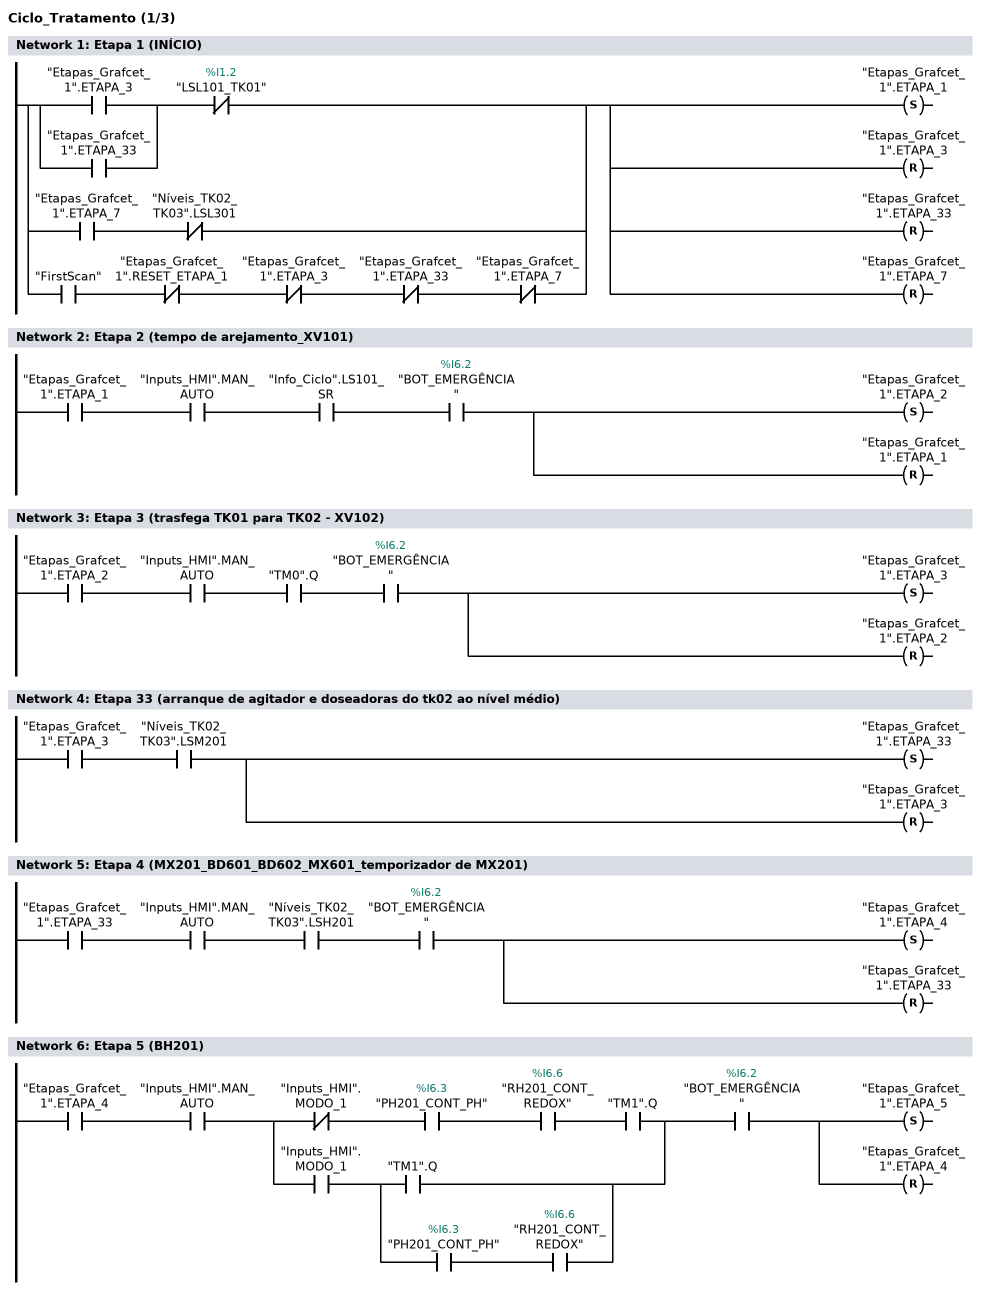
   RUNG wire#powerrail
      Contact( "Etapas_Grafcet_1".ETAPA_3 )
      wire#w1
      I_Contact( "LSL101_TK01" )
      wire#w2
      S_Coil( "Etapas_Grafcet_1".ETAPA_1 )
   END_RUNG
   RUNG wire#powerrail
      Contact( "Etapas_Grafcet_1".ETAPA_33 )
   END_RUNG wire#w1
   RUNG wire#powerrail
      Contact( "Etapas_Grafcet_1".ETAPA_7 )
      I_Contact( "Níveis_TK02_TK03".LSL301 )
   END_RUNG wire#w2
   RUNG wire#powerrail
      Contact( "FirstScan" )
      I_Contact( "Etapas_Grafcet_1".RESET_ETAPA_1 )
      I_Contact( "Etapas_Grafcet_1".ETAPA_3 )
      I_Contact( "Etapas_Grafcet_1".ETAPA_33 )
      I_Contact( "Etapas_Grafcet_1".ETAPA_7 )
   END_RUNG wire#w2
   RUNG wire#w2
      R_Coil( "Etapas_Grafcet_1".ETAPA_3 )
   END_RUNG
   RUNG wire#w2
      R_Coil( "Etapas_Grafcet_1".ETAPA_33 )
   END_RUNG
   RUNG wire#w2
      R_Coil( "Etapas_Grafcet_1".ETAPA_7 )
   END_RUNG
   // the same network as SCL:
   IF (("Etapas_Grafcet_1".ETAPA_3 OR "Etapas_Grafcet_1".ETAPA_33) AND NOT "LSL101_TK01") OR ("Etapas_Grafcet_1".ETAPA_7 AND NOT "Níveis_TK02_TK03".LSL301) OR ("FirstScan" AND NOT "Etapas_Grafcet_1".RESET_ETAPA_1 AND NOT "Etapas_Grafcet_1".ETAPA_3 AND NOT "Etapas_Grafcet_1".ETAPA_33 AND NOT "Etapas_Grafcet_1".ETAPA_7) THEN
       "Etapas_Grafcet_1".ETAPA_1 := TRUE;
   END_IF;
   #_w1 := (("Etapas_Grafcet_1".ETAPA_3 OR "Etapas_Grafcet_1".ETAPA_33) AND NOT "LSL101_TK01") OR ("Etapas_Grafcet_1".ETAPA_7 AND NOT "Níveis_TK02_TK03".LSL301) OR ("FirstScan" AND NOT "Etapas_Grafcet_1".RESET_ETAPA_1 AND NOT "Etapas_Grafcet_1".ETAPA_3 AND NOT "Etapas_Grafcet_1".ETAPA_33 AND NOT "Etapas_Grafcet_1".ETAPA_7);
   IF #_w1 THEN
       "Etapas_Grafcet_1".ETAPA_3 := FALSE;
       "Etapas_Grafcet_1".ETAPA_33 := FALSE;
       "Etapas_Grafcet_1".ETAPA_7 := FALSE;
   END_IF;
END_REGION

REGION Network 2: Etapa 2 (tempo de arejamento_XV101)
   RUNG wire#powerrail
      Contact( "Etapas_Grafcet_1".ETAPA_1 )
      Contact( "Inputs_HMI".MAN_AUTO )
      Contact( "Info_Ciclo".LS101_SR )
      Contact( "BOT_EMERGÊNCIA" )
      wire#w1
      S_Coil( "Etapas_Grafcet_1".ETAPA_2 )
   END_RUNG
   RUNG wire#w1
      R_Coil( "Etapas_Grafcet_1".ETAPA_1 )
   END_RUNG
   // the same network as SCL:
   IF "Etapas_Grafcet_1".ETAPA_1 AND "Inputs_HMI".MAN_AUTO AND "Info_Ciclo".LS101_SR AND "BOT_EMERGÊNCIA" THEN
       "Etapas_Grafcet_1".ETAPA_2 := TRUE;
       "Etapas_Grafcet_1".ETAPA_1 := FALSE;
   END_IF;
END_REGION

REGION Network 3: Etapa 3 (trasfega TK01 para TK02 - XV102)
   RUNG wire#powerrail
      Contact( "Etapas_Grafcet_1".ETAPA_2 )
      Contact( "Inputs_HMI".MAN_AUTO )
      Contact( "TM0".Q )
      Contact( "BOT_EMERGÊNCIA" )
      wire#w1
      S_Coil( "Etapas_Grafcet_1".ETAPA_3 )
   END_RUNG
   RUNG wire#w1
      R_Coil( "Etapas_Grafcet_1".ETAPA_2 )
   END_RUNG
   // the same network as SCL:
   IF "Etapas_Grafcet_1".ETAPA_2 AND "Inputs_HMI".MAN_AUTO AND "TM0".Q AND "BOT_EMERGÊNCIA" THEN
       "Etapas_Grafcet_1".ETAPA_3 := TRUE;
       "Etapas_Grafcet_1".ETAPA_2 := FALSE;
   END_IF;
END_REGION

REGION Network 4: Etapa 33 (arranque de agitador e doseadoras do tk02 ao nível médio)
   RUNG wire#powerrail
      Contact( "Etapas_Grafcet_1".ETAPA_3 )
      Contact( "Níveis_TK02_TK03".LSM201 )
      wire#w1
      S_Coil( "Etapas_Grafcet_1".ETAPA_33 )
   END_RUNG
   RUNG wire#w1
      R_Coil( "Etapas_Grafcet_1".ETAPA_3 )
   END_RUNG
   // the same network as SCL:
   IF "Etapas_Grafcet_1".ETAPA_3 AND "Níveis_TK02_TK03".LSM201 THEN
       "Etapas_Grafcet_1".ETAPA_33 := TRUE;
       "Etapas_Grafcet_1".ETAPA_3 := FALSE;
   END_IF;
END_REGION

REGION Network 5: Etapa 4 (MX201_BD601_BD602_MX601_temporizador de MX201)
   RUNG wire#powerrail
      Contact( "Etapas_Grafcet_1".ETAPA_33 )
      Contact( "Inputs_HMI".MAN_AUTO )
      Contact( "Níveis_TK02_TK03".LSH201 )
      Contact( "BOT_EMERGÊNCIA" )
      wire#w1
      S_Coil( "Etapas_Grafcet_1".ETAPA_4 )
   END_RUNG
   RUNG wire#w1
      R_Coil( "Etapas_Grafcet_1".ETAPA_33 )
   END_RUNG
   // the same network as SCL:
   IF "Etapas_Grafcet_1".ETAPA_33 AND "Inputs_HMI".MAN_AUTO AND "Níveis_TK02_TK03".LSH201 AND "BOT_EMERGÊNCIA" THEN
       "Etapas_Grafcet_1".ETAPA_4 := TRUE;
       "Etapas_Grafcet_1".ETAPA_33 := FALSE;
   END_IF;
END_REGION

REGION Network 6: Etapa 5 (BH201)
   RUNG wire#powerrail
      Contact( "Etapas_Grafcet_1".ETAPA_4 )
      Contact( "Inputs_HMI".MAN_AUTO )
      wire#w1
      I_Contact( "Inputs_HMI".MODO_1 )
      Contact( "PH201_CONT_PH" )
      Contact( "RH201_CONT_REDOX" )
      Contact( "TM1".Q )
      wire#w2
      Contact( "BOT_EMERGÊNCIA" )
      wire#w4
      S_Coil( "Etapas_Grafcet_1".ETAPA_5 )
   END_RUNG
   RUNG wire#w1
      Contact( "Inputs_HMI".MODO_1 )
      wire#w3
      Contact( "TM1".Q )
   END_RUNG wire#w2
   RUNG wire#w3
      Contact( "PH201_CONT_PH" )
      Contact( "RH201_CONT_REDOX" )
   END_RUNG wire#w2
   RUNG wire#w4
      R_Coil( "Etapas_Grafcet_1".ETAPA_4 )
   END_RUNG
   // the same network as SCL:
   IF "Etapas_Grafcet_1".ETAPA_4 AND "Inputs_HMI".MAN_AUTO AND ((NOT "Inputs_HMI".MODO_1 AND "PH201_CONT_PH" AND "RH201_CONT_REDOX" AND "TM1".Q) OR ("Inputs_HMI".MODO_1 AND ("TM1".Q OR ("PH201_CONT_PH" AND "RH201_CONT_REDOX")))) AND "BOT_EMERGÊNCIA" THEN
       "Etapas_Grafcet_1".ETAPA_5 := TRUE;
       "Etapas_Grafcet_1".ETAPA_4 := FALSE;
   END_IF;
END_REGION

REGION Network 7: Etapa 55 (arranque de agitador e doseadoras do tk03 ao nível médio)
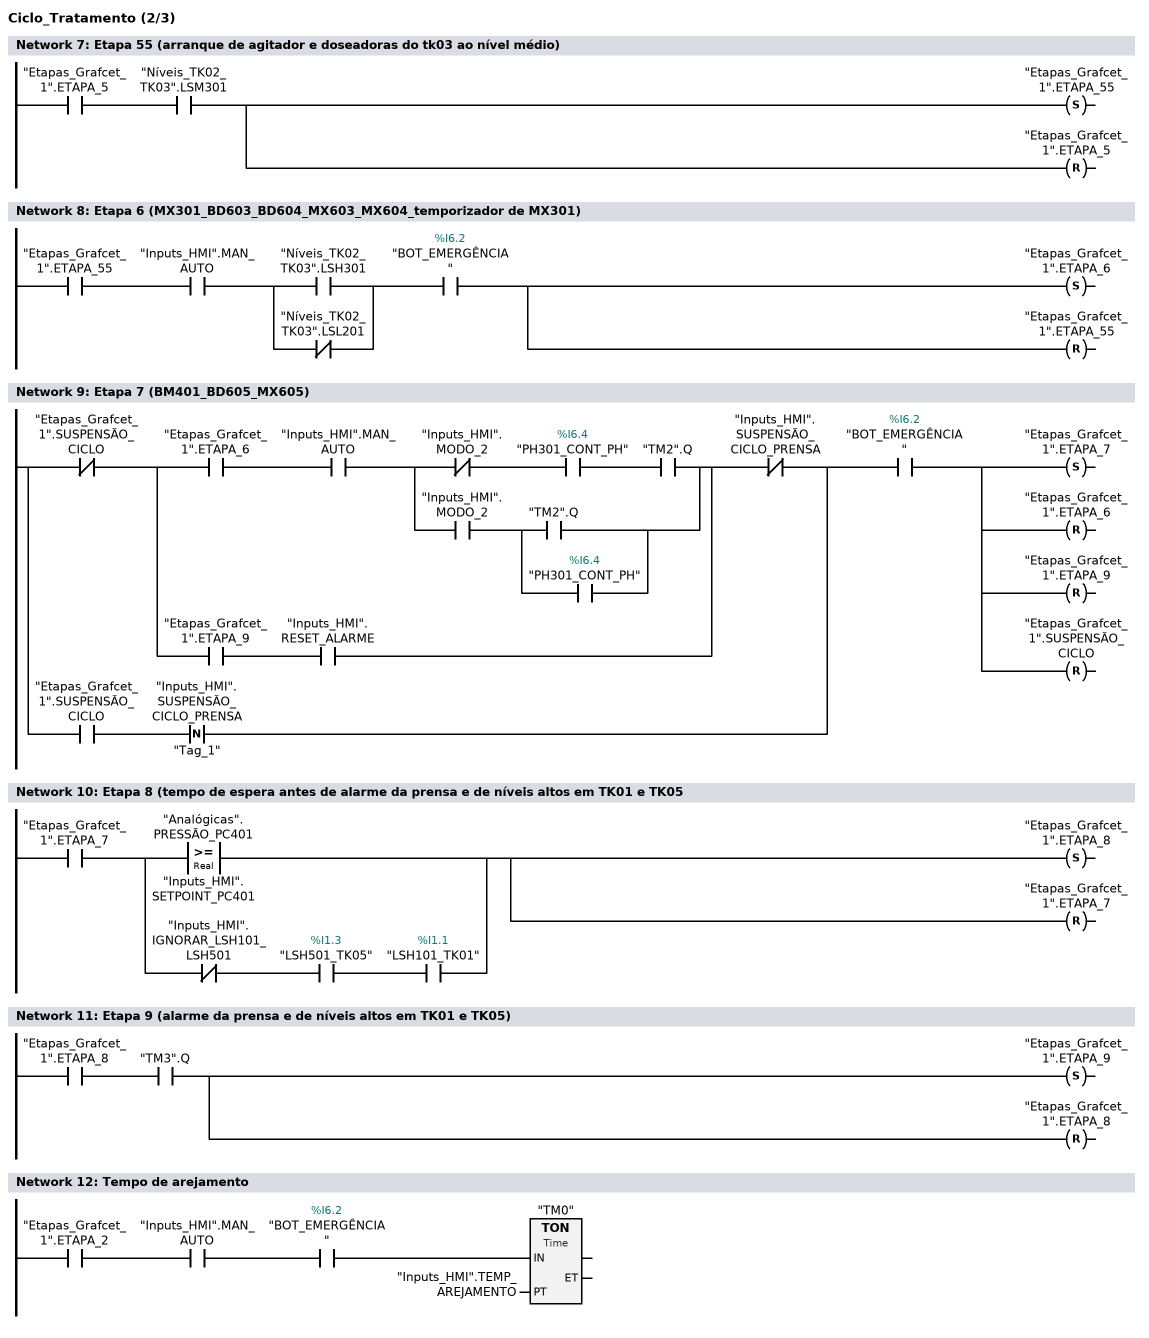
   RUNG wire#powerrail
      Contact( "Etapas_Grafcet_1".ETAPA_5 )
      Contact( "Níveis_TK02_TK03".LSM301 )
      wire#w1
      S_Coil( "Etapas_Grafcet_1".ETAPA_55 )
   END_RUNG
   RUNG wire#w1
      R_Coil( "Etapas_Grafcet_1".ETAPA_5 )
   END_RUNG
   // the same network as SCL:
   IF "Etapas_Grafcet_1".ETAPA_5 AND "Níveis_TK02_TK03".LSM301 THEN
       "Etapas_Grafcet_1".ETAPA_55 := TRUE;
       "Etapas_Grafcet_1".ETAPA_5 := FALSE;
   END_IF;
END_REGION

REGION Network 8: Etapa 6 (MX301_BD603_BD604_MX603_MX604_temporizador de MX301)
   RUNG wire#powerrail
      Contact( "Etapas_Grafcet_1".ETAPA_55 )
      Contact( "Inputs_HMI".MAN_AUTO )
      wire#w1
      Contact( "Níveis_TK02_TK03".LSH301 )
      wire#w2
      Contact( "BOT_EMERGÊNCIA" )
      wire#w3
      S_Coil( "Etapas_Grafcet_1".ETAPA_6 )
   END_RUNG
   RUNG wire#w1
      I_Contact( "Níveis_TK02_TK03".LSL201 )
   END_RUNG wire#w2
   RUNG wire#w3
      R_Coil( "Etapas_Grafcet_1".ETAPA_55 )
   END_RUNG
   // the same network as SCL:
   IF "Etapas_Grafcet_1".ETAPA_55 AND "Inputs_HMI".MAN_AUTO AND ("Níveis_TK02_TK03".LSH301 OR NOT "Níveis_TK02_TK03".LSL201) AND "BOT_EMERGÊNCIA" THEN
       "Etapas_Grafcet_1".ETAPA_6 := TRUE;
       "Etapas_Grafcet_1".ETAPA_55 := FALSE;
   END_IF;
END_REGION

REGION Network 9: Etapa 7 (BM401_BD605_MX605)
   RUNG wire#powerrail
      I_Contact( "Etapas_Grafcet_1".SUSPENSÃO_CICLO )
      wire#w1
      Contact( "Etapas_Grafcet_1".ETAPA_6 )
      Contact( "Inputs_HMI".MAN_AUTO )
      wire#w2
      I_Contact( "Inputs_HMI".MODO_2 )
      Contact( "PH301_CONT_PH" )
      Contact( "TM2".Q )
      wire#w3
      I_Contact( "Inputs_HMI".SUSPENSÃO_CICLO_PRENSA )
      wire#w5
      Contact( "BOT_EMERGÊNCIA" )
      wire#w6
      S_Coil( "Etapas_Grafcet_1".ETAPA_7 )
   END_RUNG
   RUNG wire#w2
      Contact( "Inputs_HMI".MODO_2 )
      wire#w4
      Contact( "TM2".Q )
   END_RUNG wire#w3
   RUNG wire#w4
      Contact( "PH301_CONT_PH" )
   END_RUNG wire#w3
   RUNG wire#w1
      Contact( "Etapas_Grafcet_1".ETAPA_9 )
      Contact( "Inputs_HMI".RESET_ALARME )
   END_RUNG wire#w3
   RUNG wire#powerrail
      Contact( "Etapas_Grafcet_1".SUSPENSÃO_CICLO )
      N_Contact(operand := "Inputs_HMI".SUSPENSÃO_CICLO_PRENSA, bit := "Tag_1")
   END_RUNG wire#w5
   RUNG wire#w6
      R_Coil( "Etapas_Grafcet_1".ETAPA_6 )
   END_RUNG
   RUNG wire#w6
      R_Coil( "Etapas_Grafcet_1".ETAPA_9 )
   END_RUNG
   RUNG wire#w6
      R_Coil( "Etapas_Grafcet_1".SUSPENSÃO_CICLO )
   END_RUNG
   // the same network as SCL:
   #_w1 := "Etapas_Grafcet_1".SUSPENSÃO_CICLO AND NOT "Inputs_HMI".SUSPENSÃO_CICLO_PRENSA AND "Tag_1";   // falling edge of "Inputs_HMI".SUSPENSÃO_CICLO_PRENSA
   "Tag_1" := "Inputs_HMI".SUSPENSÃO_CICLO_PRENSA;
   IF ((NOT "Etapas_Grafcet_1".SUSPENSÃO_CICLO AND (("Etapas_Grafcet_1".ETAPA_6 AND "Inputs_HMI".MAN_AUTO AND ((NOT "Inputs_HMI".MODO_2 AND "PH301_CONT_PH" AND "TM2".Q) OR ("Inputs_HMI".MODO_2 AND ("TM2".Q OR "PH301_CONT_PH")))) OR ("Etapas_Grafcet_1".ETAPA_9 AND "Inputs_HMI".RESET_ALARME)) AND NOT "Inputs_HMI".SUSPENSÃO_CICLO_PRENSA) OR #_w1) AND "BOT_EMERGÊNCIA" THEN
       "Etapas_Grafcet_1".ETAPA_7 := TRUE;
   END_IF;
   #_w2 := ((NOT "Etapas_Grafcet_1".SUSPENSÃO_CICLO AND (("Etapas_Grafcet_1".ETAPA_6 AND "Inputs_HMI".MAN_AUTO AND ((NOT "Inputs_HMI".MODO_2 AND "PH301_CONT_PH" AND "TM2".Q) OR ("Inputs_HMI".MODO_2 AND ("TM2".Q OR "PH301_CONT_PH")))) OR ("Etapas_Grafcet_1".ETAPA_9 AND "Inputs_HMI".RESET_ALARME)) AND NOT "Inputs_HMI".SUSPENSÃO_CICLO_PRENSA) OR #_w1) AND "BOT_EMERGÊNCIA";
   IF #_w2 THEN
       "Etapas_Grafcet_1".ETAPA_6 := FALSE;
       "Etapas_Grafcet_1".ETAPA_9 := FALSE;
       "Etapas_Grafcet_1".SUSPENSÃO_CICLO := FALSE;
   END_IF;
END_REGION

REGION Network 10: Etapa 8 (tempo de espera antes de alarme da prensa e de níveis altos em TK01 e TK05
   RUNG wire#powerrail
      Contact( "Etapas_Grafcet_1".ETAPA_7 )
      wire#w1
      { S7_Templates := "SrcType := Real" } GE_Contact(in1 := "Analógicas".PRESSÃO_PC401, in2 := "Inputs_HMI".SETPOINT_PC401)
      wire#w2
      S_Coil( "Etapas_Grafcet_1".ETAPA_8 )
   END_RUNG
   RUNG wire#w1
      I_Contact( "Inputs_HMI".IGNORAR_LSH101_LSH501 )
      Contact( "LSH501_TK05" )
      Contact( "LSH101_TK01" )
   END_RUNG wire#w2
   RUNG wire#w2
      R_Coil( "Etapas_Grafcet_1".ETAPA_7 )
   END_RUNG
   // the same network as SCL:
   IF "Etapas_Grafcet_1".ETAPA_7 AND (("Analógicas".PRESSÃO_PC401 >= "Inputs_HMI".SETPOINT_PC401) OR (NOT "Inputs_HMI".IGNORAR_LSH101_LSH501 AND "LSH501_TK05" AND "LSH101_TK01")) THEN
       "Etapas_Grafcet_1".ETAPA_8 := TRUE;
       "Etapas_Grafcet_1".ETAPA_7 := FALSE;
   END_IF;
END_REGION

REGION Network 11: Etapa 9 (alarme da prensa e de níveis altos em TK01 e TK05)
   RUNG wire#powerrail
      Contact( "Etapas_Grafcet_1".ETAPA_8 )
      Contact( "TM3".Q )
      wire#w1
      S_Coil( "Etapas_Grafcet_1".ETAPA_9 )
   END_RUNG
   RUNG wire#w1
      R_Coil( "Etapas_Grafcet_1".ETAPA_8 )
   END_RUNG
   // the same network as SCL:
   IF "Etapas_Grafcet_1".ETAPA_8 AND "TM3".Q THEN
       "Etapas_Grafcet_1".ETAPA_9 := TRUE;
       "Etapas_Grafcet_1".ETAPA_8 := FALSE;
   END_IF;
END_REGION

REGION Network 12: Tempo de arejamento
   RUNG wire#powerrail
      Contact( "Etapas_Grafcet_1".ETAPA_2 )
      Contact( "Inputs_HMI".MAN_AUTO )
      Contact( "BOT_EMERGÊNCIA" )
      { S7_Templates := "time_type := Time" } "TM0".TON(pt := "Inputs_HMI".TEMP_AREJAMENTO, et =>)
   END_RUNG
   // the same network as SCL:
   "TM0".TON(IN := "Etapas_Grafcet_1".ETAPA_2 AND "Inputs_HMI".MAN_AUTO AND "BOT_EMERGÊNCIA",
             PT := "Inputs_HMI".TEMP_AREJAMENTO);
END_REGION

REGION Network 13: Etapa Suspensão Ciclo
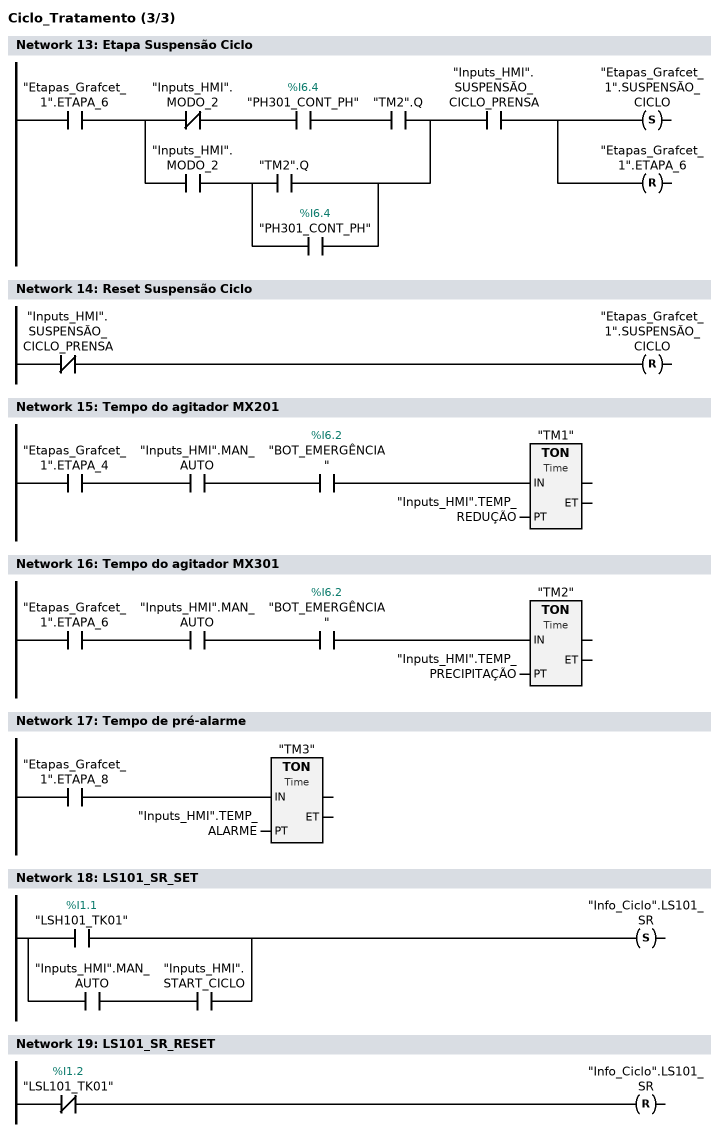
   RUNG wire#powerrail
      Contact( "Etapas_Grafcet_1".ETAPA_6 )
      wire#w1
      I_Contact( "Inputs_HMI".MODO_2 )
      Contact( "PH301_CONT_PH" )
      Contact( "TM2".Q )
      wire#w2
      Contact( "Inputs_HMI".SUSPENSÃO_CICLO_PRENSA )
      wire#w4
      S_Coil( "Etapas_Grafcet_1".SUSPENSÃO_CICLO )
   END_RUNG
   RUNG wire#w1
      Contact( "Inputs_HMI".MODO_2 )
      wire#w3
      Contact( "TM2".Q )
   END_RUNG wire#w2
   RUNG wire#w3
      Contact( "PH301_CONT_PH" )
   END_RUNG wire#w2
   RUNG wire#w4
      R_Coil( "Etapas_Grafcet_1".ETAPA_6 )
   END_RUNG
   // the same network as SCL:
   IF "Etapas_Grafcet_1".ETAPA_6 AND ((NOT "Inputs_HMI".MODO_2 AND "PH301_CONT_PH" AND "TM2".Q) OR ("Inputs_HMI".MODO_2 AND ("TM2".Q OR "PH301_CONT_PH"))) AND "Inputs_HMI".SUSPENSÃO_CICLO_PRENSA THEN
       "Etapas_Grafcet_1".SUSPENSÃO_CICLO := TRUE;
       "Etapas_Grafcet_1".ETAPA_6 := FALSE;
   END_IF;
END_REGION

REGION Network 14: Reset Suspensão Ciclo
   RUNG wire#powerrail
      I_Contact( "Inputs_HMI".SUSPENSÃO_CICLO_PRENSA )
      R_Coil( "Etapas_Grafcet_1".SUSPENSÃO_CICLO )
   END_RUNG
   // the same network as SCL:
   IF NOT "Inputs_HMI".SUSPENSÃO_CICLO_PRENSA THEN "Etapas_Grafcet_1".SUSPENSÃO_CICLO := FALSE; END_IF;
END_REGION

REGION Network 15: Tempo do agitador MX201
   RUNG wire#powerrail
      Contact( "Etapas_Grafcet_1".ETAPA_4 )
      Contact( "Inputs_HMI".MAN_AUTO )
      Contact( "BOT_EMERGÊNCIA" )
      { S7_Templates := "time_type := Time" } "TM1".TON(pt := "Inputs_HMI".TEMP_REDUÇÃO, et =>)
   END_RUNG
   // the same network as SCL:
   "TM1".TON(IN := "Etapas_Grafcet_1".ETAPA_4 AND "Inputs_HMI".MAN_AUTO AND "BOT_EMERGÊNCIA",
             PT := "Inputs_HMI".TEMP_REDUÇÃO);
END_REGION

REGION Network 16: Tempo do agitador MX301
   RUNG wire#powerrail
      Contact( "Etapas_Grafcet_1".ETAPA_6 )
      Contact( "Inputs_HMI".MAN_AUTO )
      Contact( "BOT_EMERGÊNCIA" )
      { S7_Templates := "time_type := Time" } "TM2".TON(pt := "Inputs_HMI".TEMP_PRECIPITAÇÃO, et =>)
   END_RUNG
   // the same network as SCL:
   "TM2".TON(IN := "Etapas_Grafcet_1".ETAPA_6 AND "Inputs_HMI".MAN_AUTO AND "BOT_EMERGÊNCIA",
             PT := "Inputs_HMI".TEMP_PRECIPITAÇÃO);
END_REGION

REGION Network 17: Tempo de pré-alarme
   RUNG wire#powerrail
      Contact( "Etapas_Grafcet_1".ETAPA_8 )
      { S7_Templates := "time_type := Time" } "TM3".TON(pt := "Inputs_HMI".TEMP_ALARME, et =>)
   END_RUNG
   // the same network as SCL:
   "TM3".TON(IN := "Etapas_Grafcet_1".ETAPA_8, PT := "Inputs_HMI".TEMP_ALARME);
END_REGION

REGION Network 18: LS101_SR_SET
   RUNG wire#powerrail
      Contact( "LSH101_TK01" )
      wire#w1
      S_Coil( "Info_Ciclo".LS101_SR )
   END_RUNG
   RUNG wire#powerrail
      Contact( "Inputs_HMI".MAN_AUTO )
      Contact( "Inputs_HMI".START_CICLO )
   END_RUNG wire#w1
   // the same network as SCL:
   IF "LSH101_TK01" OR ("Inputs_HMI".MAN_AUTO AND "Inputs_HMI".START_CICLO) THEN
       "Info_Ciclo".LS101_SR := TRUE;
   END_IF;
END_REGION

REGION Network 19: LS101_SR_RESET
   RUNG wire#powerrail
      I_Contact( "LSL101_TK01" )
      R_Coil( "Info_Ciclo".LS101_SR )
   END_RUNG
   // the same network as SCL:
   IF NOT "LSL101_TK01" THEN "Info_Ciclo".LS101_SR := FALSE; END_IF;
END_REGION
END_FUNCTION

FUNCTION "Estab_Níveis" : Void   // FC20, LAD
TITLE = Protege equipamentos e evita transbordo em modo manual
{ S7_Optimized_Access := 'TRUE' }
VERSION : 0.1
// stored: AutoNumber true, IsIECCheckEnabled false, SetENOAutomatically false, UDAEnableTagReadback false
BEGIN

REGION Network 1: LSL001
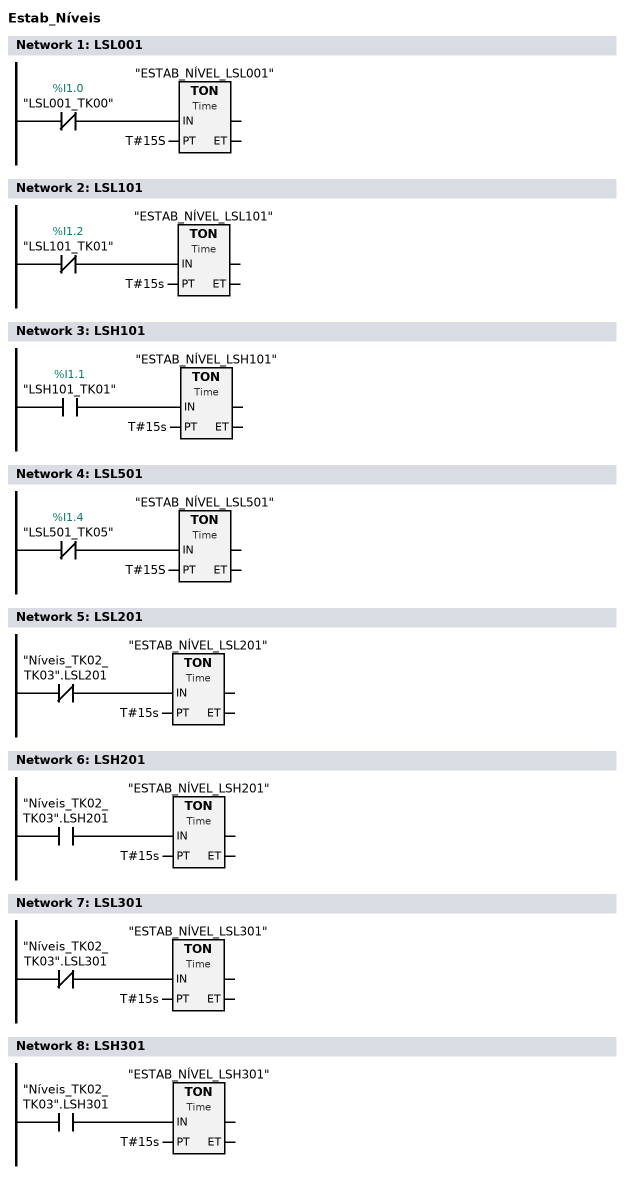
   RUNG wire#powerrail
      I_Contact( "LSL001_TK00" )
      { S7_Templates := "time_type := Time" } "ESTAB_NÍVEL_LSL001".TON(pt := T#15S, et =>)
   END_RUNG
   // the same network as SCL:
   "ESTAB_NÍVEL_LSL001".TON(IN := NOT "LSL001_TK00", PT := T#15S);
END_REGION

REGION Network 2: LSL101
   RUNG wire#powerrail
      I_Contact( "LSL101_TK01" )
      { S7_Templates := "time_type := Time" } "ESTAB_NÍVEL_LSL101".TON(pt := T#15s, et =>)
   END_RUNG
   // the same network as SCL:
   "ESTAB_NÍVEL_LSL101".TON(IN := NOT "LSL101_TK01", PT := T#15s);
END_REGION

REGION Network 3: LSH101
   RUNG wire#powerrail
      Contact( "LSH101_TK01" )
      { S7_Templates := "time_type := Time" } "ESTAB_NÍVEL_LSH101".TON(pt := T#15s, et =>)
   END_RUNG
   // the same network as SCL:
   "ESTAB_NÍVEL_LSH101".TON(IN := "LSH101_TK01", PT := T#15s);
END_REGION

REGION Network 4: LSL501
   RUNG wire#powerrail
      I_Contact( "LSL501_TK05" )
      { S7_Templates := "time_type := Time" } "ESTAB_NÍVEL_LSL501".TON(pt := T#15S, et =>)
   END_RUNG
   // the same network as SCL:
   "ESTAB_NÍVEL_LSL501".TON(IN := NOT "LSL501_TK05", PT := T#15S);
END_REGION

REGION Network 5: LSL201
   RUNG wire#powerrail
      I_Contact( "Níveis_TK02_TK03".LSL201 )
      { S7_Templates := "time_type := Time" } "ESTAB_NÍVEL_LSL201".TON(pt := T#15s, et =>)
   END_RUNG
   // the same network as SCL:
   "ESTAB_NÍVEL_LSL201".TON(IN := NOT "Níveis_TK02_TK03".LSL201, PT := T#15s);
END_REGION

REGION Network 6: LSH201
   RUNG wire#powerrail
      Contact( "Níveis_TK02_TK03".LSH201 )
      { S7_Templates := "time_type := Time" } "ESTAB_NÍVEL_LSH201".TON(pt := T#15s, et =>)
   END_RUNG
   // the same network as SCL:
   "ESTAB_NÍVEL_LSH201".TON(IN := "Níveis_TK02_TK03".LSH201, PT := T#15s);
END_REGION

REGION Network 7: LSL301
   RUNG wire#powerrail
      I_Contact( "Níveis_TK02_TK03".LSL301 )
      { S7_Templates := "time_type := Time" } "ESTAB_NÍVEL_LSL301".TON(pt := T#15s, et =>)
   END_RUNG
   // the same network as SCL:
   "ESTAB_NÍVEL_LSL301".TON(IN := NOT "Níveis_TK02_TK03".LSL301, PT := T#15s);
END_REGION

REGION Network 8: LSH301
   RUNG wire#powerrail
      Contact( "Níveis_TK02_TK03".LSH301 )
      { S7_Templates := "time_type := Time" } "ESTAB_NÍVEL_LSH301".TON(pt := T#15s, et =>)
   END_RUNG
   // the same network as SCL:
   "ESTAB_NÍVEL_LSH301".TON(IN := "Níveis_TK02_TK03".LSH301, PT := T#15s);
END_REGION
END_FUNCTION

FUNCTION "Reset_Etapas_Iniciais" : Void   // FC23, LAD
TITLE = Reset às etapas inicias em caso de falha de energia, de modo e continuar o processo do ponto onde estava
{ S7_Optimized_Access := 'TRUE' }
VERSION : 0.1
// stored: AutoNumber true, IsIECCheckEnabled false, SetENOAutomatically false, UDAEnableTagReadback false
BEGIN

REGION Network 1: Reset etapa 1
   // as etapas 3, 33 e 7 não precisam nem devem fazer reset à etapa 1. Já é feito indiretamente no FC4
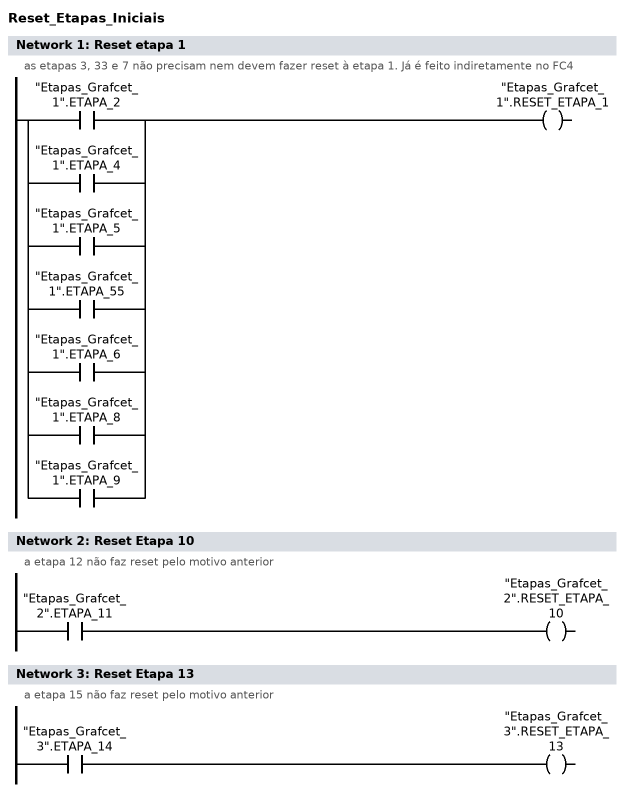
   RUNG wire#powerrail
      Contact( "Etapas_Grafcet_1".ETAPA_2 )
      wire#w1
      Coil( "Etapas_Grafcet_1".RESET_ETAPA_1 )
   END_RUNG
   RUNG wire#powerrail
      Contact( "Etapas_Grafcet_1".ETAPA_4 )
   END_RUNG wire#w1
   RUNG wire#powerrail
      Contact( "Etapas_Grafcet_1".ETAPA_5 )
   END_RUNG wire#w1
   RUNG wire#powerrail
      Contact( "Etapas_Grafcet_1".ETAPA_55 )
   END_RUNG wire#w1
   RUNG wire#powerrail
      Contact( "Etapas_Grafcet_1".ETAPA_6 )
   END_RUNG wire#w1
   RUNG wire#powerrail
      Contact( "Etapas_Grafcet_1".ETAPA_8 )
   END_RUNG wire#w1
   RUNG wire#powerrail
      Contact( "Etapas_Grafcet_1".ETAPA_9 )
   END_RUNG wire#w1
   // the same network as SCL:
   "Etapas_Grafcet_1".RESET_ETAPA_1 := "Etapas_Grafcet_1".ETAPA_2 OR "Etapas_Grafcet_1".ETAPA_4 OR "Etapas_Grafcet_1".ETAPA_5 OR "Etapas_Grafcet_1".ETAPA_55 OR "Etapas_Grafcet_1".ETAPA_6 OR "Etapas_Grafcet_1".ETAPA_8 OR "Etapas_Grafcet_1".ETAPA_9;
END_REGION

REGION Network 2: Reset Etapa 10
   // a etapa 12 não faz reset pelo motivo anterior
   RUNG wire#powerrail
      Contact( "Etapas_Grafcet_2".ETAPA_11 )
      Coil( "Etapas_Grafcet_2".RESET_ETAPA_10 )
   END_RUNG
   // the same network as SCL:
   "Etapas_Grafcet_2".RESET_ETAPA_10 := "Etapas_Grafcet_2".ETAPA_11;
END_REGION

REGION Network 3: Reset Etapa 13
   // a etapa 15 não faz reset pelo motivo anterior
   RUNG wire#powerrail
      Contact( "Etapas_Grafcet_3".ETAPA_14 )
      Coil( "Etapas_Grafcet_3".RESET_ETAPA_13 )
   END_RUNG
   // the same network as SCL:
   "Etapas_Grafcet_3".RESET_ETAPA_13 := "Etapas_Grafcet_3".ETAPA_14;
END_REGION
END_FUNCTION

FUNCTION "Saídas" : Void   // FC2, LAD
{ S7_Optimized_Access := 'TRUE' }
VERSION : 0.1
// stored: AutoNumber true, IsIECCheckEnabled false, SetENOAutomatically false, UDAEnableTagReadback false
   VAR_TEMP   // added for the SCL form of the ladder/FBD networks
      _w1 : Bool;
   END_VAR
BEGIN

REGION Network 1: bomba de alimentação ao processo BS001A
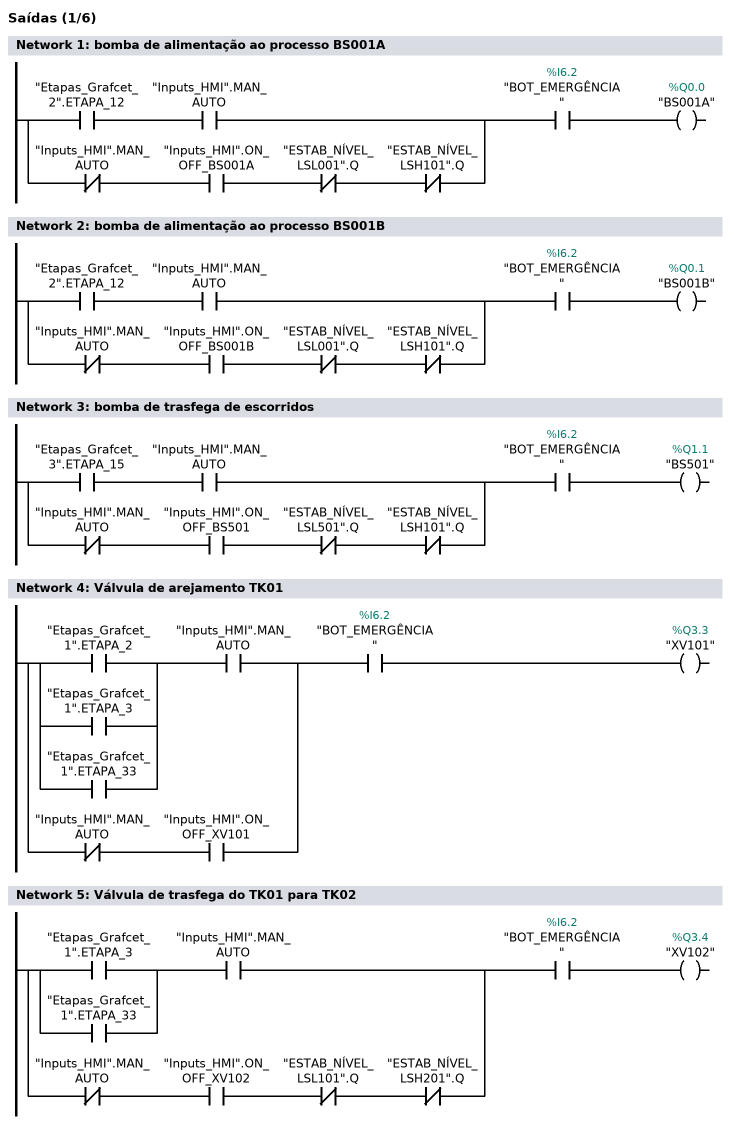
   RUNG wire#powerrail
      Contact( "Etapas_Grafcet_2".ETAPA_12 )
      Contact( "Inputs_HMI".MAN_AUTO )
      wire#w1
      Contact( "BOT_EMERGÊNCIA" )
      Coil( "BS001A" )
   END_RUNG
   RUNG wire#powerrail
      I_Contact( "Inputs_HMI".MAN_AUTO )
      Contact( "Inputs_HMI".ON_OFF_BS001A )
      I_Contact( "ESTAB_NÍVEL_LSL001".Q )
      I_Contact( "ESTAB_NÍVEL_LSH101".Q )
   END_RUNG wire#w1
   // the same network as SCL:
   "BS001A" := (("Etapas_Grafcet_2".ETAPA_12 AND "Inputs_HMI".MAN_AUTO) OR (NOT "Inputs_HMI".MAN_AUTO AND "Inputs_HMI".ON_OFF_BS001A AND NOT "ESTAB_NÍVEL_LSL001".Q AND NOT "ESTAB_NÍVEL_LSH101".Q)) AND "BOT_EMERGÊNCIA";
END_REGION

REGION Network 2: bomba de alimentação ao processo BS001B
   RUNG wire#powerrail
      Contact( "Etapas_Grafcet_2".ETAPA_12 )
      Contact( "Inputs_HMI".MAN_AUTO )
      wire#w1
      Contact( "BOT_EMERGÊNCIA" )
      Coil( "BS001B" )
   END_RUNG
   RUNG wire#powerrail
      I_Contact( "Inputs_HMI".MAN_AUTO )
      Contact( "Inputs_HMI".ON_OFF_BS001B )
      I_Contact( "ESTAB_NÍVEL_LSL001".Q )
      I_Contact( "ESTAB_NÍVEL_LSH101".Q )
   END_RUNG wire#w1
   // the same network as SCL:
   "BS001B" := (("Etapas_Grafcet_2".ETAPA_12 AND "Inputs_HMI".MAN_AUTO) OR (NOT "Inputs_HMI".MAN_AUTO AND "Inputs_HMI".ON_OFF_BS001B AND NOT "ESTAB_NÍVEL_LSL001".Q AND NOT "ESTAB_NÍVEL_LSH101".Q)) AND "BOT_EMERGÊNCIA";
END_REGION

REGION Network 3: bomba de trasfega de escorridos
   RUNG wire#powerrail
      Contact( "Etapas_Grafcet_3".ETAPA_15 )
      Contact( "Inputs_HMI".MAN_AUTO )
      wire#w1
      Contact( "BOT_EMERGÊNCIA" )
      Coil( "BS501" )
   END_RUNG
   RUNG wire#powerrail
      I_Contact( "Inputs_HMI".MAN_AUTO )
      Contact( "Inputs_HMI".ON_OFF_BS501 )
      I_Contact( "ESTAB_NÍVEL_LSL501".Q )
      I_Contact( "ESTAB_NÍVEL_LSH101".Q )
   END_RUNG wire#w1
   // the same network as SCL:
   "BS501" := (("Etapas_Grafcet_3".ETAPA_15 AND "Inputs_HMI".MAN_AUTO) OR (NOT "Inputs_HMI".MAN_AUTO AND "Inputs_HMI".ON_OFF_BS501 AND NOT "ESTAB_NÍVEL_LSL501".Q AND NOT "ESTAB_NÍVEL_LSH101".Q)) AND "BOT_EMERGÊNCIA";
END_REGION

REGION Network 4: Válvula de arejamento TK01
   RUNG wire#powerrail
      Contact( "Etapas_Grafcet_1".ETAPA_2 )
      wire#w1
      Contact( "Inputs_HMI".MAN_AUTO )
      wire#w2
      Contact( "BOT_EMERGÊNCIA" )
      Coil( "XV101" )
   END_RUNG
   RUNG wire#powerrail
      Contact( "Etapas_Grafcet_1".ETAPA_3 )
   END_RUNG wire#w1
   RUNG wire#powerrail
      Contact( "Etapas_Grafcet_1".ETAPA_33 )
   END_RUNG wire#w1
   RUNG wire#powerrail
      I_Contact( "Inputs_HMI".MAN_AUTO )
      Contact( "Inputs_HMI".ON_OFF_XV101 )
   END_RUNG wire#w2
   // the same network as SCL:
   "XV101" := ((("Etapas_Grafcet_1".ETAPA_2 OR "Etapas_Grafcet_1".ETAPA_3 OR "Etapas_Grafcet_1".ETAPA_33) AND "Inputs_HMI".MAN_AUTO) OR (NOT "Inputs_HMI".MAN_AUTO AND "Inputs_HMI".ON_OFF_XV101)) AND "BOT_EMERGÊNCIA";
END_REGION

REGION Network 5: Válvula de trasfega do TK01 para TK02
   RUNG wire#powerrail
      Contact( "Etapas_Grafcet_1".ETAPA_3 )
      wire#w1
      Contact( "Inputs_HMI".MAN_AUTO )
      wire#w2
      Contact( "BOT_EMERGÊNCIA" )
      Coil( "XV102" )
   END_RUNG
   RUNG wire#powerrail
      Contact( "Etapas_Grafcet_1".ETAPA_33 )
   END_RUNG wire#w1
   RUNG wire#powerrail
      I_Contact( "Inputs_HMI".MAN_AUTO )
      Contact( "Inputs_HMI".ON_OFF_XV102 )
      I_Contact( "ESTAB_NÍVEL_LSL101".Q )
      I_Contact( "ESTAB_NÍVEL_LSH201".Q )
   END_RUNG wire#w2
   // the same network as SCL:
   "XV102" := ((("Etapas_Grafcet_1".ETAPA_3 OR "Etapas_Grafcet_1".ETAPA_33) AND "Inputs_HMI".MAN_AUTO) OR (NOT "Inputs_HMI".MAN_AUTO AND "Inputs_HMI".ON_OFF_XV102 AND NOT "ESTAB_NÍVEL_LSL101".Q AND NOT "ESTAB_NÍVEL_LSH201".Q)) AND "BOT_EMERGÊNCIA";
END_REGION

REGION Network 6: Agitador MX201
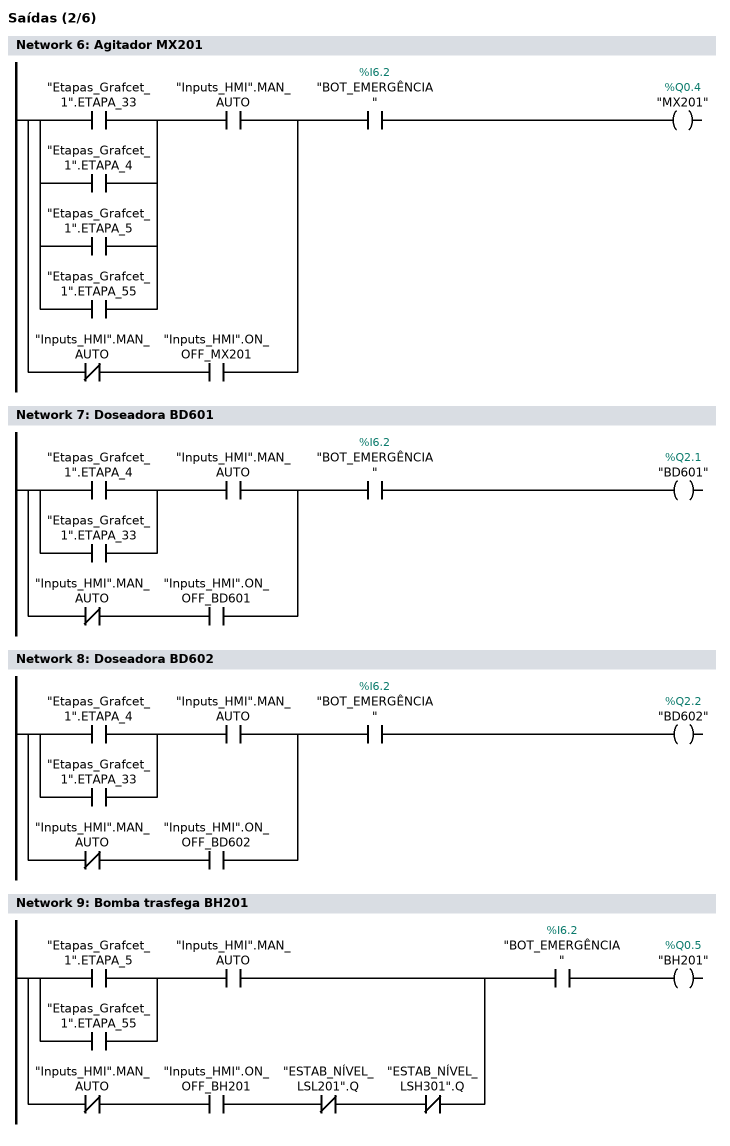
   RUNG wire#powerrail
      Contact( "Etapas_Grafcet_1".ETAPA_33 )
      wire#w1
      Contact( "Inputs_HMI".MAN_AUTO )
      wire#w2
      Contact( "BOT_EMERGÊNCIA" )
      Coil( "MX201" )
   END_RUNG
   RUNG wire#powerrail
      Contact( "Etapas_Grafcet_1".ETAPA_4 )
   END_RUNG wire#w1
   RUNG wire#powerrail
      Contact( "Etapas_Grafcet_1".ETAPA_5 )
   END_RUNG wire#w1
   RUNG wire#powerrail
      Contact( "Etapas_Grafcet_1".ETAPA_55 )
   END_RUNG wire#w1
   RUNG wire#powerrail
      I_Contact( "Inputs_HMI".MAN_AUTO )
      Contact( "Inputs_HMI".ON_OFF_MX201 )
   END_RUNG wire#w2
   // the same network as SCL:
   "MX201" := ((("Etapas_Grafcet_1".ETAPA_33 OR "Etapas_Grafcet_1".ETAPA_4 OR "Etapas_Grafcet_1".ETAPA_5 OR "Etapas_Grafcet_1".ETAPA_55) AND "Inputs_HMI".MAN_AUTO) OR (NOT "Inputs_HMI".MAN_AUTO AND "Inputs_HMI".ON_OFF_MX201)) AND "BOT_EMERGÊNCIA";
END_REGION

REGION Network 7: Doseadora BD601
   RUNG wire#powerrail
      Contact( "Etapas_Grafcet_1".ETAPA_4 )
      wire#w1
      Contact( "Inputs_HMI".MAN_AUTO )
      wire#w2
      Contact( "BOT_EMERGÊNCIA" )
      Coil( "BD601" )
   END_RUNG
   RUNG wire#powerrail
      Contact( "Etapas_Grafcet_1".ETAPA_33 )
   END_RUNG wire#w1
   RUNG wire#powerrail
      I_Contact( "Inputs_HMI".MAN_AUTO )
      Contact( "Inputs_HMI".ON_OFF_BD601 )
   END_RUNG wire#w2
   // the same network as SCL:
   "BD601" := ((("Etapas_Grafcet_1".ETAPA_4 OR "Etapas_Grafcet_1".ETAPA_33) AND "Inputs_HMI".MAN_AUTO) OR (NOT "Inputs_HMI".MAN_AUTO AND "Inputs_HMI".ON_OFF_BD601)) AND "BOT_EMERGÊNCIA";
END_REGION

REGION Network 8: Doseadora BD602
   RUNG wire#powerrail
      Contact( "Etapas_Grafcet_1".ETAPA_4 )
      wire#w1
      Contact( "Inputs_HMI".MAN_AUTO )
      wire#w2
      Contact( "BOT_EMERGÊNCIA" )
      Coil( "BD602" )
   END_RUNG
   RUNG wire#powerrail
      Contact( "Etapas_Grafcet_1".ETAPA_33 )
   END_RUNG wire#w1
   RUNG wire#powerrail
      I_Contact( "Inputs_HMI".MAN_AUTO )
      Contact( "Inputs_HMI".ON_OFF_BD602 )
   END_RUNG wire#w2
   // the same network as SCL:
   "BD602" := ((("Etapas_Grafcet_1".ETAPA_4 OR "Etapas_Grafcet_1".ETAPA_33) AND "Inputs_HMI".MAN_AUTO) OR (NOT "Inputs_HMI".MAN_AUTO AND "Inputs_HMI".ON_OFF_BD602)) AND "BOT_EMERGÊNCIA";
END_REGION

REGION Network 9: Bomba trasfega BH201
   RUNG wire#powerrail
      Contact( "Etapas_Grafcet_1".ETAPA_5 )
      wire#w1
      Contact( "Inputs_HMI".MAN_AUTO )
      wire#w2
      Contact( "BOT_EMERGÊNCIA" )
      Coil( "BH201" )
   END_RUNG
   RUNG wire#powerrail
      Contact( "Etapas_Grafcet_1".ETAPA_55 )
   END_RUNG wire#w1
   RUNG wire#powerrail
      I_Contact( "Inputs_HMI".MAN_AUTO )
      Contact( "Inputs_HMI".ON_OFF_BH201 )
      I_Contact( "ESTAB_NÍVEL_LSL201".Q )
      I_Contact( "ESTAB_NÍVEL_LSH301".Q )
   END_RUNG wire#w2
   // the same network as SCL:
   "BH201" := ((("Etapas_Grafcet_1".ETAPA_5 OR "Etapas_Grafcet_1".ETAPA_55) AND "Inputs_HMI".MAN_AUTO) OR (NOT "Inputs_HMI".MAN_AUTO AND "Inputs_HMI".ON_OFF_BH201 AND NOT "ESTAB_NÍVEL_LSL201".Q AND NOT "ESTAB_NÍVEL_LSH301".Q)) AND "BOT_EMERGÊNCIA";
END_REGION

REGION Network 10: Agitador MX301
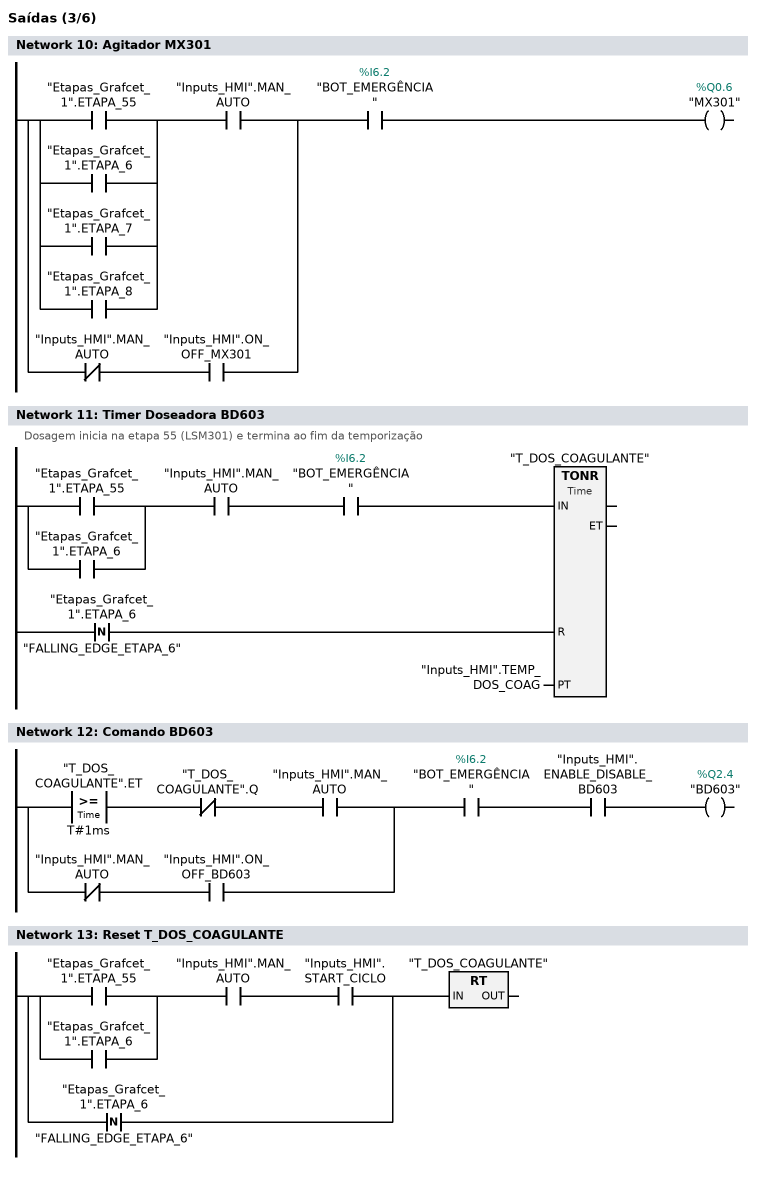
   RUNG wire#powerrail
      Contact( "Etapas_Grafcet_1".ETAPA_55 )
      wire#w1
      Contact( "Inputs_HMI".MAN_AUTO )
      wire#w2
      Contact( "BOT_EMERGÊNCIA" )
      Coil( "MX301" )
   END_RUNG
   RUNG wire#powerrail
      Contact( "Etapas_Grafcet_1".ETAPA_6 )
   END_RUNG wire#w1
   RUNG wire#powerrail
      Contact( "Etapas_Grafcet_1".ETAPA_7 )
   END_RUNG wire#w1
   RUNG wire#powerrail
      Contact( "Etapas_Grafcet_1".ETAPA_8 )
   END_RUNG wire#w1
   RUNG wire#powerrail
      I_Contact( "Inputs_HMI".MAN_AUTO )
      Contact( "Inputs_HMI".ON_OFF_MX301 )
   END_RUNG wire#w2
   // the same network as SCL:
   "MX301" := ((("Etapas_Grafcet_1".ETAPA_55 OR "Etapas_Grafcet_1".ETAPA_6 OR "Etapas_Grafcet_1".ETAPA_7 OR "Etapas_Grafcet_1".ETAPA_8) AND "Inputs_HMI".MAN_AUTO) OR (NOT "Inputs_HMI".MAN_AUTO AND "Inputs_HMI".ON_OFF_MX301)) AND "BOT_EMERGÊNCIA";
END_REGION

REGION Network 11: Timer Doseadora BD603
   // Dosagem inicia na etapa 55 (LSM301) e termina ao fim da temporização
   RUNG wire#powerrail
      Contact( "Etapas_Grafcet_1".ETAPA_55 )
      wire#w1
      Contact( "Inputs_HMI".MAN_AUTO )
      Contact( "BOT_EMERGÊNCIA" )
      { S7_Templates := "time_type := Time" } "T_DOS_COAGULANTE".TONR(r := wire#w2, pt := "Inputs_HMI".TEMP_DOS_COAG, et =>)
   END_RUNG
   RUNG wire#powerrail
      Contact( "Etapas_Grafcet_1".ETAPA_6 )
   END_RUNG wire#w1
   RUNG wire#powerrail
      N_Contact(operand := "Etapas_Grafcet_1".ETAPA_6, bit := "FALLING_EDGE_ETAPA_6")
   END_RUNG wire#w2
   // the same network as SCL:
   #_w1 := NOT "Etapas_Grafcet_1".ETAPA_6 AND "FALLING_EDGE_ETAPA_6";   // falling edge of "Etapas_Grafcet_1".ETAPA_6
   "FALLING_EDGE_ETAPA_6" := "Etapas_Grafcet_1".ETAPA_6;
   "T_DOS_COAGULANTE".TONR(IN := ("Etapas_Grafcet_1".ETAPA_55 OR "Etapas_Grafcet_1".ETAPA_6) AND "Inputs_HMI".MAN_AUTO AND "BOT_EMERGÊNCIA",
                           R := #_w1,
                           PT := "Inputs_HMI".TEMP_DOS_COAG);
END_REGION

REGION Network 12: Comando BD603
   RUNG wire#powerrail
      { S7_Templates := "SrcType := Time" } GE_Contact(in1 := "T_DOS_COAGULANTE".ET, in2 := T#1ms)
      I_Contact( "T_DOS_COAGULANTE".Q )
      Contact( "Inputs_HMI".MAN_AUTO )
      wire#w1
      Contact( "BOT_EMERGÊNCIA" )
      Contact( "Inputs_HMI".ENABLE_DISABLE_BD603 )
      Coil( "BD603" )
   END_RUNG
   RUNG wire#powerrail
      I_Contact( "Inputs_HMI".MAN_AUTO )
      Contact( "Inputs_HMI".ON_OFF_BD603 )
   END_RUNG wire#w1
   // the same network as SCL:
   "BD603" := ((("T_DOS_COAGULANTE".ET >= T#1ms) AND NOT "T_DOS_COAGULANTE".Q AND "Inputs_HMI".MAN_AUTO) OR (NOT "Inputs_HMI".MAN_AUTO AND "Inputs_HMI".ON_OFF_BD603)) AND "BOT_EMERGÊNCIA" AND "Inputs_HMI".ENABLE_DISABLE_BD603;
END_REGION

REGION Network 13: Reset T_DOS_COAGULANTE
   RUNG wire#powerrail
      Contact( "Etapas_Grafcet_1".ETAPA_55 )
      wire#w1
      Contact( "Inputs_HMI".MAN_AUTO )
      Contact( "Inputs_HMI".START_CICLO )
      wire#w2
      RT_Coil( "T_DOS_COAGULANTE" )
   END_RUNG
   RUNG wire#powerrail
      Contact( "Etapas_Grafcet_1".ETAPA_6 )
   END_RUNG wire#w1
   RUNG wire#powerrail
      N_Contact(operand := "Etapas_Grafcet_1".ETAPA_6, bit := "FALLING_EDGE_ETAPA_6")
   END_RUNG wire#w2
   // the same network as SCL:
   #_w1 := NOT "Etapas_Grafcet_1".ETAPA_6 AND "FALLING_EDGE_ETAPA_6";   // falling edge of "Etapas_Grafcet_1".ETAPA_6
   "FALLING_EDGE_ETAPA_6" := "Etapas_Grafcet_1".ETAPA_6;
   IF (("Etapas_Grafcet_1".ETAPA_55 OR "Etapas_Grafcet_1".ETAPA_6) AND "Inputs_HMI".MAN_AUTO AND "Inputs_HMI".START_CICLO) OR #_w1 THEN
       RESET_TIMER("T_DOS_COAGULANTE");
   END_IF;
END_REGION

REGION Network 14: Doseadora BD604
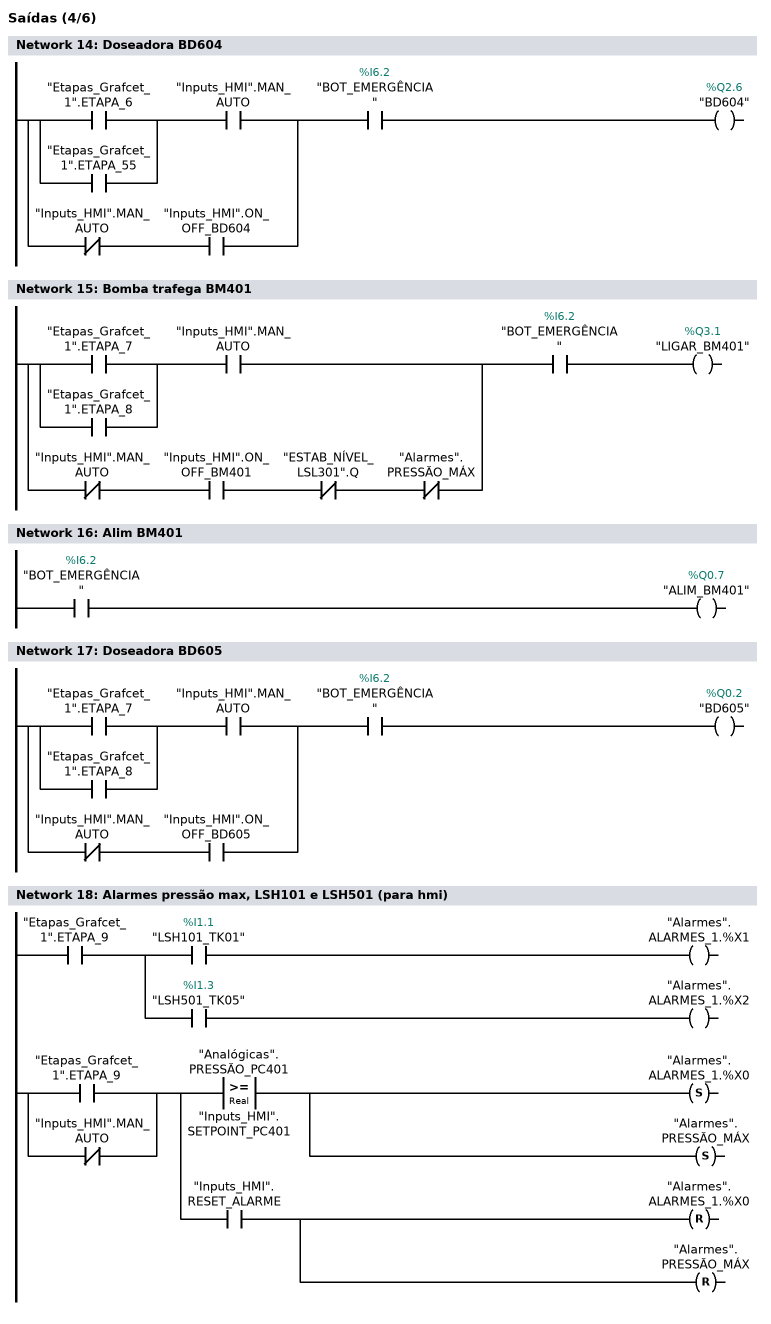
   RUNG wire#powerrail
      Contact( "Etapas_Grafcet_1".ETAPA_6 )
      wire#w1
      Contact( "Inputs_HMI".MAN_AUTO )
      wire#w2
      Contact( "BOT_EMERGÊNCIA" )
      Coil( "BD604" )
   END_RUNG
   RUNG wire#powerrail
      Contact( "Etapas_Grafcet_1".ETAPA_55 )
   END_RUNG wire#w1
   RUNG wire#powerrail
      I_Contact( "Inputs_HMI".MAN_AUTO )
      Contact( "Inputs_HMI".ON_OFF_BD604 )
   END_RUNG wire#w2
   // the same network as SCL:
   "BD604" := ((("Etapas_Grafcet_1".ETAPA_6 OR "Etapas_Grafcet_1".ETAPA_55) AND "Inputs_HMI".MAN_AUTO) OR (NOT "Inputs_HMI".MAN_AUTO AND "Inputs_HMI".ON_OFF_BD604)) AND "BOT_EMERGÊNCIA";
END_REGION

REGION Network 15: Bomba trafega BM401
   RUNG wire#powerrail
      Contact( "Etapas_Grafcet_1".ETAPA_7 )
      wire#w1
      Contact( "Inputs_HMI".MAN_AUTO )
      wire#w2
      Contact( "BOT_EMERGÊNCIA" )
      Coil( "LIGAR_BM401" )
   END_RUNG
   RUNG wire#powerrail
      Contact( "Etapas_Grafcet_1".ETAPA_8 )
   END_RUNG wire#w1
   RUNG wire#powerrail
      I_Contact( "Inputs_HMI".MAN_AUTO )
      Contact( "Inputs_HMI".ON_OFF_BM401 )
      I_Contact( "ESTAB_NÍVEL_LSL301".Q )
      I_Contact( "Alarmes".PRESSÃO_MÁX )
   END_RUNG wire#w2
   // the same network as SCL:
   "LIGAR_BM401" := ((("Etapas_Grafcet_1".ETAPA_7 OR "Etapas_Grafcet_1".ETAPA_8) AND "Inputs_HMI".MAN_AUTO) OR (NOT "Inputs_HMI".MAN_AUTO AND "Inputs_HMI".ON_OFF_BM401 AND NOT "ESTAB_NÍVEL_LSL301".Q AND NOT "Alarmes".PRESSÃO_MÁX)) AND "BOT_EMERGÊNCIA";
END_REGION

REGION Network 16: Alim BM401
   RUNG wire#powerrail
      Contact( "BOT_EMERGÊNCIA" )
      Coil( "ALIM_BM401" )
   END_RUNG
   // the same network as SCL:
   "ALIM_BM401" := "BOT_EMERGÊNCIA";
END_REGION

REGION Network 17: Doseadora BD605
   RUNG wire#powerrail
      Contact( "Etapas_Grafcet_1".ETAPA_7 )
      wire#w1
      Contact( "Inputs_HMI".MAN_AUTO )
      wire#w2
      Contact( "BOT_EMERGÊNCIA" )
      Coil( "BD605" )
   END_RUNG
   RUNG wire#powerrail
      Contact( "Etapas_Grafcet_1".ETAPA_8 )
   END_RUNG wire#w1
   RUNG wire#powerrail
      I_Contact( "Inputs_HMI".MAN_AUTO )
      Contact( "Inputs_HMI".ON_OFF_BD605 )
   END_RUNG wire#w2
   // the same network as SCL:
   "BD605" := ((("Etapas_Grafcet_1".ETAPA_7 OR "Etapas_Grafcet_1".ETAPA_8) AND "Inputs_HMI".MAN_AUTO) OR (NOT "Inputs_HMI".MAN_AUTO AND "Inputs_HMI".ON_OFF_BD605)) AND "BOT_EMERGÊNCIA";
END_REGION

REGION Network 18: Alarmes pressão max, LSH101 e LSH501 (para hmi)
   RUNG wire#powerrail
      Contact( "Etapas_Grafcet_1".ETAPA_9 )
      wire#w1
      Contact( "LSH101_TK01" )
      Coil( "Alarmes".ALARMES_1.%X1 )
   END_RUNG
   RUNG wire#w1
      Contact( "LSH501_TK05" )
      Coil( "Alarmes".ALARMES_1.%X2 )
   END_RUNG
   RUNG wire#powerrail
      Contact( "Etapas_Grafcet_1".ETAPA_9 )
      wire#w2
      { S7_Templates := "SrcType := Real" } GE_Contact(in1 := "Analógicas".PRESSÃO_PC401, in2 := "Inputs_HMI".SETPOINT_PC401)
      wire#w3
      S_Coil( "Alarmes".ALARMES_1.%X0 )
   END_RUNG
   RUNG wire#powerrail
      I_Contact( "Inputs_HMI".MAN_AUTO )
   END_RUNG wire#w2
   RUNG wire#w3
      S_Coil( "Alarmes".PRESSÃO_MÁX )
   END_RUNG
   RUNG wire#w2
      Contact( "Inputs_HMI".RESET_ALARME )
      wire#w4
      R_Coil( "Alarmes".ALARMES_1.%X0 )
   END_RUNG
   RUNG wire#w4
      R_Coil( "Alarmes".PRESSÃO_MÁX )
   END_RUNG
   // the same network as SCL:
   "Alarmes".ALARMES_1.%X1 := "Etapas_Grafcet_1".ETAPA_9 AND "LSH101_TK01";
   "Alarmes".ALARMES_1.%X2 := "Etapas_Grafcet_1".ETAPA_9 AND "LSH501_TK05";
   #_w1 := "Etapas_Grafcet_1".ETAPA_9 OR NOT "Inputs_HMI".MAN_AUTO;
   IF #_w1 AND ("Analógicas".PRESSÃO_PC401 >= "Inputs_HMI".SETPOINT_PC401) THEN
       "Alarmes".ALARMES_1.%X0 := TRUE;
       "Alarmes".PRESSÃO_MÁX := TRUE;
   END_IF;
   IF #_w1 AND "Inputs_HMI".RESET_ALARME THEN
       "Alarmes".ALARMES_1.%X0 := FALSE;
       "Alarmes".PRESSÃO_MÁX := FALSE;
   END_IF;
END_REGION

REGION Network 19: Alarme (luminoso)
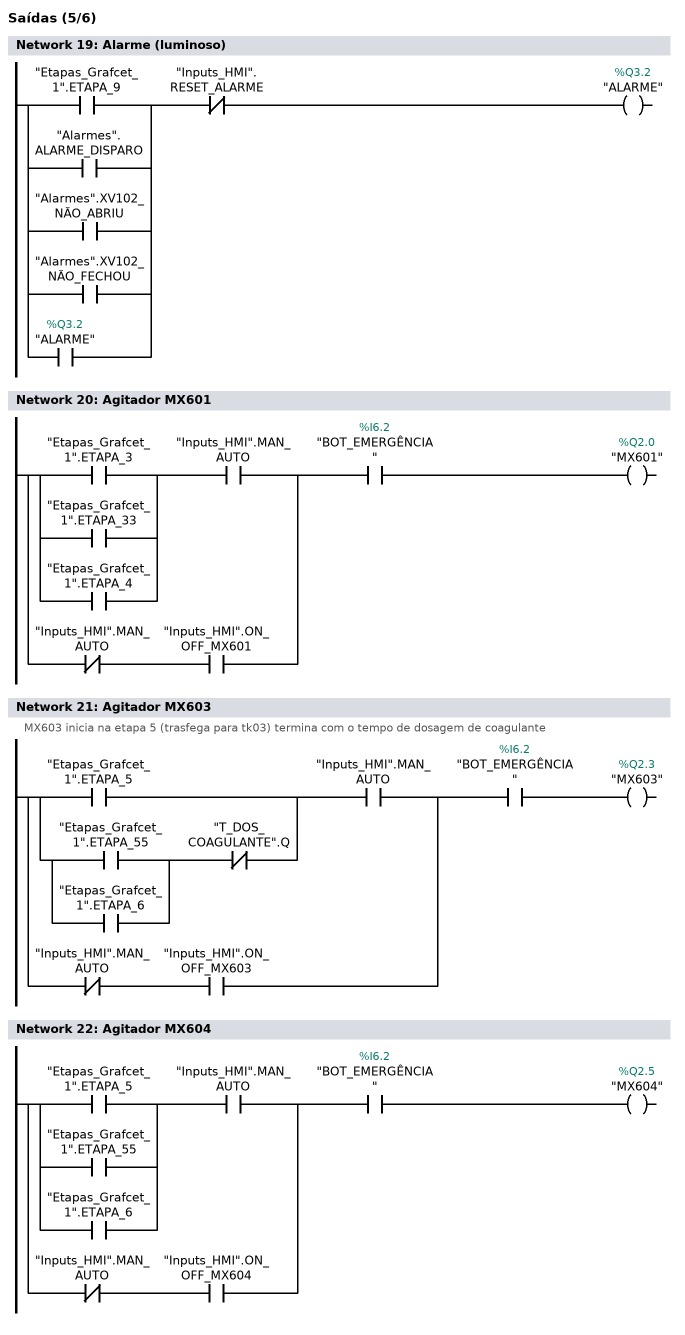
   RUNG wire#powerrail
      Contact( "Etapas_Grafcet_1".ETAPA_9 )
      wire#w1
      I_Contact( "Inputs_HMI".RESET_ALARME )
      Coil( "ALARME" )
   END_RUNG
   RUNG wire#powerrail
      Contact( "Alarmes".ALARME_DISPARO )
   END_RUNG wire#w1
   RUNG wire#powerrail
      Contact( "Alarmes".XV102_NÃO_ABRIU )
   END_RUNG wire#w1
   RUNG wire#powerrail
      Contact( "Alarmes".XV102_NÃO_FECHOU )
   END_RUNG wire#w1
   RUNG wire#powerrail
      Contact( "ALARME" )
   END_RUNG wire#w1
   // the same network as SCL:
   "ALARME" := ("Etapas_Grafcet_1".ETAPA_9 OR "Alarmes".ALARME_DISPARO OR "Alarmes".XV102_NÃO_ABRIU OR "Alarmes".XV102_NÃO_FECHOU OR "ALARME") AND NOT "Inputs_HMI".RESET_ALARME;
END_REGION

REGION Network 20: Agitador MX601
   RUNG wire#powerrail
      Contact( "Etapas_Grafcet_1".ETAPA_3 )
      wire#w1
      Contact( "Inputs_HMI".MAN_AUTO )
      wire#w2
      Contact( "BOT_EMERGÊNCIA" )
      Coil( "MX601" )
   END_RUNG
   RUNG wire#powerrail
      Contact( "Etapas_Grafcet_1".ETAPA_33 )
   END_RUNG wire#w1
   RUNG wire#powerrail
      Contact( "Etapas_Grafcet_1".ETAPA_4 )
   END_RUNG wire#w1
   RUNG wire#powerrail
      I_Contact( "Inputs_HMI".MAN_AUTO )
      Contact( "Inputs_HMI".ON_OFF_MX601 )
   END_RUNG wire#w2
   // the same network as SCL:
   "MX601" := ((("Etapas_Grafcet_1".ETAPA_3 OR "Etapas_Grafcet_1".ETAPA_33 OR "Etapas_Grafcet_1".ETAPA_4) AND "Inputs_HMI".MAN_AUTO) OR (NOT "Inputs_HMI".MAN_AUTO AND "Inputs_HMI".ON_OFF_MX601)) AND "BOT_EMERGÊNCIA";
END_REGION

REGION Network 21: Agitador MX603
   // MX603 inicia na etapa 5 (trasfega para tk03) termina com o tempo de dosagem de coagulante
   RUNG wire#powerrail
      Contact( "Etapas_Grafcet_1".ETAPA_5 )
      wire#w1
      Contact( "Inputs_HMI".MAN_AUTO )
      wire#w3
      Contact( "BOT_EMERGÊNCIA" )
      Coil( "MX603" )
   END_RUNG
   RUNG wire#powerrail
      Contact( "Etapas_Grafcet_1".ETAPA_55 )
      wire#w2
      I_Contact( "T_DOS_COAGULANTE".Q )
   END_RUNG wire#w1
   RUNG wire#powerrail
      Contact( "Etapas_Grafcet_1".ETAPA_6 )
   END_RUNG wire#w2
   RUNG wire#powerrail
      I_Contact( "Inputs_HMI".MAN_AUTO )
      Contact( "Inputs_HMI".ON_OFF_MX603 )
   END_RUNG wire#w3
   // the same network as SCL:
   "MX603" := ((("Etapas_Grafcet_1".ETAPA_5 OR (("Etapas_Grafcet_1".ETAPA_55 OR "Etapas_Grafcet_1".ETAPA_6) AND NOT "T_DOS_COAGULANTE".Q)) AND "Inputs_HMI".MAN_AUTO) OR (NOT "Inputs_HMI".MAN_AUTO AND "Inputs_HMI".ON_OFF_MX603)) AND "BOT_EMERGÊNCIA";
END_REGION

REGION Network 22: Agitador MX604
   RUNG wire#powerrail
      Contact( "Etapas_Grafcet_1".ETAPA_5 )
      wire#w1
      Contact( "Inputs_HMI".MAN_AUTO )
      wire#w2
      Contact( "BOT_EMERGÊNCIA" )
      Coil( "MX604" )
   END_RUNG
   RUNG wire#powerrail
      Contact( "Etapas_Grafcet_1".ETAPA_55 )
   END_RUNG wire#w1
   RUNG wire#powerrail
      Contact( "Etapas_Grafcet_1".ETAPA_6 )
   END_RUNG wire#w1
   RUNG wire#powerrail
      I_Contact( "Inputs_HMI".MAN_AUTO )
      Contact( "Inputs_HMI".ON_OFF_MX604 )
   END_RUNG wire#w2
   // the same network as SCL:
   "MX604" := ((("Etapas_Grafcet_1".ETAPA_5 OR "Etapas_Grafcet_1".ETAPA_55 OR "Etapas_Grafcet_1".ETAPA_6) AND "Inputs_HMI".MAN_AUTO) OR (NOT "Inputs_HMI".MAN_AUTO AND "Inputs_HMI".ON_OFF_MX604)) AND "BOT_EMERGÊNCIA";
END_REGION

REGION Network 23: Agitador MX605
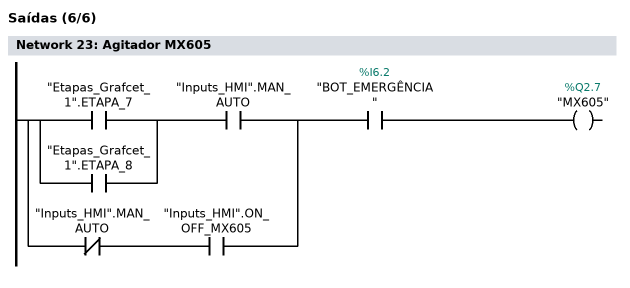
   RUNG wire#powerrail
      Contact( "Etapas_Grafcet_1".ETAPA_7 )
      wire#w1
      Contact( "Inputs_HMI".MAN_AUTO )
      wire#w2
      Contact( "BOT_EMERGÊNCIA" )
      Coil( "MX605" )
   END_RUNG
   RUNG wire#powerrail
      Contact( "Etapas_Grafcet_1".ETAPA_8 )
   END_RUNG wire#w1
   RUNG wire#powerrail
      I_Contact( "Inputs_HMI".MAN_AUTO )
      Contact( "Inputs_HMI".ON_OFF_MX605 )
   END_RUNG wire#w2
   // the same network as SCL:
   "MX605" := ((("Etapas_Grafcet_1".ETAPA_7 OR "Etapas_Grafcet_1".ETAPA_8) AND "Inputs_HMI".MAN_AUTO) OR (NOT "Inputs_HMI".MAN_AUTO AND "Inputs_HMI".ON_OFF_MX605)) AND "BOT_EMERGÊNCIA";
END_REGION
END_FUNCTION

FUNCTION "Trasfega_Escorridos" : Void   // FC3, LAD
{ S7_Optimized_Access := 'TRUE' }
VERSION : 0.1
// stored: AutoNumber true, IsIECCheckEnabled false, SetENOAutomatically false, UDAEnableTagReadback false
BEGIN

REGION Network 1: Etapa 13 (INÍCIO)
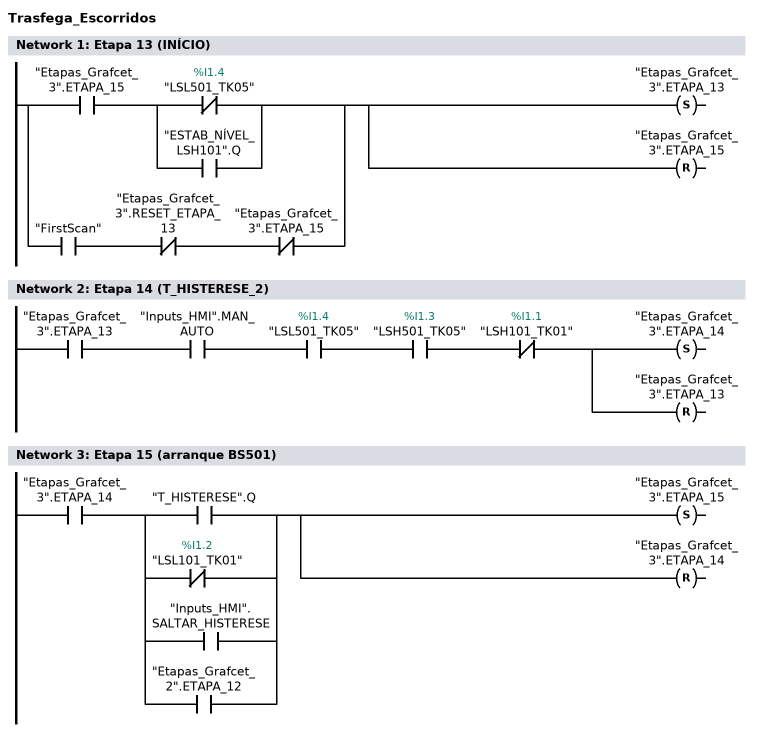
   RUNG wire#powerrail
      Contact( "Etapas_Grafcet_3".ETAPA_15 )
      wire#w1
      I_Contact( "LSL501_TK05" )
      wire#w2
      S_Coil( "Etapas_Grafcet_3".ETAPA_13 )
   END_RUNG
   RUNG wire#w1
      Contact( "ESTAB_NÍVEL_LSH101".Q )
   END_RUNG wire#w2
   RUNG wire#powerrail
      Contact( "FirstScan" )
      I_Contact( "Etapas_Grafcet_3".RESET_ETAPA_13 )
      I_Contact( "Etapas_Grafcet_3".ETAPA_15 )
   END_RUNG wire#w2
   RUNG wire#w2
      R_Coil( "Etapas_Grafcet_3".ETAPA_15 )
   END_RUNG
   // the same network as SCL:
   IF ("Etapas_Grafcet_3".ETAPA_15 AND (NOT "LSL501_TK05" OR "ESTAB_NÍVEL_LSH101".Q)) OR ("FirstScan" AND NOT "Etapas_Grafcet_3".RESET_ETAPA_13 AND NOT "Etapas_Grafcet_3".ETAPA_15) THEN
       "Etapas_Grafcet_3".ETAPA_13 := TRUE;
       "Etapas_Grafcet_3".ETAPA_15 := FALSE;
   END_IF;
END_REGION

REGION Network 2: Etapa 14 (T_HISTERESE_2)
   RUNG wire#powerrail
      Contact( "Etapas_Grafcet_3".ETAPA_13 )
      Contact( "Inputs_HMI".MAN_AUTO )
      Contact( "LSL501_TK05" )
      Contact( "LSH501_TK05" )
      I_Contact( "LSH101_TK01" )
      wire#w1
      S_Coil( "Etapas_Grafcet_3".ETAPA_14 )
   END_RUNG
   RUNG wire#w1
      R_Coil( "Etapas_Grafcet_3".ETAPA_13 )
   END_RUNG
   // the same network as SCL:
   IF "Etapas_Grafcet_3".ETAPA_13 AND "Inputs_HMI".MAN_AUTO AND "LSL501_TK05" AND "LSH501_TK05" AND NOT "LSH101_TK01" THEN
       "Etapas_Grafcet_3".ETAPA_14 := TRUE;
       "Etapas_Grafcet_3".ETAPA_13 := FALSE;
   END_IF;
END_REGION

REGION Network 3: Etapa 15 (arranque BS501)
   RUNG wire#powerrail
      Contact( "Etapas_Grafcet_3".ETAPA_14 )
      wire#w1
      Contact( "T_HISTERESE".Q )
      wire#w2
      S_Coil( "Etapas_Grafcet_3".ETAPA_15 )
   END_RUNG
   RUNG wire#w1
      I_Contact( "LSL101_TK01" )
   END_RUNG wire#w2
   RUNG wire#w1
      Contact( "Inputs_HMI".SALTAR_HISTERESE )
   END_RUNG wire#w2
   RUNG wire#w1
      Contact( "Etapas_Grafcet_2".ETAPA_12 )
   END_RUNG wire#w2
   RUNG wire#w2
      R_Coil( "Etapas_Grafcet_3".ETAPA_14 )
   END_RUNG
   // the same network as SCL:
   IF "Etapas_Grafcet_3".ETAPA_14 AND ("T_HISTERESE".Q OR NOT "LSL101_TK01" OR "Inputs_HMI".SALTAR_HISTERESE OR "Etapas_Grafcet_2".ETAPA_12) THEN
       "Etapas_Grafcet_3".ETAPA_15 := TRUE;
       "Etapas_Grafcet_3".ETAPA_14 := FALSE;
   END_IF;
END_REGION
END_FUNCTION

FUNCTION "Comando_Avaria_Bombas" : Void   // FC21, LAD
{ S7_Optimized_Access := 'TRUE' }
VERSION : 0.1
// stored: AutoNumber true, IsIECCheckEnabled false, SetENOAutomatically false, UDAEnableTagReadback false
BEGIN

REGION Network 1: Se Bomba 1 Avariar ficam a trabalhar a Bomba 2 e Bomba 3
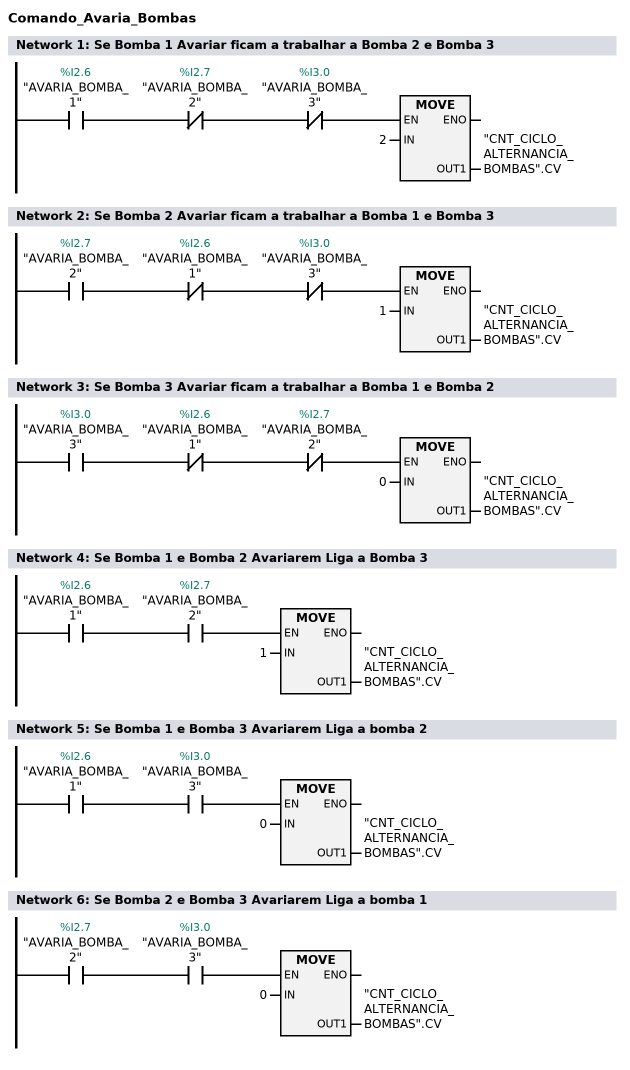
   RUNG wire#powerrail
      Contact( "AVARIA_BOMBA_1" )
      I_Contact( "AVARIA_BOMBA_2" )
      I_Contact( "AVARIA_BOMBA_3" )
      Move(in := 2, out1 => "CNT_CICLO_ALTERNANCIA_BOMBAS".CV)
   END_RUNG
   // the same network as SCL:
   IF "AVARIA_BOMBA_1" AND NOT "AVARIA_BOMBA_2" AND NOT "AVARIA_BOMBA_3" THEN
       "CNT_CICLO_ALTERNANCIA_BOMBAS".CV := 2;
   END_IF;
END_REGION

REGION Network 2: Se Bomba 2 Avariar ficam a trabalhar a Bomba 1 e Bomba 3
   RUNG wire#powerrail
      Contact( "AVARIA_BOMBA_2" )
      I_Contact( "AVARIA_BOMBA_1" )
      I_Contact( "AVARIA_BOMBA_3" )
      Move(in := 1, out1 => "CNT_CICLO_ALTERNANCIA_BOMBAS".CV)
   END_RUNG
   // the same network as SCL:
   IF "AVARIA_BOMBA_2" AND NOT "AVARIA_BOMBA_1" AND NOT "AVARIA_BOMBA_3" THEN
       "CNT_CICLO_ALTERNANCIA_BOMBAS".CV := 1;
   END_IF;
END_REGION

REGION Network 3: Se Bomba 3 Avariar ficam a trabalhar a Bomba 1 e Bomba 2
   RUNG wire#powerrail
      Contact( "AVARIA_BOMBA_3" )
      I_Contact( "AVARIA_BOMBA_1" )
      I_Contact( "AVARIA_BOMBA_2" )
      Move(in := 0, out1 => "CNT_CICLO_ALTERNANCIA_BOMBAS".CV)
   END_RUNG
   // the same network as SCL:
   IF "AVARIA_BOMBA_3" AND NOT "AVARIA_BOMBA_1" AND NOT "AVARIA_BOMBA_2" THEN
       "CNT_CICLO_ALTERNANCIA_BOMBAS".CV := 0;
   END_IF;
END_REGION

REGION Network 4: Se Bomba 1 e Bomba 2 Avariarem Liga a Bomba 3
   RUNG wire#powerrail
      Contact( "AVARIA_BOMBA_1" )
      Contact( "AVARIA_BOMBA_2" )
      Move(in := 1, out1 => "CNT_CICLO_ALTERNANCIA_BOMBAS".CV)
   END_RUNG
   // the same network as SCL:
   IF "AVARIA_BOMBA_1" AND "AVARIA_BOMBA_2" THEN "CNT_CICLO_ALTERNANCIA_BOMBAS".CV := 1; END_IF;
END_REGION

REGION Network 5: Se Bomba 1 e Bomba 3 Avariarem Liga a bomba 2
   RUNG wire#powerrail
      Contact( "AVARIA_BOMBA_1" )
      Contact( "AVARIA_BOMBA_3" )
      Move(in := 0, out1 => "CNT_CICLO_ALTERNANCIA_BOMBAS".CV)
   END_RUNG
   // the same network as SCL:
   IF "AVARIA_BOMBA_1" AND "AVARIA_BOMBA_3" THEN "CNT_CICLO_ALTERNANCIA_BOMBAS".CV := 0; END_IF;
END_REGION

REGION Network 6: Se Bomba 2 e Bomba 3 Avariarem Liga a bomba 1
   RUNG wire#powerrail
      Contact( "AVARIA_BOMBA_2" )
      Contact( "AVARIA_BOMBA_3" )
      Move(in := 0, out1 => "CNT_CICLO_ALTERNANCIA_BOMBAS".CV)
   END_RUNG
   // the same network as SCL:
   IF "AVARIA_BOMBA_2" AND "AVARIA_BOMBA_3" THEN "CNT_CICLO_ALTERNANCIA_BOMBAS".CV := 0; END_IF;
END_REGION
END_FUNCTION

FUNCTION "T_Func_Bombas" : Void   // FC9, LAD
{ S7_Optimized_Access := 'TRUE' }
VERSION : 0.1
// stored: AutoNumber true, IsIECCheckEnabled false, SetENOAutomatically false, UDAEnableTagReadback false
   VAR_TEMP   // added for the SCL form of the ladder/FBD networks
      _w1 : Bool;
   END_VAR
BEGIN

REGION Network 1: Período de tempo de alternancia das bombas
   // Se contador = 0, trabalha B1 e B2. Se = 1, trabalha B1 e B3. Se = 2, trabalha B2 e B3
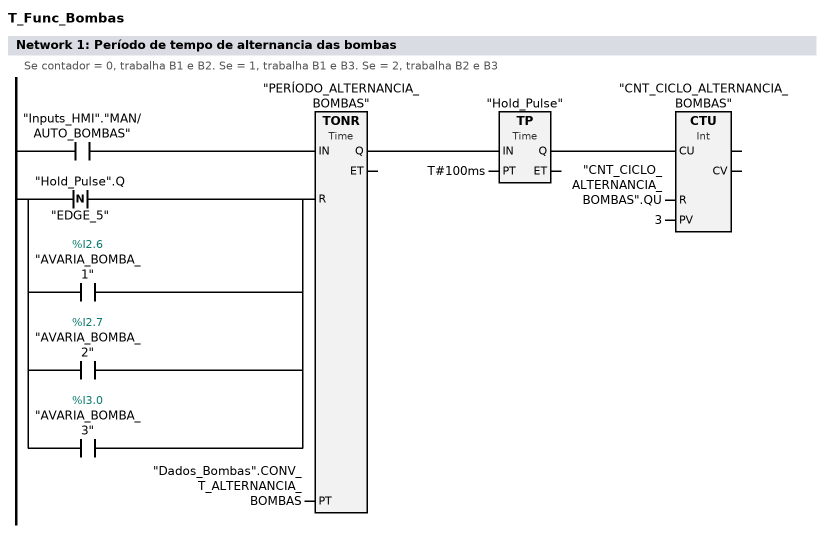
   RUNG wire#powerrail
      Contact( "Inputs_HMI"."MAN/AUTO_BOMBAS" )
      { S7_Templates := "time_type := Time" } "PERÍODO_ALTERNANCIA_BOMBAS".TONR(r := wire#w1, pt := "Dados_Bombas".CONV_T_ALTERNANCIA_BOMBAS, et =>)
      { S7_Templates := "time_type := Time" } "Hold_Pulse".TP(pt := T#100ms, et =>)
      { S7_Templates := "value_type := Int" } "CNT_CICLO_ALTERNANCIA_BOMBAS".CTU(r := "CNT_CICLO_ALTERNANCIA_BOMBAS".QU, pv := 3, cv =>)
   END_RUNG
   RUNG wire#powerrail
      N_Contact(operand := "Hold_Pulse".Q, bit := "EDGE_5")
   END_RUNG wire#w1
   RUNG wire#powerrail
      Contact( "AVARIA_BOMBA_1" )
   END_RUNG wire#w1
   RUNG wire#powerrail
      Contact( "AVARIA_BOMBA_2" )
   END_RUNG wire#w1
   RUNG wire#powerrail
      Contact( "AVARIA_BOMBA_3" )
   END_RUNG wire#w1
   // the same network as SCL:
   #_w1 := NOT "Hold_Pulse".Q AND "EDGE_5";   // falling edge of "Hold_Pulse".Q
   "EDGE_5" := "Hold_Pulse".Q;
   "PERÍODO_ALTERNANCIA_BOMBAS".TONR(IN := "Inputs_HMI"."MAN/AUTO_BOMBAS",
                           R := #_w1 OR "AVARIA_BOMBA_1" OR "AVARIA_BOMBA_2" OR "AVARIA_BOMBA_3",
                           PT := "Dados_Bombas".CONV_T_ALTERNANCIA_BOMBAS);
   "Hold_Pulse".TP(IN := "PERÍODO_ALTERNANCIA_BOMBAS".Q, PT := T#100ms);
   "CNT_CICLO_ALTERNANCIA_BOMBAS".CTU(CU := "Hold_Pulse".Q, R := "CNT_CICLO_ALTERNANCIA_BOMBAS".QU, PV := 3);
END_REGION
END_FUNCTION

FUNCTION "Totalizador_Bombas" : Void   // FC10, LAD
{ S7_Optimized_Access := 'TRUE' }
VERSION : 0.1
// stored: AutoNumber true, IsIECCheckEnabled false, SetENOAutomatically false, UDAEnableTagReadback false
BEGIN

REGION Network 1
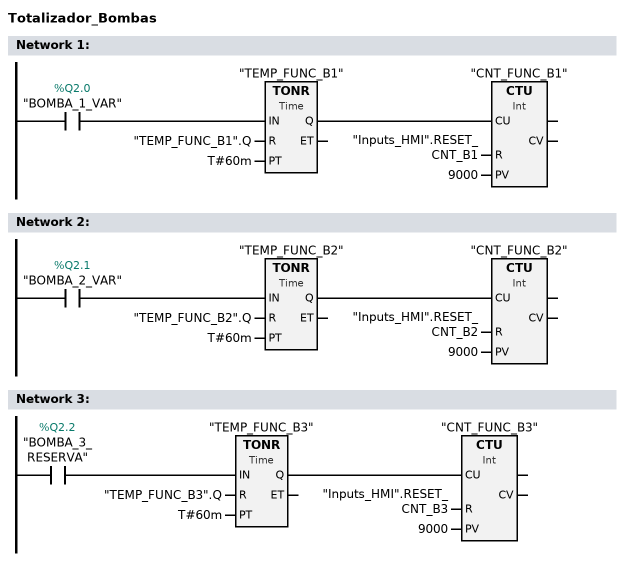
   RUNG wire#powerrail
      Contact( "BOMBA_1_VAR" )
      { S7_Templates := "time_type := Time" } "TEMP_FUNC_B1".TONR(r := "TEMP_FUNC_B1".Q, pt := T#60m, et =>)
      { S7_Templates := "value_type := Int" } "CNT_FUNC_B1".CTU(r := "Inputs_HMI".RESET_CNT_B1, pv := 9000, cv =>)
   END_RUNG
   // the same network as SCL:
   "TEMP_FUNC_B1".TONR(IN := "BOMBA_1_VAR", R := "TEMP_FUNC_B1".Q, PT := T#60m);
   "CNT_FUNC_B1".CTU(CU := "TEMP_FUNC_B1".Q, R := "Inputs_HMI".RESET_CNT_B1, PV := 9000);
END_REGION

REGION Network 2
   RUNG wire#powerrail
      Contact( "BOMBA_2_VAR" )
      { S7_Templates := "time_type := Time" } "TEMP_FUNC_B2".TONR(r := "TEMP_FUNC_B2".Q, pt := T#60m, et =>)
      { S7_Templates := "value_type := Int" } "CNT_FUNC_B2".CTU(r := "Inputs_HMI".RESET_CNT_B2, pv := 9000, cv =>)
   END_RUNG
   // the same network as SCL:
   "TEMP_FUNC_B2".TONR(IN := "BOMBA_2_VAR", R := "TEMP_FUNC_B2".Q, PT := T#60m);
   "CNT_FUNC_B2".CTU(CU := "TEMP_FUNC_B2".Q, R := "Inputs_HMI".RESET_CNT_B2, PV := 9000);
END_REGION

REGION Network 3
   RUNG wire#powerrail
      Contact( "BOMBA_3_RESERVA" )
      { S7_Templates := "time_type := Time" } "TEMP_FUNC_B3".TONR(r := "TEMP_FUNC_B3".Q, pt := T#60m, et =>)
      { S7_Templates := "value_type := Int" } "CNT_FUNC_B3".CTU(r := "Inputs_HMI".RESET_CNT_B3, pv := 9000, cv =>)
   END_RUNG
   // the same network as SCL:
   "TEMP_FUNC_B3".TONR(IN := "BOMBA_3_RESERVA", R := "TEMP_FUNC_B3".Q, PT := T#60m);
   "CNT_FUNC_B3".CTU(CU := "TEMP_FUNC_B3".Q, R := "Inputs_HMI".RESET_CNT_B3, PV := 9000);
END_REGION
END_FUNCTION

FUNCTION "Ciclo_Hórario_Filtros" : Void   // FC16, LAD
{ S7_Optimized_Access := 'TRUE' }
VERSION : 0.1
// stored: AutoNumber true, IsIECCheckEnabled false, SetENOAutomatically false, UDAEnableTagReadback false
   VAR_TEMP   // added for the SCL form of the ladder/FBD networks
      _w1 : Bool;
   END_VAR
BEGIN

REGION Network 1: Leitura de tempo do sistema
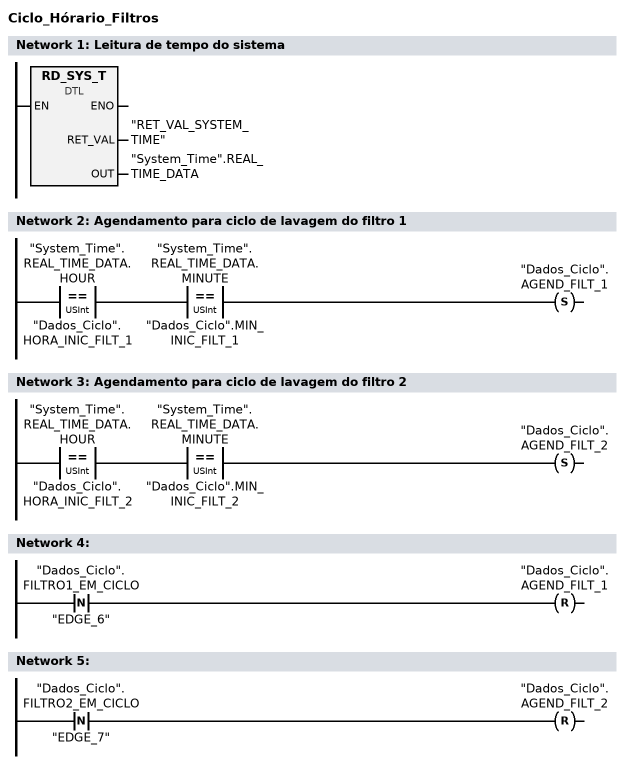
   RUNG wire#powerrail
      { S7_Templates := "date_type := DTL" } RD_SYS_T(RET_VAL => "RET_VAL_SYSTEM_TIME", OUT => "System_Time".REAL_TIME_DATA)
   END_RUNG
   // the same network as SCL:
   "RET_VAL_SYSTEM_TIME" := RD_SYS_T(OUT => "System_Time".REAL_TIME_DATA);
END_REGION

REGION Network 2: Agendamento para ciclo de lavagem do filtro 1
   RUNG wire#powerrail
      { S7_Templates := "SrcType := USInt" } EQ_Contact(in1 := "System_Time".REAL_TIME_DATA.HOUR, in2 := "Dados_Ciclo".HORA_INIC_FILT_1)
      { S7_Templates := "SrcType := USInt" } EQ_Contact(in1 := "System_Time".REAL_TIME_DATA.MINUTE, in2 := "Dados_Ciclo".MIN_INIC_FILT_1)
      S_Coil( "Dados_Ciclo".AGEND_FILT_1 )
   END_RUNG
   // the same network as SCL:
   IF ("System_Time".REAL_TIME_DATA.HOUR = "Dados_Ciclo".HORA_INIC_FILT_1) AND ("System_Time".REAL_TIME_DATA.MINUTE = "Dados_Ciclo".MIN_INIC_FILT_1) THEN
       "Dados_Ciclo".AGEND_FILT_1 := TRUE;
   END_IF;
END_REGION

REGION Network 3: Agendamento para ciclo de lavagem do filtro 2
   RUNG wire#powerrail
      { S7_Templates := "SrcType := USInt" } EQ_Contact(in1 := "System_Time".REAL_TIME_DATA.HOUR, in2 := "Dados_Ciclo".HORA_INIC_FILT_2)
      { S7_Templates := "SrcType := USInt" } EQ_Contact(in1 := "System_Time".REAL_TIME_DATA.MINUTE, in2 := "Dados_Ciclo".MIN_INIC_FILT_2)
      S_Coil( "Dados_Ciclo".AGEND_FILT_2 )
   END_RUNG
   // the same network as SCL:
   IF ("System_Time".REAL_TIME_DATA.HOUR = "Dados_Ciclo".HORA_INIC_FILT_2) AND ("System_Time".REAL_TIME_DATA.MINUTE = "Dados_Ciclo".MIN_INIC_FILT_2) THEN
       "Dados_Ciclo".AGEND_FILT_2 := TRUE;
   END_IF;
END_REGION

REGION Network 4
   RUNG wire#powerrail
      N_Contact(operand := "Dados_Ciclo".FILTRO1_EM_CICLO, bit := "EDGE_6")
      R_Coil( "Dados_Ciclo".AGEND_FILT_1 )
   END_RUNG
   // the same network as SCL:
   #_w1 := NOT "Dados_Ciclo".FILTRO1_EM_CICLO AND "EDGE_6";   // falling edge of "Dados_Ciclo".FILTRO1_EM_CICLO
   "EDGE_6" := "Dados_Ciclo".FILTRO1_EM_CICLO;
   IF #_w1 THEN "Dados_Ciclo".AGEND_FILT_1 := FALSE; END_IF;
END_REGION

REGION Network 5
   RUNG wire#powerrail
      N_Contact(operand := "Dados_Ciclo".FILTRO2_EM_CICLO, bit := "EDGE_7")
      R_Coil( "Dados_Ciclo".AGEND_FILT_2 )
   END_RUNG
   // the same network as SCL:
   #_w1 := NOT "Dados_Ciclo".FILTRO2_EM_CICLO AND "EDGE_7";   // falling edge of "Dados_Ciclo".FILTRO2_EM_CICLO
   "EDGE_7" := "Dados_Ciclo".FILTRO2_EM_CICLO;
   IF #_w1 THEN "Dados_Ciclo".AGEND_FILT_2 := FALSE; END_IF;
END_REGION
END_FUNCTION

FUNCTION "Ciclo_Limpeza" : Void   // FC1, LAD
TITLE = Ciclo de lavagem e enxaguamento
{ S7_Optimized_Access := 'TRUE' }
VERSION : 0.1
// stored: AutoNumber true, IsIECCheckEnabled false, SetENOAutomatically false, UDAEnableTagReadback false
   VAR_TEMP   // added for the SCL form of the ladder/FBD networks
      _w1 : Bool;
      _w2 : Bool;
      _w3 : Bool;
   END_VAR
BEGIN

REGION Network 1: Etapa 1 (Início)
   // Início com EV's na posição de filtração. As bombas podem estar ligadas ou não, conforme a posição do switch 4
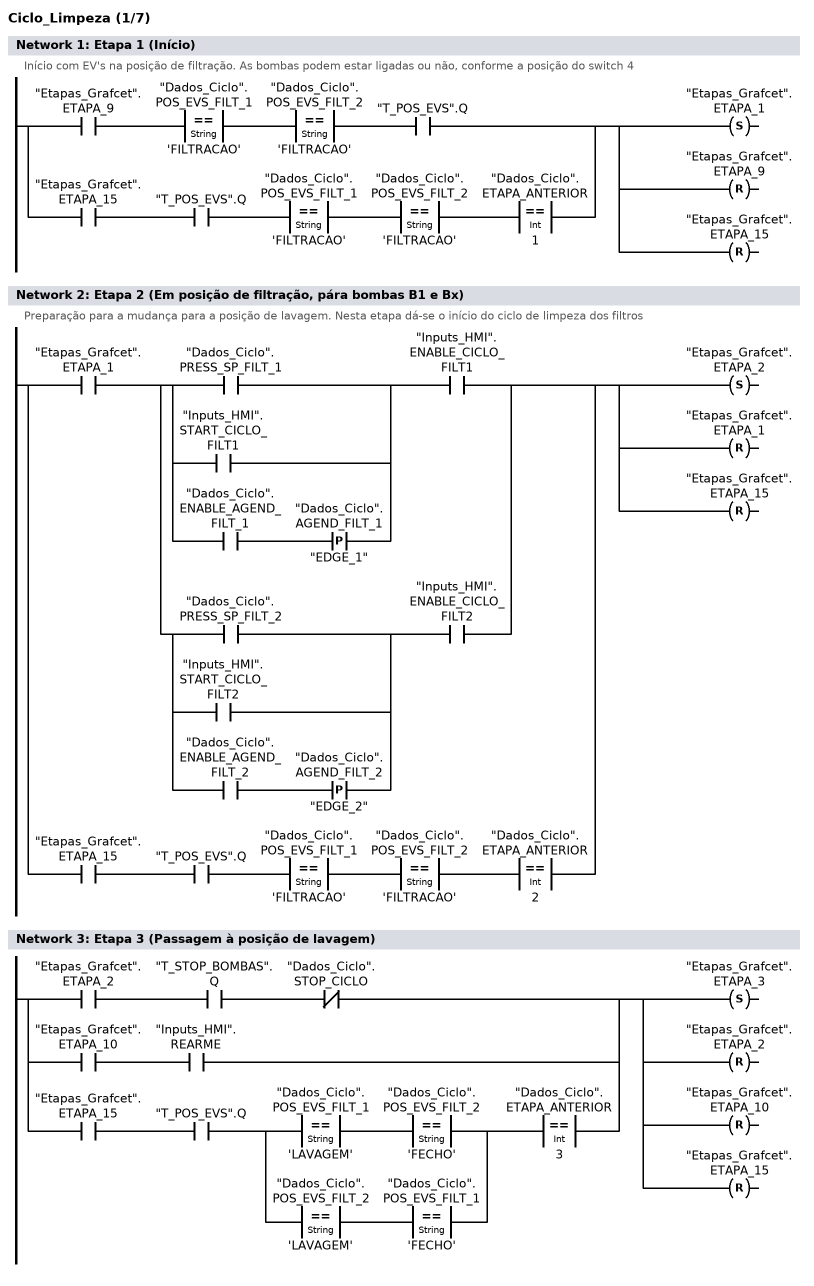
   RUNG wire#powerrail
      Contact( "Etapas_Grafcet".ETAPA_9 )
      { S7_Templates := "SrcType := String" } EQ_Contact(in1 := "Dados_Ciclo".POS_EVS_FILT_1, in2 := 'FILTRACAO')
      { S7_Templates := "SrcType := String" } EQ_Contact(in1 := "Dados_Ciclo".POS_EVS_FILT_2, in2 := 'FILTRACAO')
      Contact( "T_POS_EVS".Q )
      wire#w1
      S_Coil( "Etapas_Grafcet".ETAPA_1 )
   END_RUNG
   RUNG wire#powerrail
      Contact( "Etapas_Grafcet".ETAPA_15 )
      Contact( "T_POS_EVS".Q )
      { S7_Templates := "SrcType := String" } EQ_Contact(in1 := "Dados_Ciclo".POS_EVS_FILT_1, in2 := 'FILTRACAO')
      { S7_Templates := "SrcType := String" } EQ_Contact(in1 := "Dados_Ciclo".POS_EVS_FILT_2, in2 := 'FILTRACAO')
      { S7_Templates := "SrcType := Int" } EQ_Contact(in1 := "Dados_Ciclo".ETAPA_ANTERIOR, in2 := 1)
   END_RUNG wire#w1
   RUNG wire#w1
      R_Coil( "Etapas_Grafcet".ETAPA_9 )
   END_RUNG
   RUNG wire#w1
      R_Coil( "Etapas_Grafcet".ETAPA_15 )
   END_RUNG
   // the same network as SCL:
   IF ("Etapas_Grafcet".ETAPA_9 AND ("Dados_Ciclo".POS_EVS_FILT_1 = 'FILTRACAO') AND ("Dados_Ciclo".POS_EVS_FILT_2 = 'FILTRACAO') AND "T_POS_EVS".Q) OR ("Etapas_Grafcet".ETAPA_15 AND "T_POS_EVS".Q AND ("Dados_Ciclo".POS_EVS_FILT_1 = 'FILTRACAO') AND ("Dados_Ciclo".POS_EVS_FILT_2 = 'FILTRACAO') AND ("Dados_Ciclo".ETAPA_ANTERIOR = 1)) THEN
       "Etapas_Grafcet".ETAPA_1 := TRUE;
   END_IF;
   #_w1 := ("Etapas_Grafcet".ETAPA_9 AND ("Dados_Ciclo".POS_EVS_FILT_1 = 'FILTRACAO') AND ("Dados_Ciclo".POS_EVS_FILT_2 = 'FILTRACAO') AND "T_POS_EVS".Q) OR ("Etapas_Grafcet".ETAPA_15 AND "T_POS_EVS".Q AND ("Dados_Ciclo".POS_EVS_FILT_1 = 'FILTRACAO') AND ("Dados_Ciclo".POS_EVS_FILT_2 = 'FILTRACAO') AND ("Dados_Ciclo".ETAPA_ANTERIOR = 1));
   IF #_w1 THEN
       "Etapas_Grafcet".ETAPA_9 := FALSE;
       "Etapas_Grafcet".ETAPA_15 := FALSE;
   END_IF;
END_REGION

REGION Network 2: Etapa 2 (Em posição de filtração, pára bombas B1 e Bx)
   // Preparação para a mudança para a posição de lavagem. Nesta etapa dá-se o início do ciclo de limpeza dos filtros
   RUNG wire#powerrail
      Contact( "Etapas_Grafcet".ETAPA_1 )
      wire#w1
      Contact( "Dados_Ciclo".PRESS_SP_FILT_1 )
      wire#w2
      Contact( "Inputs_HMI".ENABLE_CICLO_FILT1 )
      wire#w3
      S_Coil( "Etapas_Grafcet".ETAPA_2 )
   END_RUNG
   RUNG wire#w1
      Contact( "Inputs_HMI".START_CICLO_FILT1 )
   END_RUNG wire#w2
   RUNG wire#w1
      Contact( "Dados_Ciclo".ENABLE_AGEND_FILT_1 )
      P_Contact(operand := "Dados_Ciclo".AGEND_FILT_1, bit := "EDGE_1")
   END_RUNG wire#w2
   RUNG wire#w1
      Contact( "Dados_Ciclo".PRESS_SP_FILT_2 )
      wire#w4
      Contact( "Inputs_HMI".ENABLE_CICLO_FILT2 )
   END_RUNG wire#w3
   RUNG wire#w1
      Contact( "Inputs_HMI".START_CICLO_FILT2 )
   END_RUNG wire#w4
   RUNG wire#w1
      Contact( "Dados_Ciclo".ENABLE_AGEND_FILT_2 )
      P_Contact(operand := "Dados_Ciclo".AGEND_FILT_2, bit := "EDGE_2")
   END_RUNG wire#w4
   RUNG wire#powerrail
      Contact( "Etapas_Grafcet".ETAPA_15 )
      Contact( "T_POS_EVS".Q )
      { S7_Templates := "SrcType := String" } EQ_Contact(in1 := "Dados_Ciclo".POS_EVS_FILT_1, in2 := 'FILTRACAO')
      { S7_Templates := "SrcType := String" } EQ_Contact(in1 := "Dados_Ciclo".POS_EVS_FILT_2, in2 := 'FILTRACAO')
      { S7_Templates := "SrcType := Int" } EQ_Contact(in1 := "Dados_Ciclo".ETAPA_ANTERIOR, in2 := 2)
   END_RUNG wire#w3
   RUNG wire#w3
      R_Coil( "Etapas_Grafcet".ETAPA_1 )
   END_RUNG
   RUNG wire#w3
      R_Coil( "Etapas_Grafcet".ETAPA_15 )
   END_RUNG
   // the same network as SCL:
   #_w1 := "Etapas_Grafcet".ETAPA_1 AND "Dados_Ciclo".ENABLE_AGEND_FILT_1 AND "Dados_Ciclo".AGEND_FILT_1 AND NOT "EDGE_1";   // rising edge of "Dados_Ciclo".AGEND_FILT_1
   "EDGE_1" := "Dados_Ciclo".AGEND_FILT_1;
   #_w2 := "Etapas_Grafcet".ETAPA_1 AND "Dados_Ciclo".ENABLE_AGEND_FILT_2 AND "Dados_Ciclo".AGEND_FILT_2 AND NOT "EDGE_2";   // rising edge of "Dados_Ciclo".AGEND_FILT_2
   "EDGE_2" := "Dados_Ciclo".AGEND_FILT_2;
   IF ((("Etapas_Grafcet".ETAPA_1 AND ("Dados_Ciclo".PRESS_SP_FILT_1 OR "Inputs_HMI".START_CICLO_FILT1)) OR #_w1) AND "Inputs_HMI".ENABLE_CICLO_FILT1) OR ((("Etapas_Grafcet".ETAPA_1 AND ("Dados_Ciclo".PRESS_SP_FILT_2 OR "Inputs_HMI".START_CICLO_FILT2)) OR #_w2) AND "Inputs_HMI".ENABLE_CICLO_FILT2) OR ("Etapas_Grafcet".ETAPA_15 AND "T_POS_EVS".Q AND ("Dados_Ciclo".POS_EVS_FILT_1 = 'FILTRACAO') AND ("Dados_Ciclo".POS_EVS_FILT_2 = 'FILTRACAO') AND ("Dados_Ciclo".ETAPA_ANTERIOR = 2)) THEN
       "Etapas_Grafcet".ETAPA_2 := TRUE;
   END_IF;
   #_w3 := ((("Etapas_Grafcet".ETAPA_1 AND ("Dados_Ciclo".PRESS_SP_FILT_1 OR "Inputs_HMI".START_CICLO_FILT1)) OR #_w1) AND "Inputs_HMI".ENABLE_CICLO_FILT1) OR ((("Etapas_Grafcet".ETAPA_1 AND ("Dados_Ciclo".PRESS_SP_FILT_2 OR "Inputs_HMI".START_CICLO_FILT2)) OR #_w2) AND "Inputs_HMI".ENABLE_CICLO_FILT2) OR ("Etapas_Grafcet".ETAPA_15 AND "T_POS_EVS".Q AND ("Dados_Ciclo".POS_EVS_FILT_1 = 'FILTRACAO') AND ("Dados_Ciclo".POS_EVS_FILT_2 = 'FILTRACAO') AND ("Dados_Ciclo".ETAPA_ANTERIOR = 2));
   IF #_w3 THEN
       "Etapas_Grafcet".ETAPA_1 := FALSE;
       "Etapas_Grafcet".ETAPA_15 := FALSE;
   END_IF;
END_REGION

REGION Network 3: Etapa 3 (Passagem à posição de lavagem)
   RUNG wire#powerrail
      Contact( "Etapas_Grafcet".ETAPA_2 )
      Contact( "T_STOP_BOMBAS".Q )
      I_Contact( "Dados_Ciclo".STOP_CICLO )
      wire#w1
      S_Coil( "Etapas_Grafcet".ETAPA_3 )
   END_RUNG
   RUNG wire#powerrail
      Contact( "Etapas_Grafcet".ETAPA_10 )
      Contact( "Inputs_HMI".REARME )
   END_RUNG wire#w1
   RUNG wire#powerrail
      Contact( "Etapas_Grafcet".ETAPA_15 )
      Contact( "T_POS_EVS".Q )
      wire#w2
      { S7_Templates := "SrcType := String" } EQ_Contact(in1 := "Dados_Ciclo".POS_EVS_FILT_1, in2 := 'LAVAGEM')
      { S7_Templates := "SrcType := String" } EQ_Contact(in1 := "Dados_Ciclo".POS_EVS_FILT_2, in2 := 'FECHO')
      wire#w3
      { S7_Templates := "SrcType := Int" } EQ_Contact(in1 := "Dados_Ciclo".ETAPA_ANTERIOR, in2 := 3)
   END_RUNG wire#w1
   RUNG wire#w2
      { S7_Templates := "SrcType := String" } EQ_Contact(in1 := "Dados_Ciclo".POS_EVS_FILT_2, in2 := 'LAVAGEM')
      { S7_Templates := "SrcType := String" } EQ_Contact(in1 := "Dados_Ciclo".POS_EVS_FILT_1, in2 := 'FECHO')
   END_RUNG wire#w3
   RUNG wire#w1
      R_Coil( "Etapas_Grafcet".ETAPA_2 )
   END_RUNG
   RUNG wire#w1
      R_Coil( "Etapas_Grafcet".ETAPA_10 )
   END_RUNG
   RUNG wire#w1
      R_Coil( "Etapas_Grafcet".ETAPA_15 )
   END_RUNG
   // the same network as SCL:
   IF ("Etapas_Grafcet".ETAPA_2 AND "T_STOP_BOMBAS".Q AND NOT "Dados_Ciclo".STOP_CICLO) OR ("Etapas_Grafcet".ETAPA_10 AND "Inputs_HMI".REARME) OR ("Etapas_Grafcet".ETAPA_15 AND "T_POS_EVS".Q AND ((("Dados_Ciclo".POS_EVS_FILT_1 = 'LAVAGEM') AND ("Dados_Ciclo".POS_EVS_FILT_2 = 'FECHO')) OR (("Dados_Ciclo".POS_EVS_FILT_2 = 'LAVAGEM') AND ("Dados_Ciclo".POS_EVS_FILT_1 = 'FECHO'))) AND ("Dados_Ciclo".ETAPA_ANTERIOR = 3)) THEN
       "Etapas_Grafcet".ETAPA_3 := TRUE;
   END_IF;
   #_w1 := ("Etapas_Grafcet".ETAPA_2 AND "T_STOP_BOMBAS".Q AND NOT "Dados_Ciclo".STOP_CICLO) OR ("Etapas_Grafcet".ETAPA_10 AND "Inputs_HMI".REARME) OR ("Etapas_Grafcet".ETAPA_15 AND "T_POS_EVS".Q AND ((("Dados_Ciclo".POS_EVS_FILT_1 = 'LAVAGEM') AND ("Dados_Ciclo".POS_EVS_FILT_2 = 'FECHO')) OR (("Dados_Ciclo".POS_EVS_FILT_2 = 'LAVAGEM') AND ("Dados_Ciclo".POS_EVS_FILT_1 = 'FECHO'))) AND ("Dados_Ciclo".ETAPA_ANTERIOR = 3));
   IF #_w1 THEN
       "Etapas_Grafcet".ETAPA_2 := FALSE;
       "Etapas_Grafcet".ETAPA_10 := FALSE;
       "Etapas_Grafcet".ETAPA_15 := FALSE;
   END_IF;
END_REGION

REGION Network 4: Etapa 4 (Em lavagem, B1 e BX ligadas)
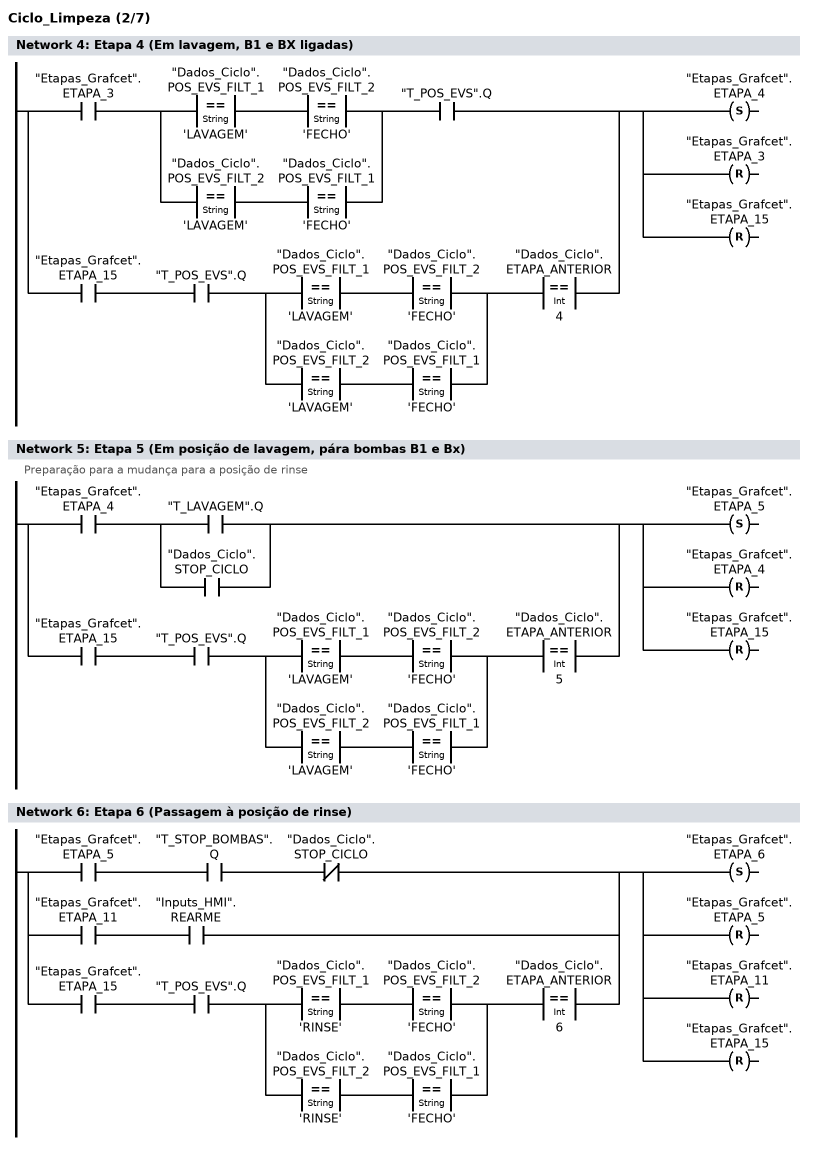
   RUNG wire#powerrail
      Contact( "Etapas_Grafcet".ETAPA_3 )
      wire#w1
      { S7_Templates := "SrcType := String" } EQ_Contact(in1 := "Dados_Ciclo".POS_EVS_FILT_1, in2 := 'LAVAGEM')
      { S7_Templates := "SrcType := String" } EQ_Contact(in1 := "Dados_Ciclo".POS_EVS_FILT_2, in2 := 'FECHO')
      wire#w2
      Contact( "T_POS_EVS".Q )
      wire#w3
      S_Coil( "Etapas_Grafcet".ETAPA_4 )
   END_RUNG
   RUNG wire#w1
      { S7_Templates := "SrcType := String" } EQ_Contact(in1 := "Dados_Ciclo".POS_EVS_FILT_2, in2 := 'LAVAGEM')
      { S7_Templates := "SrcType := String" } EQ_Contact(in1 := "Dados_Ciclo".POS_EVS_FILT_1, in2 := 'FECHO')
   END_RUNG wire#w2
   RUNG wire#powerrail
      Contact( "Etapas_Grafcet".ETAPA_15 )
      Contact( "T_POS_EVS".Q )
      wire#w4
      { S7_Templates := "SrcType := String" } EQ_Contact(in1 := "Dados_Ciclo".POS_EVS_FILT_1, in2 := 'LAVAGEM')
      { S7_Templates := "SrcType := String" } EQ_Contact(in1 := "Dados_Ciclo".POS_EVS_FILT_2, in2 := 'FECHO')
      wire#w5
      { S7_Templates := "SrcType := Int" } EQ_Contact(in1 := "Dados_Ciclo".ETAPA_ANTERIOR, in2 := 4)
   END_RUNG wire#w3
   RUNG wire#w4
      { S7_Templates := "SrcType := String" } EQ_Contact(in1 := "Dados_Ciclo".POS_EVS_FILT_2, in2 := 'LAVAGEM')
      { S7_Templates := "SrcType := String" } EQ_Contact(in1 := "Dados_Ciclo".POS_EVS_FILT_1, in2 := 'FECHO')
   END_RUNG wire#w5
   RUNG wire#w3
      R_Coil( "Etapas_Grafcet".ETAPA_3 )
   END_RUNG
   RUNG wire#w3
      R_Coil( "Etapas_Grafcet".ETAPA_15 )
   END_RUNG
   // the same network as SCL:
   IF ("Etapas_Grafcet".ETAPA_3 AND ((("Dados_Ciclo".POS_EVS_FILT_1 = 'LAVAGEM') AND ("Dados_Ciclo".POS_EVS_FILT_2 = 'FECHO')) OR (("Dados_Ciclo".POS_EVS_FILT_2 = 'LAVAGEM') AND ("Dados_Ciclo".POS_EVS_FILT_1 = 'FECHO'))) AND "T_POS_EVS".Q) OR ("Etapas_Grafcet".ETAPA_15 AND "T_POS_EVS".Q AND ((("Dados_Ciclo".POS_EVS_FILT_1 = 'LAVAGEM') AND ("Dados_Ciclo".POS_EVS_FILT_2 = 'FECHO')) OR (("Dados_Ciclo".POS_EVS_FILT_2 = 'LAVAGEM') AND ("Dados_Ciclo".POS_EVS_FILT_1 = 'FECHO'))) AND ("Dados_Ciclo".ETAPA_ANTERIOR = 4)) THEN
       "Etapas_Grafcet".ETAPA_4 := TRUE;
   END_IF;
   #_w1 := ("Etapas_Grafcet".ETAPA_3 AND ((("Dados_Ciclo".POS_EVS_FILT_1 = 'LAVAGEM') AND ("Dados_Ciclo".POS_EVS_FILT_2 = 'FECHO')) OR (("Dados_Ciclo".POS_EVS_FILT_2 = 'LAVAGEM') AND ("Dados_Ciclo".POS_EVS_FILT_1 = 'FECHO'))) AND "T_POS_EVS".Q) OR ("Etapas_Grafcet".ETAPA_15 AND "T_POS_EVS".Q AND ((("Dados_Ciclo".POS_EVS_FILT_1 = 'LAVAGEM') AND ("Dados_Ciclo".POS_EVS_FILT_2 = 'FECHO')) OR (("Dados_Ciclo".POS_EVS_FILT_2 = 'LAVAGEM') AND ("Dados_Ciclo".POS_EVS_FILT_1 = 'FECHO'))) AND ("Dados_Ciclo".ETAPA_ANTERIOR = 4));
   IF #_w1 THEN
       "Etapas_Grafcet".ETAPA_3 := FALSE;
       "Etapas_Grafcet".ETAPA_15 := FALSE;
   END_IF;
END_REGION

REGION Network 5: Etapa 5 (Em posição de lavagem, pára bombas B1 e Bx)
   // Preparação para a mudança para a posição de rinse
   RUNG wire#powerrail
      Contact( "Etapas_Grafcet".ETAPA_4 )
      wire#w1
      Contact( "T_LAVAGEM".Q )
      wire#w2
      S_Coil( "Etapas_Grafcet".ETAPA_5 )
   END_RUNG
   RUNG wire#w1
      Contact( "Dados_Ciclo".STOP_CICLO )
   END_RUNG wire#w2
   RUNG wire#powerrail
      Contact( "Etapas_Grafcet".ETAPA_15 )
      Contact( "T_POS_EVS".Q )
      wire#w3
      { S7_Templates := "SrcType := String" } EQ_Contact(in1 := "Dados_Ciclo".POS_EVS_FILT_1, in2 := 'LAVAGEM')
      { S7_Templates := "SrcType := String" } EQ_Contact(in1 := "Dados_Ciclo".POS_EVS_FILT_2, in2 := 'FECHO')
      wire#w4
      { S7_Templates := "SrcType := Int" } EQ_Contact(in1 := "Dados_Ciclo".ETAPA_ANTERIOR, in2 := 5)
   END_RUNG wire#w2
   RUNG wire#w3
      { S7_Templates := "SrcType := String" } EQ_Contact(in1 := "Dados_Ciclo".POS_EVS_FILT_2, in2 := 'LAVAGEM')
      { S7_Templates := "SrcType := String" } EQ_Contact(in1 := "Dados_Ciclo".POS_EVS_FILT_1, in2 := 'FECHO')
   END_RUNG wire#w4
   RUNG wire#w2
      R_Coil( "Etapas_Grafcet".ETAPA_4 )
   END_RUNG
   RUNG wire#w2
      R_Coil( "Etapas_Grafcet".ETAPA_15 )
   END_RUNG
   // the same network as SCL:
   IF ("Etapas_Grafcet".ETAPA_4 AND ("T_LAVAGEM".Q OR "Dados_Ciclo".STOP_CICLO)) OR ("Etapas_Grafcet".ETAPA_15 AND "T_POS_EVS".Q AND ((("Dados_Ciclo".POS_EVS_FILT_1 = 'LAVAGEM') AND ("Dados_Ciclo".POS_EVS_FILT_2 = 'FECHO')) OR (("Dados_Ciclo".POS_EVS_FILT_2 = 'LAVAGEM') AND ("Dados_Ciclo".POS_EVS_FILT_1 = 'FECHO'))) AND ("Dados_Ciclo".ETAPA_ANTERIOR = 5)) THEN
       "Etapas_Grafcet".ETAPA_5 := TRUE;
   END_IF;
   #_w1 := ("Etapas_Grafcet".ETAPA_4 AND ("T_LAVAGEM".Q OR "Dados_Ciclo".STOP_CICLO)) OR ("Etapas_Grafcet".ETAPA_15 AND "T_POS_EVS".Q AND ((("Dados_Ciclo".POS_EVS_FILT_1 = 'LAVAGEM') AND ("Dados_Ciclo".POS_EVS_FILT_2 = 'FECHO')) OR (("Dados_Ciclo".POS_EVS_FILT_2 = 'LAVAGEM') AND ("Dados_Ciclo".POS_EVS_FILT_1 = 'FECHO'))) AND ("Dados_Ciclo".ETAPA_ANTERIOR = 5));
   IF #_w1 THEN
       "Etapas_Grafcet".ETAPA_4 := FALSE;
       "Etapas_Grafcet".ETAPA_15 := FALSE;
   END_IF;
END_REGION

REGION Network 6: Etapa 6 (Passagem à posição de rinse)
   RUNG wire#powerrail
      Contact( "Etapas_Grafcet".ETAPA_5 )
      Contact( "T_STOP_BOMBAS".Q )
      I_Contact( "Dados_Ciclo".STOP_CICLO )
      wire#w1
      S_Coil( "Etapas_Grafcet".ETAPA_6 )
   END_RUNG
   RUNG wire#powerrail
      Contact( "Etapas_Grafcet".ETAPA_11 )
      Contact( "Inputs_HMI".REARME )
   END_RUNG wire#w1
   RUNG wire#powerrail
      Contact( "Etapas_Grafcet".ETAPA_15 )
      Contact( "T_POS_EVS".Q )
      wire#w2
      { S7_Templates := "SrcType := String" } EQ_Contact(in1 := "Dados_Ciclo".POS_EVS_FILT_1, in2 := 'RINSE')
      { S7_Templates := "SrcType := String" } EQ_Contact(in1 := "Dados_Ciclo".POS_EVS_FILT_2, in2 := 'FECHO')
      wire#w3
      { S7_Templates := "SrcType := Int" } EQ_Contact(in1 := "Dados_Ciclo".ETAPA_ANTERIOR, in2 := 6)
   END_RUNG wire#w1
   RUNG wire#w2
      { S7_Templates := "SrcType := String" } EQ_Contact(in1 := "Dados_Ciclo".POS_EVS_FILT_2, in2 := 'RINSE')
      { S7_Templates := "SrcType := String" } EQ_Contact(in1 := "Dados_Ciclo".POS_EVS_FILT_1, in2 := 'FECHO')
   END_RUNG wire#w3
   RUNG wire#w1
      R_Coil( "Etapas_Grafcet".ETAPA_5 )
   END_RUNG
   RUNG wire#w1
      R_Coil( "Etapas_Grafcet".ETAPA_11 )
   END_RUNG
   RUNG wire#w1
      R_Coil( "Etapas_Grafcet".ETAPA_15 )
   END_RUNG
   // the same network as SCL:
   IF ("Etapas_Grafcet".ETAPA_5 AND "T_STOP_BOMBAS".Q AND NOT "Dados_Ciclo".STOP_CICLO) OR ("Etapas_Grafcet".ETAPA_11 AND "Inputs_HMI".REARME) OR ("Etapas_Grafcet".ETAPA_15 AND "T_POS_EVS".Q AND ((("Dados_Ciclo".POS_EVS_FILT_1 = 'RINSE') AND ("Dados_Ciclo".POS_EVS_FILT_2 = 'FECHO')) OR (("Dados_Ciclo".POS_EVS_FILT_2 = 'RINSE') AND ("Dados_Ciclo".POS_EVS_FILT_1 = 'FECHO'))) AND ("Dados_Ciclo".ETAPA_ANTERIOR = 6)) THEN
       "Etapas_Grafcet".ETAPA_6 := TRUE;
   END_IF;
   #_w1 := ("Etapas_Grafcet".ETAPA_5 AND "T_STOP_BOMBAS".Q AND NOT "Dados_Ciclo".STOP_CICLO) OR ("Etapas_Grafcet".ETAPA_11 AND "Inputs_HMI".REARME) OR ("Etapas_Grafcet".ETAPA_15 AND "T_POS_EVS".Q AND ((("Dados_Ciclo".POS_EVS_FILT_1 = 'RINSE') AND ("Dados_Ciclo".POS_EVS_FILT_2 = 'FECHO')) OR (("Dados_Ciclo".POS_EVS_FILT_2 = 'RINSE') AND ("Dados_Ciclo".POS_EVS_FILT_1 = 'FECHO'))) AND ("Dados_Ciclo".ETAPA_ANTERIOR = 6));
   IF #_w1 THEN
       "Etapas_Grafcet".ETAPA_5 := FALSE;
       "Etapas_Grafcet".ETAPA_11 := FALSE;
       "Etapas_Grafcet".ETAPA_15 := FALSE;
   END_IF;
END_REGION

REGION Network 7: Etapa 7 (Em rinse, B1 ligada)
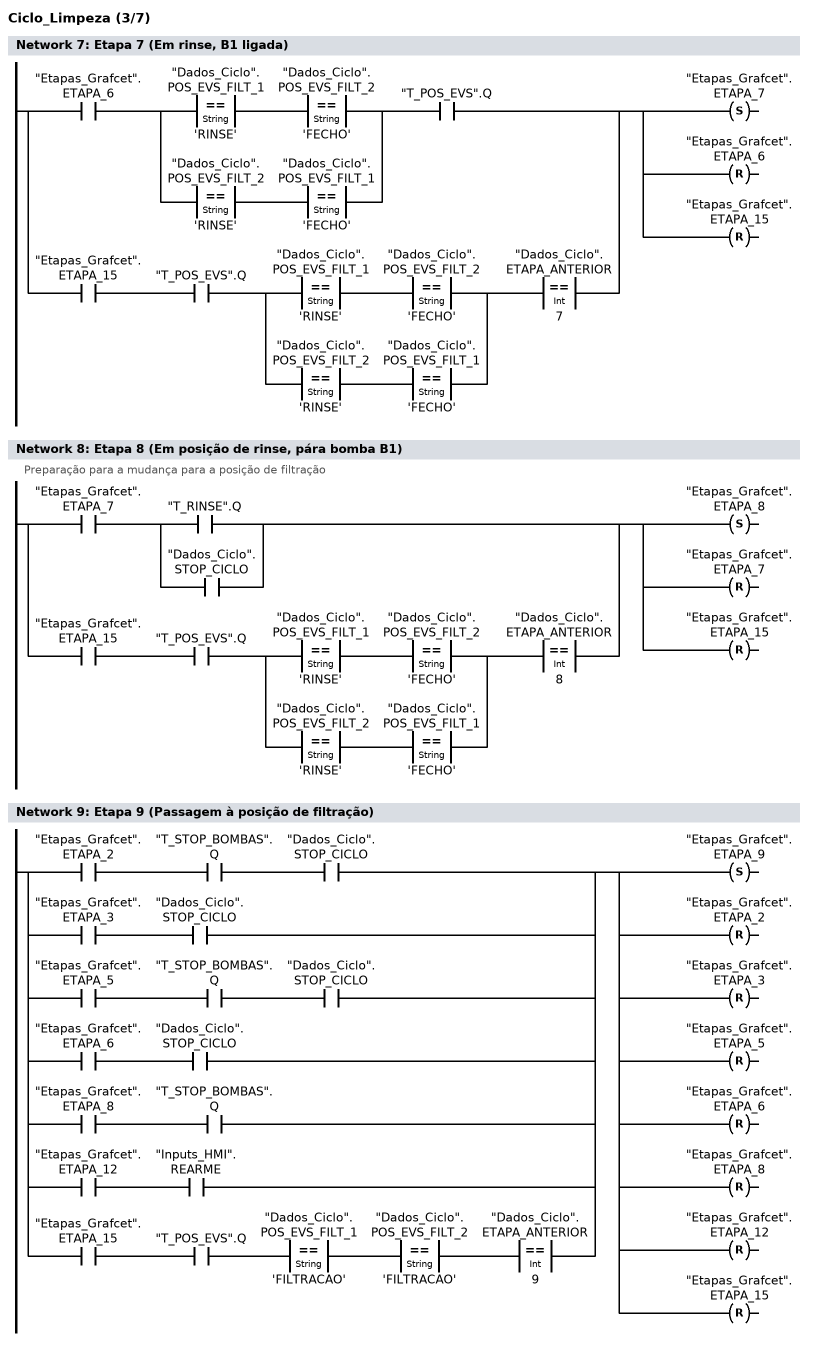
   RUNG wire#powerrail
      Contact( "Etapas_Grafcet".ETAPA_6 )
      wire#w1
      { S7_Templates := "SrcType := String" } EQ_Contact(in1 := "Dados_Ciclo".POS_EVS_FILT_1, in2 := 'RINSE')
      { S7_Templates := "SrcType := String" } EQ_Contact(in1 := "Dados_Ciclo".POS_EVS_FILT_2, in2 := 'FECHO')
      wire#w2
      Contact( "T_POS_EVS".Q )
      wire#w3
      S_Coil( "Etapas_Grafcet".ETAPA_7 )
   END_RUNG
   RUNG wire#w1
      { S7_Templates := "SrcType := String" } EQ_Contact(in1 := "Dados_Ciclo".POS_EVS_FILT_2, in2 := 'RINSE')
      { S7_Templates := "SrcType := String" } EQ_Contact(in1 := "Dados_Ciclo".POS_EVS_FILT_1, in2 := 'FECHO')
   END_RUNG wire#w2
   RUNG wire#powerrail
      Contact( "Etapas_Grafcet".ETAPA_15 )
      Contact( "T_POS_EVS".Q )
      wire#w4
      { S7_Templates := "SrcType := String" } EQ_Contact(in1 := "Dados_Ciclo".POS_EVS_FILT_1, in2 := 'RINSE')
      { S7_Templates := "SrcType := String" } EQ_Contact(in1 := "Dados_Ciclo".POS_EVS_FILT_2, in2 := 'FECHO')
      wire#w5
      { S7_Templates := "SrcType := Int" } EQ_Contact(in1 := "Dados_Ciclo".ETAPA_ANTERIOR, in2 := 7)
   END_RUNG wire#w3
   RUNG wire#w4
      { S7_Templates := "SrcType := String" } EQ_Contact(in1 := "Dados_Ciclo".POS_EVS_FILT_2, in2 := 'RINSE')
      { S7_Templates := "SrcType := String" } EQ_Contact(in1 := "Dados_Ciclo".POS_EVS_FILT_1, in2 := 'FECHO')
   END_RUNG wire#w5
   RUNG wire#w3
      R_Coil( "Etapas_Grafcet".ETAPA_6 )
   END_RUNG
   RUNG wire#w3
      R_Coil( "Etapas_Grafcet".ETAPA_15 )
   END_RUNG
   // the same network as SCL:
   IF ("Etapas_Grafcet".ETAPA_6 AND ((("Dados_Ciclo".POS_EVS_FILT_1 = 'RINSE') AND ("Dados_Ciclo".POS_EVS_FILT_2 = 'FECHO')) OR (("Dados_Ciclo".POS_EVS_FILT_2 = 'RINSE') AND ("Dados_Ciclo".POS_EVS_FILT_1 = 'FECHO'))) AND "T_POS_EVS".Q) OR ("Etapas_Grafcet".ETAPA_15 AND "T_POS_EVS".Q AND ((("Dados_Ciclo".POS_EVS_FILT_1 = 'RINSE') AND ("Dados_Ciclo".POS_EVS_FILT_2 = 'FECHO')) OR (("Dados_Ciclo".POS_EVS_FILT_2 = 'RINSE') AND ("Dados_Ciclo".POS_EVS_FILT_1 = 'FECHO'))) AND ("Dados_Ciclo".ETAPA_ANTERIOR = 7)) THEN
       "Etapas_Grafcet".ETAPA_7 := TRUE;
   END_IF;
   #_w1 := ("Etapas_Grafcet".ETAPA_6 AND ((("Dados_Ciclo".POS_EVS_FILT_1 = 'RINSE') AND ("Dados_Ciclo".POS_EVS_FILT_2 = 'FECHO')) OR (("Dados_Ciclo".POS_EVS_FILT_2 = 'RINSE') AND ("Dados_Ciclo".POS_EVS_FILT_1 = 'FECHO'))) AND "T_POS_EVS".Q) OR ("Etapas_Grafcet".ETAPA_15 AND "T_POS_EVS".Q AND ((("Dados_Ciclo".POS_EVS_FILT_1 = 'RINSE') AND ("Dados_Ciclo".POS_EVS_FILT_2 = 'FECHO')) OR (("Dados_Ciclo".POS_EVS_FILT_2 = 'RINSE') AND ("Dados_Ciclo".POS_EVS_FILT_1 = 'FECHO'))) AND ("Dados_Ciclo".ETAPA_ANTERIOR = 7));
   IF #_w1 THEN
       "Etapas_Grafcet".ETAPA_6 := FALSE;
       "Etapas_Grafcet".ETAPA_15 := FALSE;
   END_IF;
END_REGION

REGION Network 8: Etapa 8 (Em posição de rinse, pára bomba B1)
   // Preparação para a mudança para a posição de filtração
   RUNG wire#powerrail
      Contact( "Etapas_Grafcet".ETAPA_7 )
      wire#w1
      Contact( "T_RINSE".Q )
      wire#w2
      S_Coil( "Etapas_Grafcet".ETAPA_8 )
   END_RUNG
   RUNG wire#w1
      Contact( "Dados_Ciclo".STOP_CICLO )
   END_RUNG wire#w2
   RUNG wire#powerrail
      Contact( "Etapas_Grafcet".ETAPA_15 )
      Contact( "T_POS_EVS".Q )
      wire#w3
      { S7_Templates := "SrcType := String" } EQ_Contact(in1 := "Dados_Ciclo".POS_EVS_FILT_1, in2 := 'RINSE')
      { S7_Templates := "SrcType := String" } EQ_Contact(in1 := "Dados_Ciclo".POS_EVS_FILT_2, in2 := 'FECHO')
      wire#w4
      { S7_Templates := "SrcType := Int" } EQ_Contact(in1 := "Dados_Ciclo".ETAPA_ANTERIOR, in2 := 8)
   END_RUNG wire#w2
   RUNG wire#w3
      { S7_Templates := "SrcType := String" } EQ_Contact(in1 := "Dados_Ciclo".POS_EVS_FILT_2, in2 := 'RINSE')
      { S7_Templates := "SrcType := String" } EQ_Contact(in1 := "Dados_Ciclo".POS_EVS_FILT_1, in2 := 'FECHO')
   END_RUNG wire#w4
   RUNG wire#w2
      R_Coil( "Etapas_Grafcet".ETAPA_7 )
   END_RUNG
   RUNG wire#w2
      R_Coil( "Etapas_Grafcet".ETAPA_15 )
   END_RUNG
   // the same network as SCL:
   IF ("Etapas_Grafcet".ETAPA_7 AND ("T_RINSE".Q OR "Dados_Ciclo".STOP_CICLO)) OR ("Etapas_Grafcet".ETAPA_15 AND "T_POS_EVS".Q AND ((("Dados_Ciclo".POS_EVS_FILT_1 = 'RINSE') AND ("Dados_Ciclo".POS_EVS_FILT_2 = 'FECHO')) OR (("Dados_Ciclo".POS_EVS_FILT_2 = 'RINSE') AND ("Dados_Ciclo".POS_EVS_FILT_1 = 'FECHO'))) AND ("Dados_Ciclo".ETAPA_ANTERIOR = 8)) THEN
       "Etapas_Grafcet".ETAPA_8 := TRUE;
   END_IF;
   #_w1 := ("Etapas_Grafcet".ETAPA_7 AND ("T_RINSE".Q OR "Dados_Ciclo".STOP_CICLO)) OR ("Etapas_Grafcet".ETAPA_15 AND "T_POS_EVS".Q AND ((("Dados_Ciclo".POS_EVS_FILT_1 = 'RINSE') AND ("Dados_Ciclo".POS_EVS_FILT_2 = 'FECHO')) OR (("Dados_Ciclo".POS_EVS_FILT_2 = 'RINSE') AND ("Dados_Ciclo".POS_EVS_FILT_1 = 'FECHO'))) AND ("Dados_Ciclo".ETAPA_ANTERIOR = 8));
   IF #_w1 THEN
       "Etapas_Grafcet".ETAPA_7 := FALSE;
       "Etapas_Grafcet".ETAPA_15 := FALSE;
   END_IF;
END_REGION

REGION Network 9: Etapa 9 (Passagem à posição de filtração)
   RUNG wire#powerrail
      Contact( "Etapas_Grafcet".ETAPA_2 )
      Contact( "T_STOP_BOMBAS".Q )
      Contact( "Dados_Ciclo".STOP_CICLO )
      wire#w1
      S_Coil( "Etapas_Grafcet".ETAPA_9 )
   END_RUNG
   RUNG wire#powerrail
      Contact( "Etapas_Grafcet".ETAPA_3 )
      Contact( "Dados_Ciclo".STOP_CICLO )
   END_RUNG wire#w1
   RUNG wire#powerrail
      Contact( "Etapas_Grafcet".ETAPA_5 )
      Contact( "T_STOP_BOMBAS".Q )
      Contact( "Dados_Ciclo".STOP_CICLO )
   END_RUNG wire#w1
   RUNG wire#powerrail
      Contact( "Etapas_Grafcet".ETAPA_6 )
      Contact( "Dados_Ciclo".STOP_CICLO )
   END_RUNG wire#w1
   RUNG wire#powerrail
      Contact( "Etapas_Grafcet".ETAPA_8 )
      Contact( "T_STOP_BOMBAS".Q )
   END_RUNG wire#w1
   RUNG wire#powerrail
      Contact( "Etapas_Grafcet".ETAPA_12 )
      Contact( "Inputs_HMI".REARME )
   END_RUNG wire#w1
   RUNG wire#powerrail
      Contact( "Etapas_Grafcet".ETAPA_15 )
      Contact( "T_POS_EVS".Q )
      { S7_Templates := "SrcType := String" } EQ_Contact(in1 := "Dados_Ciclo".POS_EVS_FILT_1, in2 := 'FILTRACAO')
      { S7_Templates := "SrcType := String" } EQ_Contact(in1 := "Dados_Ciclo".POS_EVS_FILT_2, in2 := 'FILTRACAO')
      { S7_Templates := "SrcType := Int" } EQ_Contact(in1 := "Dados_Ciclo".ETAPA_ANTERIOR, in2 := 9)
   END_RUNG wire#w1
   RUNG wire#w1
      R_Coil( "Etapas_Grafcet".ETAPA_2 )
   END_RUNG
   RUNG wire#w1
      R_Coil( "Etapas_Grafcet".ETAPA_3 )
   END_RUNG
   RUNG wire#w1
      R_Coil( "Etapas_Grafcet".ETAPA_5 )
   END_RUNG
   RUNG wire#w1
      R_Coil( "Etapas_Grafcet".ETAPA_6 )
   END_RUNG
   RUNG wire#w1
      R_Coil( "Etapas_Grafcet".ETAPA_8 )
   END_RUNG
   RUNG wire#w1
      R_Coil( "Etapas_Grafcet".ETAPA_12 )
   END_RUNG
   RUNG wire#w1
      R_Coil( "Etapas_Grafcet".ETAPA_15 )
   END_RUNG
   // the same network as SCL:
   IF ("Etapas_Grafcet".ETAPA_2 AND "T_STOP_BOMBAS".Q AND "Dados_Ciclo".STOP_CICLO) OR ("Etapas_Grafcet".ETAPA_3 AND "Dados_Ciclo".STOP_CICLO) OR ("Etapas_Grafcet".ETAPA_5 AND "T_STOP_BOMBAS".Q AND "Dados_Ciclo".STOP_CICLO) OR ("Etapas_Grafcet".ETAPA_6 AND "Dados_Ciclo".STOP_CICLO) OR ("Etapas_Grafcet".ETAPA_8 AND "T_STOP_BOMBAS".Q) OR ("Etapas_Grafcet".ETAPA_12 AND "Inputs_HMI".REARME) OR ("Etapas_Grafcet".ETAPA_15 AND "T_POS_EVS".Q AND ("Dados_Ciclo".POS_EVS_FILT_1 = 'FILTRACAO') AND ("Dados_Ciclo".POS_EVS_FILT_2 = 'FILTRACAO') AND ("Dados_Ciclo".ETAPA_ANTERIOR = 9)) THEN
       "Etapas_Grafcet".ETAPA_9 := TRUE;
   END_IF;
   #_w1 := ("Etapas_Grafcet".ETAPA_2 AND "T_STOP_BOMBAS".Q AND "Dados_Ciclo".STOP_CICLO) OR ("Etapas_Grafcet".ETAPA_3 AND "Dados_Ciclo".STOP_CICLO) OR ("Etapas_Grafcet".ETAPA_5 AND "T_STOP_BOMBAS".Q AND "Dados_Ciclo".STOP_CICLO) OR ("Etapas_Grafcet".ETAPA_6 AND "Dados_Ciclo".STOP_CICLO) OR ("Etapas_Grafcet".ETAPA_8 AND "T_STOP_BOMBAS".Q) OR ("Etapas_Grafcet".ETAPA_12 AND "Inputs_HMI".REARME) OR ("Etapas_Grafcet".ETAPA_15 AND "T_POS_EVS".Q AND ("Dados_Ciclo".POS_EVS_FILT_1 = 'FILTRACAO') AND ("Dados_Ciclo".POS_EVS_FILT_2 = 'FILTRACAO') AND ("Dados_Ciclo".ETAPA_ANTERIOR = 9));
   IF #_w1 THEN
       "Etapas_Grafcet".ETAPA_2 := FALSE;
       "Etapas_Grafcet".ETAPA_3 := FALSE;
       "Etapas_Grafcet".ETAPA_5 := FALSE;
       "Etapas_Grafcet".ETAPA_6 := FALSE;
       "Etapas_Grafcet".ETAPA_8 := FALSE;
       "Etapas_Grafcet".ETAPA_12 := FALSE;
       "Etapas_Grafcet".ETAPA_15 := FALSE;
   END_IF;
END_REGION

REGION Network 10: ETAPA 10 (Alarme posição lavagem)
   // As ev's não estão na posição de lavagem / fecho
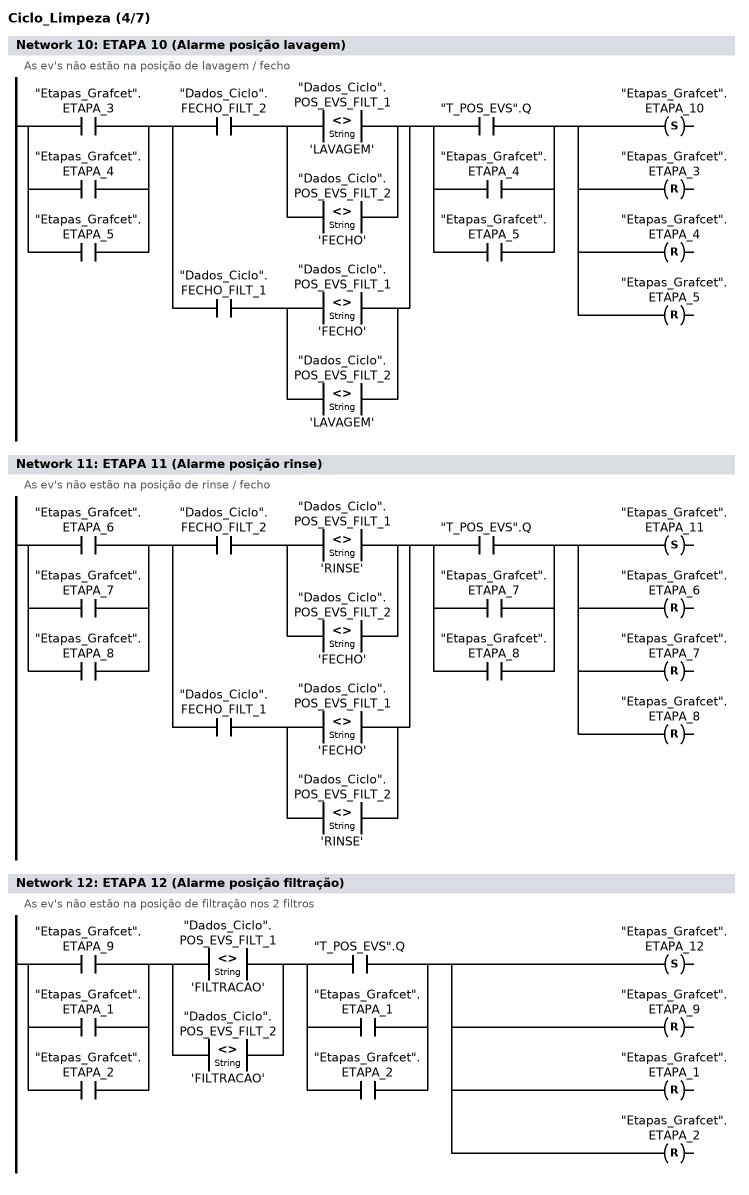
   RUNG wire#powerrail
      Contact( "Etapas_Grafcet".ETAPA_3 )
      wire#w1
      Contact( "Dados_Ciclo".FECHO_FILT_2 )
      wire#w2
      { S7_Templates := "SrcType := String" } NE_Contact(in1 := "Dados_Ciclo".POS_EVS_FILT_1, in2 := 'LAVAGEM')
      wire#w3
      Contact( "T_POS_EVS".Q )
      wire#w5
      S_Coil( "Etapas_Grafcet".ETAPA_10 )
   END_RUNG
   RUNG wire#powerrail
      Contact( "Etapas_Grafcet".ETAPA_4 )
   END_RUNG wire#w1
   RUNG wire#powerrail
      Contact( "Etapas_Grafcet".ETAPA_5 )
   END_RUNG wire#w1
   RUNG wire#w2
      { S7_Templates := "SrcType := String" } NE_Contact(in1 := "Dados_Ciclo".POS_EVS_FILT_2, in2 := 'FECHO')
   END_RUNG wire#w3
   RUNG wire#w1
      Contact( "Dados_Ciclo".FECHO_FILT_1 )
      wire#w4
      { S7_Templates := "SrcType := String" } NE_Contact(in1 := "Dados_Ciclo".POS_EVS_FILT_1, in2 := 'FECHO')
   END_RUNG wire#w3
   RUNG wire#w4
      { S7_Templates := "SrcType := String" } NE_Contact(in1 := "Dados_Ciclo".POS_EVS_FILT_2, in2 := 'LAVAGEM')
   END_RUNG wire#w3
   RUNG wire#w3
      Contact( "Etapas_Grafcet".ETAPA_4 )
   END_RUNG wire#w5
   RUNG wire#w3
      Contact( "Etapas_Grafcet".ETAPA_5 )
   END_RUNG wire#w5
   RUNG wire#w5
      R_Coil( "Etapas_Grafcet".ETAPA_3 )
   END_RUNG
   RUNG wire#w5
      R_Coil( "Etapas_Grafcet".ETAPA_4 )
   END_RUNG
   RUNG wire#w5
      R_Coil( "Etapas_Grafcet".ETAPA_5 )
   END_RUNG
   // the same network as SCL:
   IF ("Etapas_Grafcet".ETAPA_3 OR "Etapas_Grafcet".ETAPA_4 OR "Etapas_Grafcet".ETAPA_5) AND (("Dados_Ciclo".FECHO_FILT_2 AND (("Dados_Ciclo".POS_EVS_FILT_1 <> 'LAVAGEM') OR ("Dados_Ciclo".POS_EVS_FILT_2 <> 'FECHO'))) OR ("Dados_Ciclo".FECHO_FILT_1 AND (("Dados_Ciclo".POS_EVS_FILT_1 <> 'FECHO') OR ("Dados_Ciclo".POS_EVS_FILT_2 <> 'LAVAGEM')))) AND ("T_POS_EVS".Q OR "Etapas_Grafcet".ETAPA_4 OR "Etapas_Grafcet".ETAPA_5) THEN
       "Etapas_Grafcet".ETAPA_10 := TRUE;
   END_IF;
   #_w1 := ("Etapas_Grafcet".ETAPA_3 OR "Etapas_Grafcet".ETAPA_4 OR "Etapas_Grafcet".ETAPA_5) AND (("Dados_Ciclo".FECHO_FILT_2 AND (("Dados_Ciclo".POS_EVS_FILT_1 <> 'LAVAGEM') OR ("Dados_Ciclo".POS_EVS_FILT_2 <> 'FECHO'))) OR ("Dados_Ciclo".FECHO_FILT_1 AND (("Dados_Ciclo".POS_EVS_FILT_1 <> 'FECHO') OR ("Dados_Ciclo".POS_EVS_FILT_2 <> 'LAVAGEM')))) AND ("T_POS_EVS".Q OR "Etapas_Grafcet".ETAPA_4 OR "Etapas_Grafcet".ETAPA_5);
   IF #_w1 THEN
       "Etapas_Grafcet".ETAPA_3 := FALSE;
       "Etapas_Grafcet".ETAPA_4 := FALSE;
       "Etapas_Grafcet".ETAPA_5 := FALSE;
   END_IF;
END_REGION

REGION Network 11: ETAPA 11 (Alarme posição rinse)
   // As ev's não estão na posição de rinse / fecho
   RUNG wire#powerrail
      Contact( "Etapas_Grafcet".ETAPA_6 )
      wire#w1
      Contact( "Dados_Ciclo".FECHO_FILT_2 )
      wire#w2
      { S7_Templates := "SrcType := String" } NE_Contact(in1 := "Dados_Ciclo".POS_EVS_FILT_1, in2 := 'RINSE')
      wire#w3
      Contact( "T_POS_EVS".Q )
      wire#w5
      S_Coil( "Etapas_Grafcet".ETAPA_11 )
   END_RUNG
   RUNG wire#powerrail
      Contact( "Etapas_Grafcet".ETAPA_7 )
   END_RUNG wire#w1
   RUNG wire#powerrail
      Contact( "Etapas_Grafcet".ETAPA_8 )
   END_RUNG wire#w1
   RUNG wire#w2
      { S7_Templates := "SrcType := String" } NE_Contact(in1 := "Dados_Ciclo".POS_EVS_FILT_2, in2 := 'FECHO')
   END_RUNG wire#w3
   RUNG wire#w1
      Contact( "Dados_Ciclo".FECHO_FILT_1 )
      wire#w4
      { S7_Templates := "SrcType := String" } NE_Contact(in1 := "Dados_Ciclo".POS_EVS_FILT_1, in2 := 'FECHO')
   END_RUNG wire#w3
   RUNG wire#w4
      { S7_Templates := "SrcType := String" } NE_Contact(in1 := "Dados_Ciclo".POS_EVS_FILT_2, in2 := 'RINSE')
   END_RUNG wire#w3
   RUNG wire#w3
      Contact( "Etapas_Grafcet".ETAPA_7 )
   END_RUNG wire#w5
   RUNG wire#w3
      Contact( "Etapas_Grafcet".ETAPA_8 )
   END_RUNG wire#w5
   RUNG wire#w5
      R_Coil( "Etapas_Grafcet".ETAPA_6 )
   END_RUNG
   RUNG wire#w5
      R_Coil( "Etapas_Grafcet".ETAPA_7 )
   END_RUNG
   RUNG wire#w5
      R_Coil( "Etapas_Grafcet".ETAPA_8 )
   END_RUNG
   // the same network as SCL:
   IF ("Etapas_Grafcet".ETAPA_6 OR "Etapas_Grafcet".ETAPA_7 OR "Etapas_Grafcet".ETAPA_8) AND (("Dados_Ciclo".FECHO_FILT_2 AND (("Dados_Ciclo".POS_EVS_FILT_1 <> 'RINSE') OR ("Dados_Ciclo".POS_EVS_FILT_2 <> 'FECHO'))) OR ("Dados_Ciclo".FECHO_FILT_1 AND (("Dados_Ciclo".POS_EVS_FILT_1 <> 'FECHO') OR ("Dados_Ciclo".POS_EVS_FILT_2 <> 'RINSE')))) AND ("T_POS_EVS".Q OR "Etapas_Grafcet".ETAPA_7 OR "Etapas_Grafcet".ETAPA_8) THEN
       "Etapas_Grafcet".ETAPA_11 := TRUE;
   END_IF;
   #_w1 := ("Etapas_Grafcet".ETAPA_6 OR "Etapas_Grafcet".ETAPA_7 OR "Etapas_Grafcet".ETAPA_8) AND (("Dados_Ciclo".FECHO_FILT_2 AND (("Dados_Ciclo".POS_EVS_FILT_1 <> 'RINSE') OR ("Dados_Ciclo".POS_EVS_FILT_2 <> 'FECHO'))) OR ("Dados_Ciclo".FECHO_FILT_1 AND (("Dados_Ciclo".POS_EVS_FILT_1 <> 'FECHO') OR ("Dados_Ciclo".POS_EVS_FILT_2 <> 'RINSE')))) AND ("T_POS_EVS".Q OR "Etapas_Grafcet".ETAPA_7 OR "Etapas_Grafcet".ETAPA_8);
   IF #_w1 THEN
       "Etapas_Grafcet".ETAPA_6 := FALSE;
       "Etapas_Grafcet".ETAPA_7 := FALSE;
       "Etapas_Grafcet".ETAPA_8 := FALSE;
   END_IF;
END_REGION

REGION Network 12: ETAPA 12 (Alarme posição filtração)
   // As ev's não estão na posição de filtração nos 2 filtros
   RUNG wire#powerrail
      Contact( "Etapas_Grafcet".ETAPA_9 )
      wire#w1
      { S7_Templates := "SrcType := String" } NE_Contact(in1 := "Dados_Ciclo".POS_EVS_FILT_1, in2 := 'FILTRACAO')
      wire#w2
      Contact( "T_POS_EVS".Q )
      wire#w3
      S_Coil( "Etapas_Grafcet".ETAPA_12 )
   END_RUNG
   RUNG wire#powerrail
      Contact( "Etapas_Grafcet".ETAPA_1 )
   END_RUNG wire#w1
   RUNG wire#powerrail
      Contact( "Etapas_Grafcet".ETAPA_2 )
   END_RUNG wire#w1
   RUNG wire#w1
      { S7_Templates := "SrcType := String" } NE_Contact(in1 := "Dados_Ciclo".POS_EVS_FILT_2, in2 := 'FILTRACAO')
   END_RUNG wire#w2
   RUNG wire#w2
      Contact( "Etapas_Grafcet".ETAPA_1 )
   END_RUNG wire#w3
   RUNG wire#w2
      Contact( "Etapas_Grafcet".ETAPA_2 )
   END_RUNG wire#w3
   RUNG wire#w3
      R_Coil( "Etapas_Grafcet".ETAPA_9 )
   END_RUNG
   RUNG wire#w3
      R_Coil( "Etapas_Grafcet".ETAPA_1 )
   END_RUNG
   RUNG wire#w3
      R_Coil( "Etapas_Grafcet".ETAPA_2 )
   END_RUNG
   // the same network as SCL:
   IF ("Etapas_Grafcet".ETAPA_9 OR "Etapas_Grafcet".ETAPA_1 OR "Etapas_Grafcet".ETAPA_2) AND (("Dados_Ciclo".POS_EVS_FILT_1 <> 'FILTRACAO') OR ("Dados_Ciclo".POS_EVS_FILT_2 <> 'FILTRACAO')) AND ("T_POS_EVS".Q OR "Etapas_Grafcet".ETAPA_1 OR "Etapas_Grafcet".ETAPA_2) THEN
       "Etapas_Grafcet".ETAPA_12 := TRUE;
   END_IF;
   #_w1 := ("Etapas_Grafcet".ETAPA_9 OR "Etapas_Grafcet".ETAPA_1 OR "Etapas_Grafcet".ETAPA_2) AND (("Dados_Ciclo".POS_EVS_FILT_1 <> 'FILTRACAO') OR ("Dados_Ciclo".POS_EVS_FILT_2 <> 'FILTRACAO')) AND ("T_POS_EVS".Q OR "Etapas_Grafcet".ETAPA_1 OR "Etapas_Grafcet".ETAPA_2);
   IF #_w1 THEN
       "Etapas_Grafcet".ETAPA_9 := FALSE;
       "Etapas_Grafcet".ETAPA_1 := FALSE;
       "Etapas_Grafcet".ETAPA_2 := FALSE;
   END_IF;
END_REGION

REGION Network 13: Etapa 13 (Preparação para modo manual)
   // A etapa_n são as etapas de 1 a 9. A etapa 13 corresponde à preparação para entrada em manual. Param as bombas e mantém a posição das válvulas da etapa anterior. O reset às etapas de 1 a 9 é feito em Controlo_Ciclo_Manual
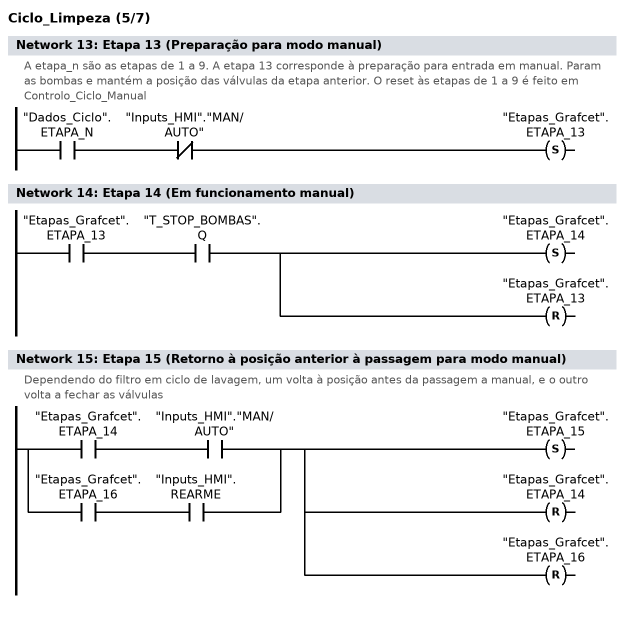
   RUNG wire#powerrail
      Contact( "Dados_Ciclo".ETAPA_N )
      I_Contact( "Inputs_HMI"."MAN/AUTO" )
      S_Coil( "Etapas_Grafcet".ETAPA_13 )
   END_RUNG
   // the same network as SCL:
   IF "Dados_Ciclo".ETAPA_N AND NOT "Inputs_HMI"."MAN/AUTO" THEN "Etapas_Grafcet".ETAPA_13 := TRUE; END_IF;
END_REGION

REGION Network 14: Etapa 14 (Em funcionamento manual)
   RUNG wire#powerrail
      Contact( "Etapas_Grafcet".ETAPA_13 )
      Contact( "T_STOP_BOMBAS".Q )
      wire#w1
      S_Coil( "Etapas_Grafcet".ETAPA_14 )
   END_RUNG
   RUNG wire#w1
      R_Coil( "Etapas_Grafcet".ETAPA_13 )
   END_RUNG
   // the same network as SCL:
   IF "Etapas_Grafcet".ETAPA_13 AND "T_STOP_BOMBAS".Q THEN
       "Etapas_Grafcet".ETAPA_14 := TRUE;
       "Etapas_Grafcet".ETAPA_13 := FALSE;
   END_IF;
END_REGION

REGION Network 15: Etapa 15 (Retorno à posição anterior à passagem para modo manual)
   // Dependendo do filtro em ciclo de lavagem, um volta à posição antes da passagem a manual, e o outro volta a fechar as válvulas
   RUNG wire#powerrail
      Contact( "Etapas_Grafcet".ETAPA_14 )
      Contact( "Inputs_HMI"."MAN/AUTO" )
      wire#w1
      S_Coil( "Etapas_Grafcet".ETAPA_15 )
   END_RUNG
   RUNG wire#powerrail
      Contact( "Etapas_Grafcet".ETAPA_16 )
      Contact( "Inputs_HMI".REARME )
   END_RUNG wire#w1
   RUNG wire#w1
      R_Coil( "Etapas_Grafcet".ETAPA_14 )
   END_RUNG
   RUNG wire#w1
      R_Coil( "Etapas_Grafcet".ETAPA_16 )
   END_RUNG
   // the same network as SCL:
   IF ("Etapas_Grafcet".ETAPA_14 AND "Inputs_HMI"."MAN/AUTO") OR ("Etapas_Grafcet".ETAPA_16 AND "Inputs_HMI".REARME) THEN
       "Etapas_Grafcet".ETAPA_15 := TRUE;
   END_IF;
   #_w1 := ("Etapas_Grafcet".ETAPA_14 AND "Inputs_HMI"."MAN/AUTO") OR ("Etapas_Grafcet".ETAPA_16 AND "Inputs_HMI".REARME);
   IF #_w1 THEN
       "Etapas_Grafcet".ETAPA_14 := FALSE;
       "Etapas_Grafcet".ETAPA_16 := FALSE;
   END_IF;
END_REGION

REGION Network 16: Etapa 16 (alarme em modo manual)
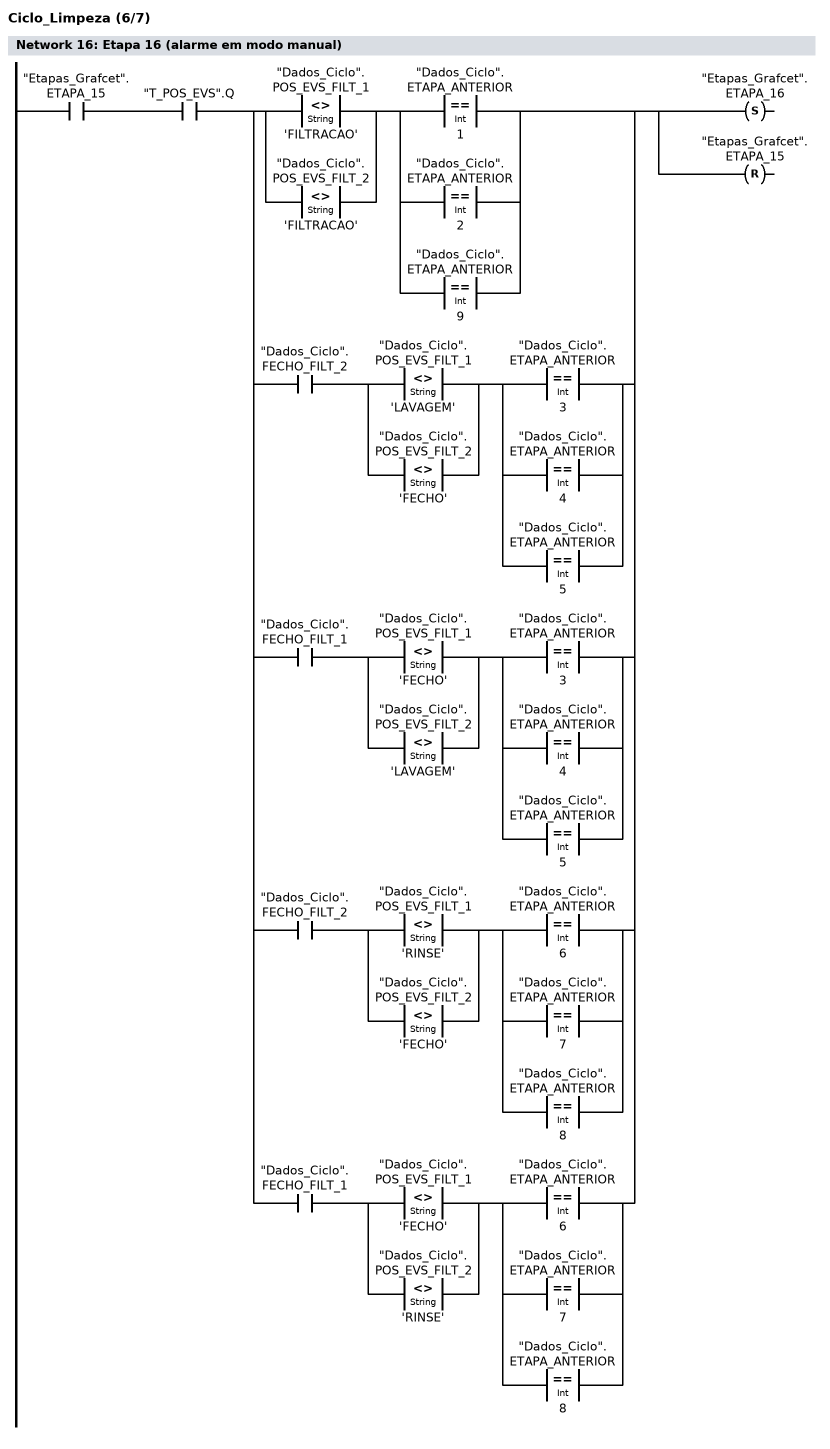
   RUNG wire#powerrail
      Contact( "Etapas_Grafcet".ETAPA_15 )
      Contact( "T_POS_EVS".Q )
      wire#w1
      { S7_Templates := "SrcType := String" } NE_Contact(in1 := "Dados_Ciclo".POS_EVS_FILT_1, in2 := 'FILTRACAO')
      wire#w2
      { S7_Templates := "SrcType := Int" } EQ_Contact(in1 := "Dados_Ciclo".ETAPA_ANTERIOR, in2 := 1)
      wire#w3
      S_Coil( "Etapas_Grafcet".ETAPA_16 )
   END_RUNG
   RUNG wire#w1
      { S7_Templates := "SrcType := String" } NE_Contact(in1 := "Dados_Ciclo".POS_EVS_FILT_2, in2 := 'FILTRACAO')
   END_RUNG wire#w2
   RUNG wire#w2
      { S7_Templates := "SrcType := Int" } EQ_Contact(in1 := "Dados_Ciclo".ETAPA_ANTERIOR, in2 := 2)
   END_RUNG wire#w3
   RUNG wire#w2
      { S7_Templates := "SrcType := Int" } EQ_Contact(in1 := "Dados_Ciclo".ETAPA_ANTERIOR, in2 := 9)
   END_RUNG wire#w3
   RUNG wire#w1
      Contact( "Dados_Ciclo".FECHO_FILT_2 )
      wire#w4
      { S7_Templates := "SrcType := String" } NE_Contact(in1 := "Dados_Ciclo".POS_EVS_FILT_1, in2 := 'LAVAGEM')
      wire#w5
      { S7_Templates := "SrcType := Int" } EQ_Contact(in1 := "Dados_Ciclo".ETAPA_ANTERIOR, in2 := 3)
   END_RUNG wire#w3
   RUNG wire#w4
      { S7_Templates := "SrcType := String" } NE_Contact(in1 := "Dados_Ciclo".POS_EVS_FILT_2, in2 := 'FECHO')
   END_RUNG wire#w5
   RUNG wire#w5
      { S7_Templates := "SrcType := Int" } EQ_Contact(in1 := "Dados_Ciclo".ETAPA_ANTERIOR, in2 := 4)
   END_RUNG wire#w3
   RUNG wire#w5
      { S7_Templates := "SrcType := Int" } EQ_Contact(in1 := "Dados_Ciclo".ETAPA_ANTERIOR, in2 := 5)
   END_RUNG wire#w3
   RUNG wire#w1
      Contact( "Dados_Ciclo".FECHO_FILT_1 )
      wire#w6
      { S7_Templates := "SrcType := String" } NE_Contact(in1 := "Dados_Ciclo".POS_EVS_FILT_1, in2 := 'FECHO')
      wire#w7
      { S7_Templates := "SrcType := Int" } EQ_Contact(in1 := "Dados_Ciclo".ETAPA_ANTERIOR, in2 := 3)
   END_RUNG wire#w3
   RUNG wire#w6
      { S7_Templates := "SrcType := String" } NE_Contact(in1 := "Dados_Ciclo".POS_EVS_FILT_2, in2 := 'LAVAGEM')
   END_RUNG wire#w7
   RUNG wire#w7
      { S7_Templates := "SrcType := Int" } EQ_Contact(in1 := "Dados_Ciclo".ETAPA_ANTERIOR, in2 := 4)
   END_RUNG wire#w3
   RUNG wire#w7
      { S7_Templates := "SrcType := Int" } EQ_Contact(in1 := "Dados_Ciclo".ETAPA_ANTERIOR, in2 := 5)
   END_RUNG wire#w3
   RUNG wire#w1
      Contact( "Dados_Ciclo".FECHO_FILT_2 )
      wire#w8
      { S7_Templates := "SrcType := String" } NE_Contact(in1 := "Dados_Ciclo".POS_EVS_FILT_1, in2 := 'RINSE')
      wire#w9
      { S7_Templates := "SrcType := Int" } EQ_Contact(in1 := "Dados_Ciclo".ETAPA_ANTERIOR, in2 := 6)
   END_RUNG wire#w3
   RUNG wire#w8
      { S7_Templates := "SrcType := String" } NE_Contact(in1 := "Dados_Ciclo".POS_EVS_FILT_2, in2 := 'FECHO')
   END_RUNG wire#w9
   RUNG wire#w9
      { S7_Templates := "SrcType := Int" } EQ_Contact(in1 := "Dados_Ciclo".ETAPA_ANTERIOR, in2 := 7)
   END_RUNG wire#w3
   RUNG wire#w9
      { S7_Templates := "SrcType := Int" } EQ_Contact(in1 := "Dados_Ciclo".ETAPA_ANTERIOR, in2 := 8)
   END_RUNG wire#w3
   RUNG wire#w1
      Contact( "Dados_Ciclo".FECHO_FILT_1 )
      wire#w10
      { S7_Templates := "SrcType := String" } NE_Contact(in1 := "Dados_Ciclo".POS_EVS_FILT_1, in2 := 'FECHO')
      wire#w11
      { S7_Templates := "SrcType := Int" } EQ_Contact(in1 := "Dados_Ciclo".ETAPA_ANTERIOR, in2 := 6)
   END_RUNG wire#w3
   RUNG wire#w10
      { S7_Templates := "SrcType := String" } NE_Contact(in1 := "Dados_Ciclo".POS_EVS_FILT_2, in2 := 'RINSE')
   END_RUNG wire#w11
   RUNG wire#w11
      { S7_Templates := "SrcType := Int" } EQ_Contact(in1 := "Dados_Ciclo".ETAPA_ANTERIOR, in2 := 7)
   END_RUNG wire#w3
   RUNG wire#w11
      { S7_Templates := "SrcType := Int" } EQ_Contact(in1 := "Dados_Ciclo".ETAPA_ANTERIOR, in2 := 8)
   END_RUNG wire#w3
   RUNG wire#w3
      R_Coil( "Etapas_Grafcet".ETAPA_15 )
   END_RUNG
   // the same network as SCL:
   IF "Etapas_Grafcet".ETAPA_15 AND "T_POS_EVS".Q AND (((("Dados_Ciclo".POS_EVS_FILT_1 <> 'FILTRACAO') OR ("Dados_Ciclo".POS_EVS_FILT_2 <> 'FILTRACAO')) AND (("Dados_Ciclo".ETAPA_ANTERIOR = 1) OR ("Dados_Ciclo".ETAPA_ANTERIOR = 2) OR ("Dados_Ciclo".ETAPA_ANTERIOR = 9))) OR ("Dados_Ciclo".FECHO_FILT_2 AND (("Dados_Ciclo".POS_EVS_FILT_1 <> 'LAVAGEM') OR ("Dados_Ciclo".POS_EVS_FILT_2 <> 'FECHO')) AND (("Dados_Ciclo".ETAPA_ANTERIOR = 3) OR ("Dados_Ciclo".ETAPA_ANTERIOR = 4) OR ("Dados_Ciclo".ETAPA_ANTERIOR = 5))) OR ("Dados_Ciclo".FECHO_FILT_1 AND (("Dados_Ciclo".POS_EVS_FILT_1 <> 'FECHO') OR ("Dados_Ciclo".POS_EVS_FILT_2 <> 'LAVAGEM')) AND (("Dados_Ciclo".ETAPA_ANTERIOR = 3) OR ("Dados_Ciclo".ETAPA_ANTERIOR = 4) OR ("Dados_Ciclo".ETAPA_ANTERIOR = 5))) OR ("Dados_Ciclo".FECHO_FILT_2 AND (("Dados_Ciclo".POS_EVS_FILT_1 <> 'RINSE') OR ("Dados_Ciclo".POS_EVS_FILT_2 <> 'FECHO')) AND (("Dados_Ciclo".ETAPA_ANTERIOR = 6) OR ("Dados_Ciclo".ETAPA_ANTERIOR = 7) OR ("Dados_Ciclo".ETAPA_ANTERIOR = 8))) OR ("Dados_Ciclo".FECHO_FILT_1 AND (("Dados_Ciclo".POS_EVS_FILT_1 <> 'FECHO') OR ("Dados_Ciclo".POS_EVS_FILT_2 <> 'RINSE')) AND (("Dados_Ciclo".ETAPA_ANTERIOR = 6) OR ("Dados_Ciclo".ETAPA_ANTERIOR = 7) OR ("Dados_Ciclo".ETAPA_ANTERIOR = 8)))) THEN
       "Etapas_Grafcet".ETAPA_16 := TRUE;
       "Etapas_Grafcet".ETAPA_15 := FALSE;
   END_IF;
END_REGION

REGION Network 17: Tempo de paragem das bombas (T1 no grafcet)
   // Espera um dado tempo para que as bombas parem, de modo a poder mudar a posição das ev's
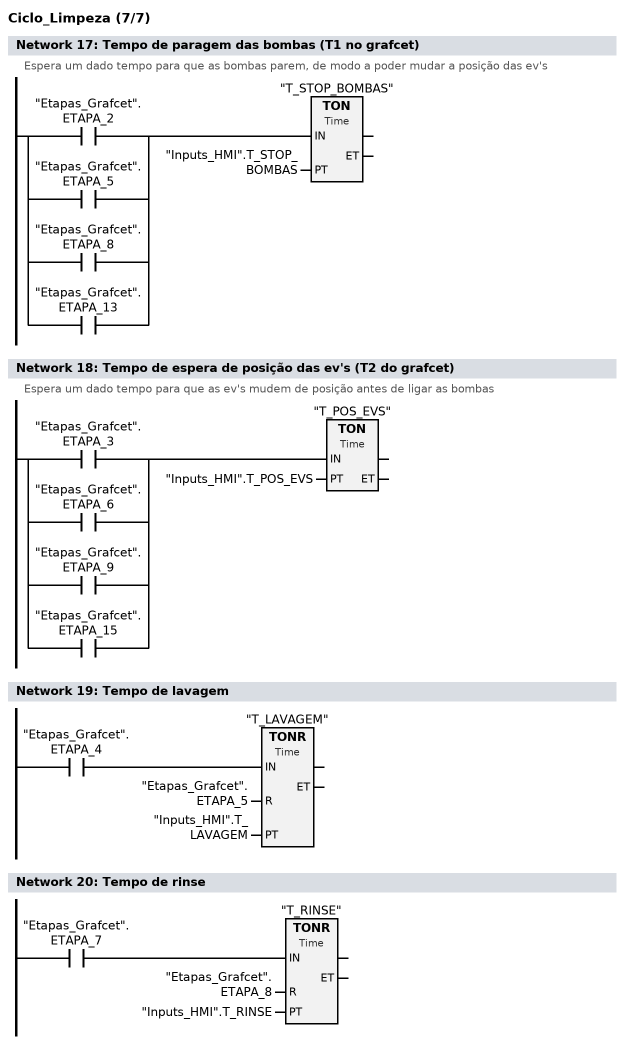
   RUNG wire#powerrail
      Contact( "Etapas_Grafcet".ETAPA_2 )
      wire#w1
      { S7_Templates := "time_type := Time" } "T_STOP_BOMBAS".TON(pt := "Inputs_HMI".T_STOP_BOMBAS, et =>)
   END_RUNG
   RUNG wire#powerrail
      Contact( "Etapas_Grafcet".ETAPA_5 )
   END_RUNG wire#w1
   RUNG wire#powerrail
      Contact( "Etapas_Grafcet".ETAPA_8 )
   END_RUNG wire#w1
   RUNG wire#powerrail
      Contact( "Etapas_Grafcet".ETAPA_13 )
   END_RUNG wire#w1
   // the same network as SCL:
   "T_STOP_BOMBAS".TON(IN := "Etapas_Grafcet".ETAPA_2 OR "Etapas_Grafcet".ETAPA_5 OR "Etapas_Grafcet".ETAPA_8 OR "Etapas_Grafcet".ETAPA_13,
                       PT := "Inputs_HMI".T_STOP_BOMBAS);
END_REGION

REGION Network 18: Tempo de espera de posição das ev's (T2 do grafcet)
   // Espera um dado tempo para que as ev's mudem de posição antes de ligar as bombas
   RUNG wire#powerrail
      Contact( "Etapas_Grafcet".ETAPA_3 )
      wire#w1
      { S7_Templates := "time_type := Time" } "T_POS_EVS".TON(pt := "Inputs_HMI".T_POS_EVS, et =>)
   END_RUNG
   RUNG wire#powerrail
      Contact( "Etapas_Grafcet".ETAPA_6 )
   END_RUNG wire#w1
   RUNG wire#powerrail
      Contact( "Etapas_Grafcet".ETAPA_9 )
   END_RUNG wire#w1
   RUNG wire#powerrail
      Contact( "Etapas_Grafcet".ETAPA_15 )
   END_RUNG wire#w1
   // the same network as SCL:
   "T_POS_EVS".TON(IN := "Etapas_Grafcet".ETAPA_3 OR "Etapas_Grafcet".ETAPA_6 OR "Etapas_Grafcet".ETAPA_9 OR "Etapas_Grafcet".ETAPA_15,
                   PT := "Inputs_HMI".T_POS_EVS);
END_REGION

REGION Network 19: Tempo de lavagem
   RUNG wire#powerrail
      Contact( "Etapas_Grafcet".ETAPA_4 )
      { S7_Templates := "time_type := Time" } "T_LAVAGEM".TONR(r := "Etapas_Grafcet".ETAPA_5, pt := "Inputs_HMI".T_LAVAGEM, et =>)
   END_RUNG
   // the same network as SCL:
   "T_LAVAGEM".TONR(IN := "Etapas_Grafcet".ETAPA_4, R := "Etapas_Grafcet".ETAPA_5, PT := "Inputs_HMI".T_LAVAGEM);
END_REGION

REGION Network 20: Tempo de rinse
   RUNG wire#powerrail
      Contact( "Etapas_Grafcet".ETAPA_7 )
      { S7_Templates := "time_type := Time" } "T_RINSE".TONR(r := "Etapas_Grafcet".ETAPA_8, pt := "Inputs_HMI".T_RINSE, et =>)
   END_RUNG
   // the same network as SCL:
   "T_RINSE".TONR(IN := "Etapas_Grafcet".ETAPA_7, R := "Etapas_Grafcet".ETAPA_8, PT := "Inputs_HMI".T_RINSE);
END_REGION
END_FUNCTION

FUNCTION "Controlo_Ciclo_Limpeza" : Void   // FC2, LAD
{ S7_Optimized_Access := 'TRUE' }
VERSION : 0.1
// stored: AutoNumber true, IsIECCheckEnabled false, SetENOAutomatically false, UDAEnableTagReadback false
   VAR_TEMP   // added for the SCL form of the ladder/FBD networks
      _w1 : Bool;
   END_VAR
BEGIN

REGION Network 1: Hold Etapa 1
   // Devido à etapa 1 fazer reset a si mesma, foi necessário criar esta memória para indicar que tal filtro está em ciclo
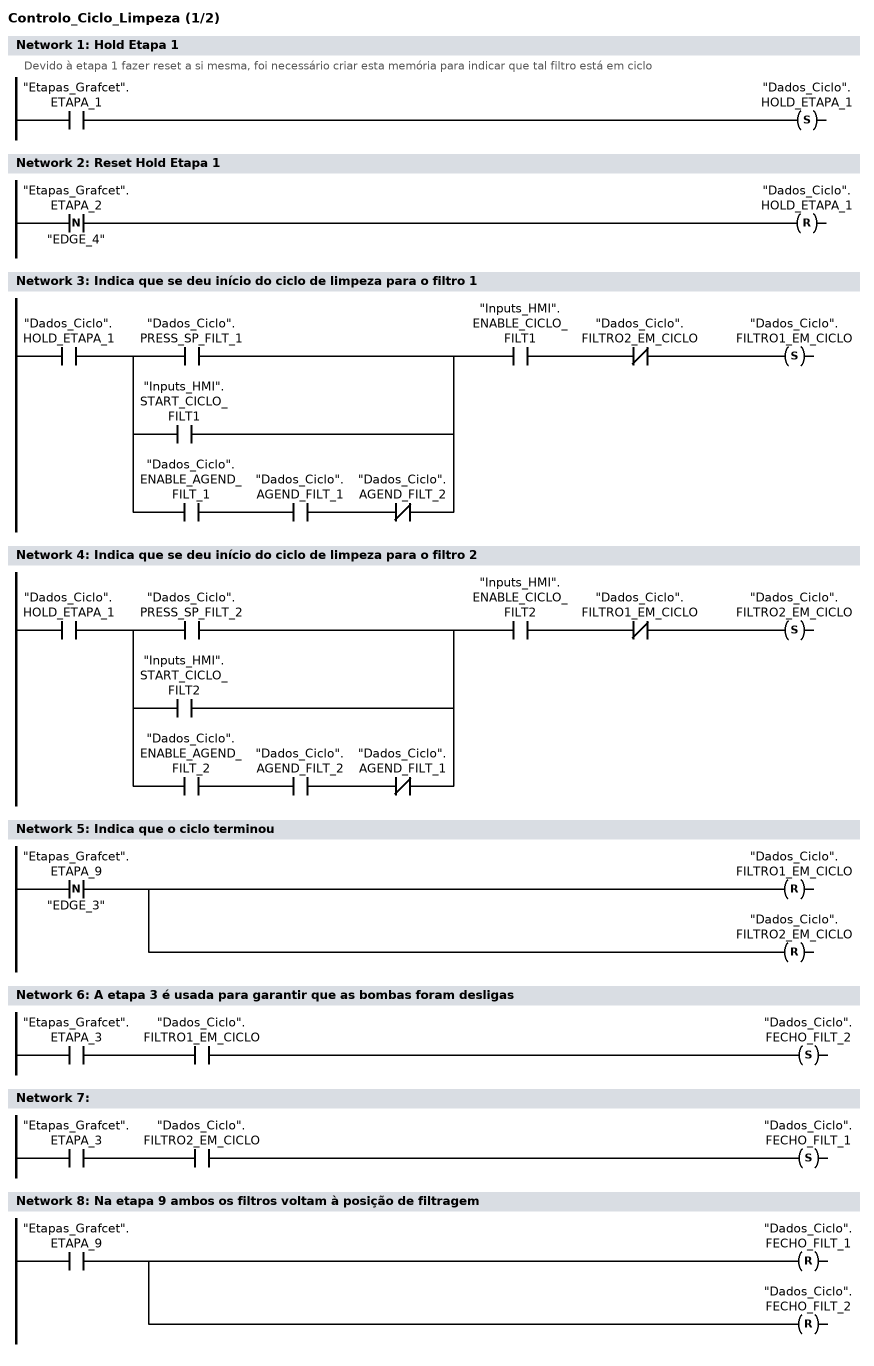
   RUNG wire#powerrail
      Contact( "Etapas_Grafcet".ETAPA_1 )
      S_Coil( "Dados_Ciclo".HOLD_ETAPA_1 )
   END_RUNG
   // the same network as SCL:
   IF "Etapas_Grafcet".ETAPA_1 THEN "Dados_Ciclo".HOLD_ETAPA_1 := TRUE; END_IF;
END_REGION

REGION Network 2: Reset Hold Etapa 1
   RUNG wire#powerrail
      N_Contact(operand := "Etapas_Grafcet".ETAPA_2, bit := "EDGE_4")
      R_Coil( "Dados_Ciclo".HOLD_ETAPA_1 )
   END_RUNG
   // the same network as SCL:
   #_w1 := NOT "Etapas_Grafcet".ETAPA_2 AND "EDGE_4";   // falling edge of "Etapas_Grafcet".ETAPA_2
   "EDGE_4" := "Etapas_Grafcet".ETAPA_2;
   IF #_w1 THEN "Dados_Ciclo".HOLD_ETAPA_1 := FALSE; END_IF;
END_REGION

REGION Network 3: Indica que se deu início do ciclo de limpeza para o filtro 1
   RUNG wire#powerrail
      Contact( "Dados_Ciclo".HOLD_ETAPA_1 )
      wire#w1
      Contact( "Dados_Ciclo".PRESS_SP_FILT_1 )
      wire#w2
      Contact( "Inputs_HMI".ENABLE_CICLO_FILT1 )
      I_Contact( "Dados_Ciclo".FILTRO2_EM_CICLO )
      S_Coil( "Dados_Ciclo".FILTRO1_EM_CICLO )
   END_RUNG
   RUNG wire#w1
      Contact( "Inputs_HMI".START_CICLO_FILT1 )
   END_RUNG wire#w2
   RUNG wire#w1
      Contact( "Dados_Ciclo".ENABLE_AGEND_FILT_1 )
      Contact( "Dados_Ciclo".AGEND_FILT_1 )
      I_Contact( "Dados_Ciclo".AGEND_FILT_2 )
   END_RUNG wire#w2
   // the same network as SCL:
   IF "Dados_Ciclo".HOLD_ETAPA_1 AND ("Dados_Ciclo".PRESS_SP_FILT_1 OR "Inputs_HMI".START_CICLO_FILT1 OR ("Dados_Ciclo".ENABLE_AGEND_FILT_1 AND "Dados_Ciclo".AGEND_FILT_1 AND NOT "Dados_Ciclo".AGEND_FILT_2)) AND "Inputs_HMI".ENABLE_CICLO_FILT1 AND NOT "Dados_Ciclo".FILTRO2_EM_CICLO THEN
       "Dados_Ciclo".FILTRO1_EM_CICLO := TRUE;
   END_IF;
END_REGION

REGION Network 4: Indica que se deu início do ciclo de limpeza para o filtro 2
   RUNG wire#powerrail
      Contact( "Dados_Ciclo".HOLD_ETAPA_1 )
      wire#w1
      Contact( "Dados_Ciclo".PRESS_SP_FILT_2 )
      wire#w2
      Contact( "Inputs_HMI".ENABLE_CICLO_FILT2 )
      I_Contact( "Dados_Ciclo".FILTRO1_EM_CICLO )
      S_Coil( "Dados_Ciclo".FILTRO2_EM_CICLO )
   END_RUNG
   RUNG wire#w1
      Contact( "Inputs_HMI".START_CICLO_FILT2 )
   END_RUNG wire#w2
   RUNG wire#w1
      Contact( "Dados_Ciclo".ENABLE_AGEND_FILT_2 )
      Contact( "Dados_Ciclo".AGEND_FILT_2 )
      I_Contact( "Dados_Ciclo".AGEND_FILT_1 )
   END_RUNG wire#w2
   // the same network as SCL:
   IF "Dados_Ciclo".HOLD_ETAPA_1 AND ("Dados_Ciclo".PRESS_SP_FILT_2 OR "Inputs_HMI".START_CICLO_FILT2 OR ("Dados_Ciclo".ENABLE_AGEND_FILT_2 AND "Dados_Ciclo".AGEND_FILT_2 AND NOT "Dados_Ciclo".AGEND_FILT_1)) AND "Inputs_HMI".ENABLE_CICLO_FILT2 AND NOT "Dados_Ciclo".FILTRO1_EM_CICLO THEN
       "Dados_Ciclo".FILTRO2_EM_CICLO := TRUE;
   END_IF;
END_REGION

REGION Network 5: Indica que o ciclo terminou
   RUNG wire#powerrail
      N_Contact(operand := "Etapas_Grafcet".ETAPA_9, bit := "EDGE_3")
      wire#w1
      R_Coil( "Dados_Ciclo".FILTRO1_EM_CICLO )
   END_RUNG
   RUNG wire#w1
      R_Coil( "Dados_Ciclo".FILTRO2_EM_CICLO )
   END_RUNG
   // the same network as SCL:
   #_w1 := NOT "Etapas_Grafcet".ETAPA_9 AND "EDGE_3";   // falling edge of "Etapas_Grafcet".ETAPA_9
   "EDGE_3" := "Etapas_Grafcet".ETAPA_9;
   IF #_w1 THEN
       "Dados_Ciclo".FILTRO1_EM_CICLO := FALSE;
       "Dados_Ciclo".FILTRO2_EM_CICLO := FALSE;
   END_IF;
END_REGION

REGION Network 6: A etapa 3 é usada para garantir que as bombas foram desligas
   RUNG wire#powerrail
      Contact( "Etapas_Grafcet".ETAPA_3 )
      Contact( "Dados_Ciclo".FILTRO1_EM_CICLO )
      S_Coil( "Dados_Ciclo".FECHO_FILT_2 )
   END_RUNG
   // the same network as SCL:
   IF "Etapas_Grafcet".ETAPA_3 AND "Dados_Ciclo".FILTRO1_EM_CICLO THEN
       "Dados_Ciclo".FECHO_FILT_2 := TRUE;
   END_IF;
END_REGION

REGION Network 7
   RUNG wire#powerrail
      Contact( "Etapas_Grafcet".ETAPA_3 )
      Contact( "Dados_Ciclo".FILTRO2_EM_CICLO )
      S_Coil( "Dados_Ciclo".FECHO_FILT_1 )
   END_RUNG
   // the same network as SCL:
   IF "Etapas_Grafcet".ETAPA_3 AND "Dados_Ciclo".FILTRO2_EM_CICLO THEN
       "Dados_Ciclo".FECHO_FILT_1 := TRUE;
   END_IF;
END_REGION

REGION Network 8: Na etapa 9 ambos os filtros voltam à posição de filtragem
   RUNG wire#powerrail
      Contact( "Etapas_Grafcet".ETAPA_9 )
      wire#w1
      R_Coil( "Dados_Ciclo".FECHO_FILT_1 )
   END_RUNG
   RUNG wire#w1
      R_Coil( "Dados_Ciclo".FECHO_FILT_2 )
   END_RUNG
   // the same network as SCL:
   IF "Etapas_Grafcet".ETAPA_9 THEN
       "Dados_Ciclo".FECHO_FILT_1 := FALSE;
       "Dados_Ciclo".FECHO_FILT_2 := FALSE;
   END_IF;
END_REGION

REGION Network 9: Set à paragem de ciclo
